// TIA Portal V17 export
// export: Created 2025-05-22T05:59:43.897412Z, ExportSetting WithDefaults, DisplayName Totally Integrated Automation Portal, DisplayVersion V17 Update 8, DisplayName TIA Portal Openness, DisplayVersion V17 Update 8, DisplayName TIA Portal Version Control Interface, DisplayVersion V17, DisplayName SINAMICS Startdrive Advanced, DisplayVersion V17 SP2, DisplayName SINAMICS Startdrive G110M, G120, G120C, G120D, G120P, G115D, DisplayVersion V17 SP2, DisplayName SINAMICS Startdrive G130, G150, S120, S150, SINAMICS MV, S210, DisplayVersion V17 SP2, DisplayName STEP 7 Professional, DisplayVersion V17 Update 8, DisplayName SINUMERIK ONE STEP 7 Toolbox, DisplayVersion V17 Update 12, DisplayName SINUMERIK ONE PLC Basic Program Plus, DisplayVersion V17 Update 12, DisplayName SINUMERIK 840D sl STEP 7 Toolbox, DisplayVersion V17 Update 12, DisplayName STEP 7 Safety, DisplayVersion V17 Update 6, DisplayName WinCC Advanced, DisplayVersion V17 Update 8
FUNCTION "FC7331_MACHINE_TO_ROBOT_CELL_INTERLOCK" : Void   // FC7331, LAD
{ S7_Optimized_Access := 'FALSE' }
AUTHOR : ETXETAR
VERSION : 1.0
// stored: AutoNumber false, IsIECCheckEnabled false, SetENOAutomatically false, UDAEnableTagReadback false
   VAR_TEMP
      OPTION_OFF : Bool;
      OPTION_ON : Bool;
      dry_load_side0 : Bool;
      dry_load_side180 : Bool;
      Status_receive : Int;
      QC_FORECAST : Int;
      QC_EXPIRED : Int;
      QC_COUNTS : Int;
      RETVAL_FILL : Int;
      temp0 : Int;
      status_sfc21 : Int;
      RETVAL_FILL_1 : Int;
      ONE : Byte;
      ZERO : Byte;
      retval_sfc21 : Int;
      Counts_for_error : Int;
      AUX_1_GTRY_SWITCH_OFF : Bool;
      AUX_2_GTRY_SWITCH_OFF : Bool;
      WITH_MANUAL_LOADER : Bool;
      WITH_OUT_MANUAL_LOADER : Bool;
      PART_TYPE_POSSIBLE : Bool;
      SHIFTING_DEVICES_OK : Bool;
      PART_ID_NEXT_FIXT : Bool;
      PART_TYPE_GTY : Bool;
      STATUS : Byte;
      RET : Byte;
   END_VAR
   VAR CONSTANT
      FC_NUMBER : DInt := 7331;   // FC NUMBER
   END_VAR
   VAR_TEMP   // added for the SCL form of the ladder/FBD networks
      _w1 : Bool;
   END_VAR
BEGIN

REGION Network 1: >>>>>>>>>>>>>>>> INTERLOCKS MACHINE TO CELL GENERAL <<<<<<<<<<<<<<<<
END_REGION

REGION Network 2: MACHINE MEASURING STATION CALIBRATION REQUIRED
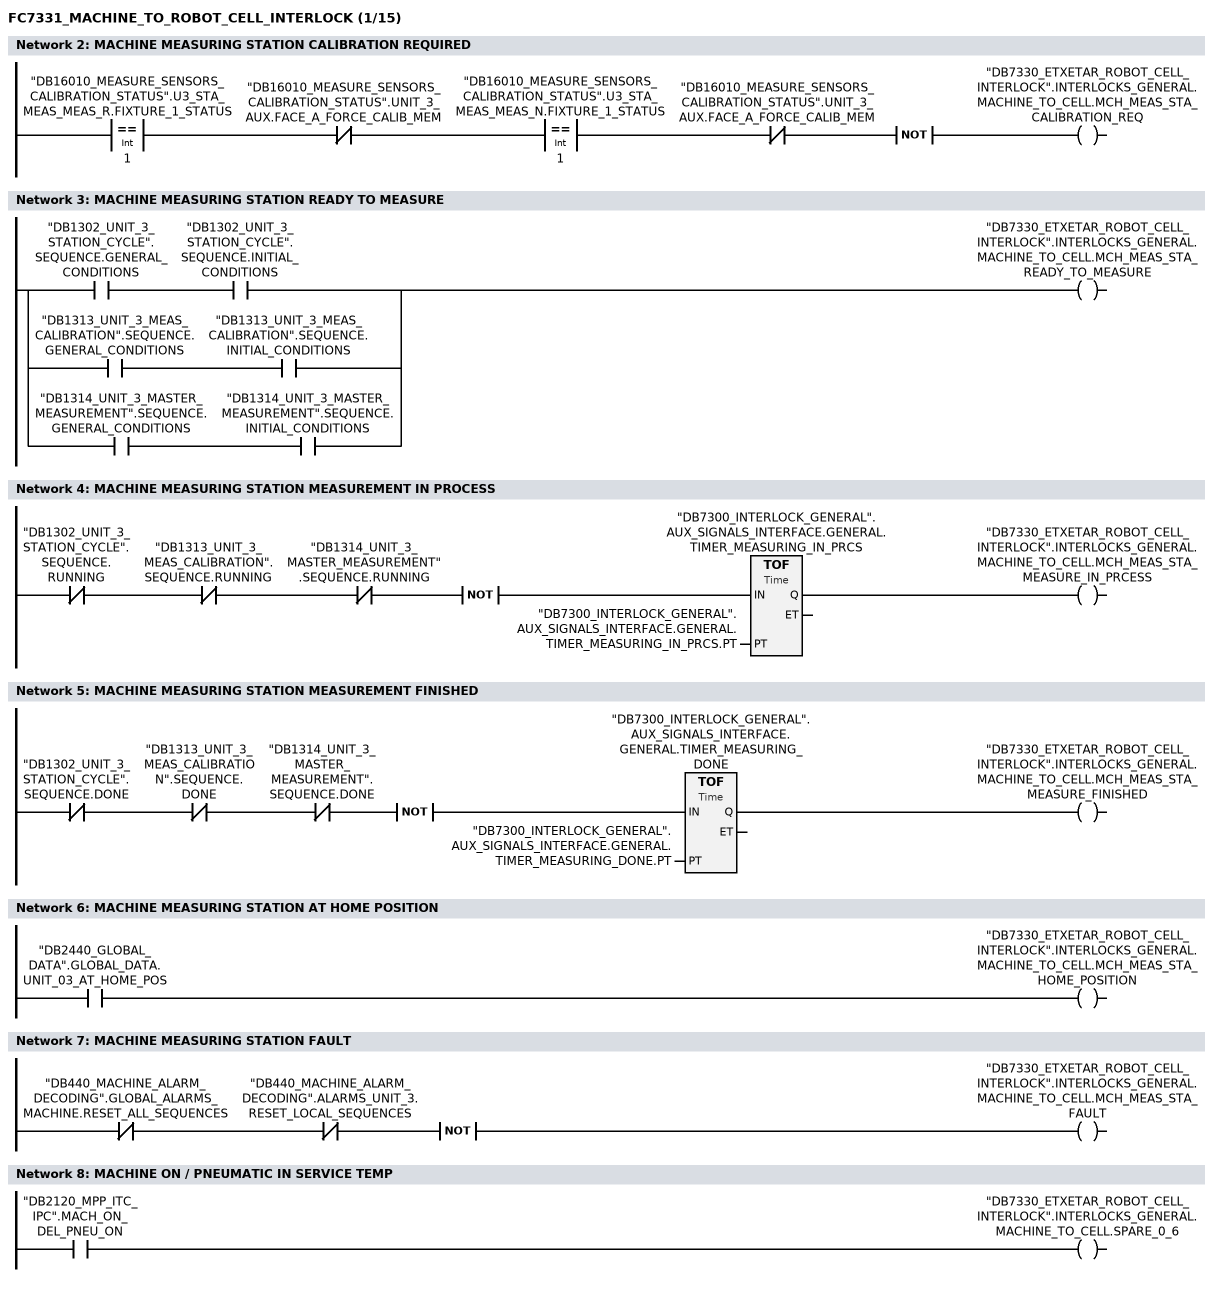
   RUNG wire#powerrail
      { S7_Templates := "SrcType := Int" } EQ_Contact(in1 := "DB16010_MEASURE_SENSORS_CALIBRATION_STATUS".U3_STA_MEAS_MEAS_R.FIXTURE_1_STATUS, in2 := 1)
      I_Contact( "DB16010_MEASURE_SENSORS_CALIBRATION_STATUS".UNIT_3_AUX.FACE_A_FORCE_CALIB_MEM )
      { S7_Templates := "SrcType := Int" } EQ_Contact(in1 := "DB16010_MEASURE_SENSORS_CALIBRATION_STATUS".U3_STA_MEAS_MEAS_N.FIXTURE_1_STATUS, in2 := 1)
      I_Contact( "DB16010_MEASURE_SENSORS_CALIBRATION_STATUS".UNIT_3_AUX.FACE_A_FORCE_CALIB_MEM )
      Not()
      Coil( "DB7330_ETXETAR_ROBOT_CELL_INTERLOCK".INTERLOCKS_GENERAL.MACHINE_TO_CELL.MCH_MEAS_STA_CALIBRATION_REQ )
   END_RUNG
   // the same network as SCL:
   "DB7330_ETXETAR_ROBOT_CELL_INTERLOCK".INTERLOCKS_GENERAL.MACHINE_TO_CELL.MCH_MEAS_STA_CALIBRATION_REQ := NOT (("DB16010_MEASURE_SENSORS_CALIBRATION_STATUS".U3_STA_MEAS_MEAS_R.FIXTURE_1_STATUS = 1) AND NOT "DB16010_MEASURE_SENSORS_CALIBRATION_STATUS".UNIT_3_AUX.FACE_A_FORCE_CALIB_MEM AND ("DB16010_MEASURE_SENSORS_CALIBRATION_STATUS".U3_STA_MEAS_MEAS_N.FIXTURE_1_STATUS = 1) AND NOT "DB16010_MEASURE_SENSORS_CALIBRATION_STATUS".UNIT_3_AUX.FACE_A_FORCE_CALIB_MEM);
END_REGION

REGION Network 3: MACHINE MEASURING STATION READY TO MEASURE
   RUNG wire#powerrail
      Contact( "DB1302_UNIT_3_STATION_CYCLE".SEQUENCE.GENERAL_CONDITIONS )
      Contact( "DB1302_UNIT_3_STATION_CYCLE".SEQUENCE.INITIAL_CONDITIONS )
      wire#w1
      Coil( "DB7330_ETXETAR_ROBOT_CELL_INTERLOCK".INTERLOCKS_GENERAL.MACHINE_TO_CELL.MCH_MEAS_STA_READY_TO_MEASURE )
   END_RUNG
   RUNG wire#powerrail
      Contact( "DB1313_UNIT_3_MEAS_CALIBRATION".SEQUENCE.GENERAL_CONDITIONS )
      Contact( "DB1313_UNIT_3_MEAS_CALIBRATION".SEQUENCE.INITIAL_CONDITIONS )
   END_RUNG wire#w1
   RUNG wire#powerrail
      Contact( "DB1314_UNIT_3_MASTER_MEASUREMENT".SEQUENCE.GENERAL_CONDITIONS )
      Contact( "DB1314_UNIT_3_MASTER_MEASUREMENT".SEQUENCE.INITIAL_CONDITIONS )
   END_RUNG wire#w1
   // the same network as SCL:
   "DB7330_ETXETAR_ROBOT_CELL_INTERLOCK".INTERLOCKS_GENERAL.MACHINE_TO_CELL.MCH_MEAS_STA_READY_TO_MEASURE := ("DB1302_UNIT_3_STATION_CYCLE".SEQUENCE.GENERAL_CONDITIONS AND "DB1302_UNIT_3_STATION_CYCLE".SEQUENCE.INITIAL_CONDITIONS) OR ("DB1313_UNIT_3_MEAS_CALIBRATION".SEQUENCE.GENERAL_CONDITIONS AND "DB1313_UNIT_3_MEAS_CALIBRATION".SEQUENCE.INITIAL_CONDITIONS) OR ("DB1314_UNIT_3_MASTER_MEASUREMENT".SEQUENCE.GENERAL_CONDITIONS AND "DB1314_UNIT_3_MASTER_MEASUREMENT".SEQUENCE.INITIAL_CONDITIONS);
END_REGION

REGION Network 4: MACHINE MEASURING STATION MEASUREMENT IN PROCESS
   RUNG wire#powerrail
      I_Contact( "DB1302_UNIT_3_STATION_CYCLE".SEQUENCE.RUNNING )
      I_Contact( "DB1313_UNIT_3_MEAS_CALIBRATION".SEQUENCE.RUNNING )
      I_Contact( "DB1314_UNIT_3_MASTER_MEASUREMENT".SEQUENCE.RUNNING )
      Not()
      { S7_Templates := "time_type := Time" } "DB7300_INTERLOCK_GENERAL".AUX_SIGNALS_INTERFACE.GENERAL.TIMER_MEASURING_IN_PRCS.TOF(pt := "DB7300_INTERLOCK_GENERAL".AUX_SIGNALS_INTERFACE.GENERAL.TIMER_MEASURING_IN_PRCS.PT, et =>)
      Coil( "DB7330_ETXETAR_ROBOT_CELL_INTERLOCK".INTERLOCKS_GENERAL.MACHINE_TO_CELL.MCH_MEAS_STA_MEASURE_IN_PRCESS )
   END_RUNG
   // the same network as SCL:
   "DB7300_INTERLOCK_GENERAL".AUX_SIGNALS_INTERFACE.GENERAL.TIMER_MEASURING_IN_PRCS.TOF(IN := NOT (NOT "DB1302_UNIT_3_STATION_CYCLE".SEQUENCE.RUNNING AND NOT "DB1313_UNIT_3_MEAS_CALIBRATION".SEQUENCE.RUNNING AND NOT "DB1314_UNIT_3_MASTER_MEASUREMENT".SEQUENCE.RUNNING),
                           PT := "DB7300_INTERLOCK_GENERAL".AUX_SIGNALS_INTERFACE.GENERAL.TIMER_MEASURING_IN_PRCS.PT);
   "DB7330_ETXETAR_ROBOT_CELL_INTERLOCK".INTERLOCKS_GENERAL.MACHINE_TO_CELL.MCH_MEAS_STA_MEASURE_IN_PRCESS := "DB7300_INTERLOCK_GENERAL".AUX_SIGNALS_INTERFACE.GENERAL.TIMER_MEASURING_IN_PRCS.Q;
END_REGION

REGION Network 5: MACHINE MEASURING STATION MEASUREMENT FINISHED
   RUNG wire#powerrail
      I_Contact( "DB1302_UNIT_3_STATION_CYCLE".SEQUENCE.DONE )
      I_Contact( "DB1313_UNIT_3_MEAS_CALIBRATION".SEQUENCE.DONE )
      I_Contact( "DB1314_UNIT_3_MASTER_MEASUREMENT".SEQUENCE.DONE )
      Not()
      { S7_Templates := "time_type := Time" } "DB7300_INTERLOCK_GENERAL".AUX_SIGNALS_INTERFACE.GENERAL.TIMER_MEASURING_DONE.TOF(pt := "DB7300_INTERLOCK_GENERAL".AUX_SIGNALS_INTERFACE.GENERAL.TIMER_MEASURING_DONE.PT, et =>)
      Coil( "DB7330_ETXETAR_ROBOT_CELL_INTERLOCK".INTERLOCKS_GENERAL.MACHINE_TO_CELL.MCH_MEAS_STA_MEASURE_FINISHED )
   END_RUNG
   // the same network as SCL:
   "DB7300_INTERLOCK_GENERAL".AUX_SIGNALS_INTERFACE.GENERAL.TIMER_MEASURING_DONE.TOF(IN := NOT (NOT "DB1302_UNIT_3_STATION_CYCLE".SEQUENCE.DONE AND NOT "DB1313_UNIT_3_MEAS_CALIBRATION".SEQUENCE.DONE AND NOT "DB1314_UNIT_3_MASTER_MEASUREMENT".SEQUENCE.DONE),
                           PT := "DB7300_INTERLOCK_GENERAL".AUX_SIGNALS_INTERFACE.GENERAL.TIMER_MEASURING_DONE.PT);
   "DB7330_ETXETAR_ROBOT_CELL_INTERLOCK".INTERLOCKS_GENERAL.MACHINE_TO_CELL.MCH_MEAS_STA_MEASURE_FINISHED := "DB7300_INTERLOCK_GENERAL".AUX_SIGNALS_INTERFACE.GENERAL.TIMER_MEASURING_DONE.Q;
END_REGION

REGION Network 6: MACHINE MEASURING STATION AT HOME POSITION
   RUNG wire#powerrail
      Contact( "DB2440_GLOBAL_DATA".GLOBAL_DATA.UNIT_03_AT_HOME_POS )
      Coil( "DB7330_ETXETAR_ROBOT_CELL_INTERLOCK".INTERLOCKS_GENERAL.MACHINE_TO_CELL.MCH_MEAS_STA_HOME_POSITION )
   END_RUNG
   // the same network as SCL:
   "DB7330_ETXETAR_ROBOT_CELL_INTERLOCK".INTERLOCKS_GENERAL.MACHINE_TO_CELL.MCH_MEAS_STA_HOME_POSITION := "DB2440_GLOBAL_DATA".GLOBAL_DATA.UNIT_03_AT_HOME_POS;
END_REGION

REGION Network 7: MACHINE MEASURING STATION FAULT
   RUNG wire#powerrail
      I_Contact( "DB440_MACHINE_ALARM_DECODING".GLOBAL_ALARMS_MACHINE.RESET_ALL_SEQUENCES )
      I_Contact( "DB440_MACHINE_ALARM_DECODING".ALARMS_UNIT_3.RESET_LOCAL_SEQUENCES )
      Not()
      Coil( "DB7330_ETXETAR_ROBOT_CELL_INTERLOCK".INTERLOCKS_GENERAL.MACHINE_TO_CELL.MCH_MEAS_STA_FAULT )
   END_RUNG
   // the same network as SCL:
   "DB7330_ETXETAR_ROBOT_CELL_INTERLOCK".INTERLOCKS_GENERAL.MACHINE_TO_CELL.MCH_MEAS_STA_FAULT := NOT (NOT "DB440_MACHINE_ALARM_DECODING".GLOBAL_ALARMS_MACHINE.RESET_ALL_SEQUENCES AND NOT "DB440_MACHINE_ALARM_DECODING".ALARMS_UNIT_3.RESET_LOCAL_SEQUENCES);
END_REGION

REGION Network 8: MACHINE ON / PNEUMATIC IN SERVICE TEMP
   RUNG wire#powerrail
      Contact( "DB2120_MPP_ITC_IPC".MACH_ON_DEL_PNEU_ON )
      Coil( "DB7330_ETXETAR_ROBOT_CELL_INTERLOCK".INTERLOCKS_GENERAL.MACHINE_TO_CELL.SPARE_0_6 )
   END_RUNG
   // the same network as SCL:
   "DB7330_ETXETAR_ROBOT_CELL_INTERLOCK".INTERLOCKS_GENERAL.MACHINE_TO_CELL.SPARE_0_6 := "DB2120_MPP_ITC_IPC".MACH_ON_DEL_PNEU_ON;
END_REGION

REGION Network 9: MACHINE MEASURING STATION MICROEPSILON FACE R ENABLED
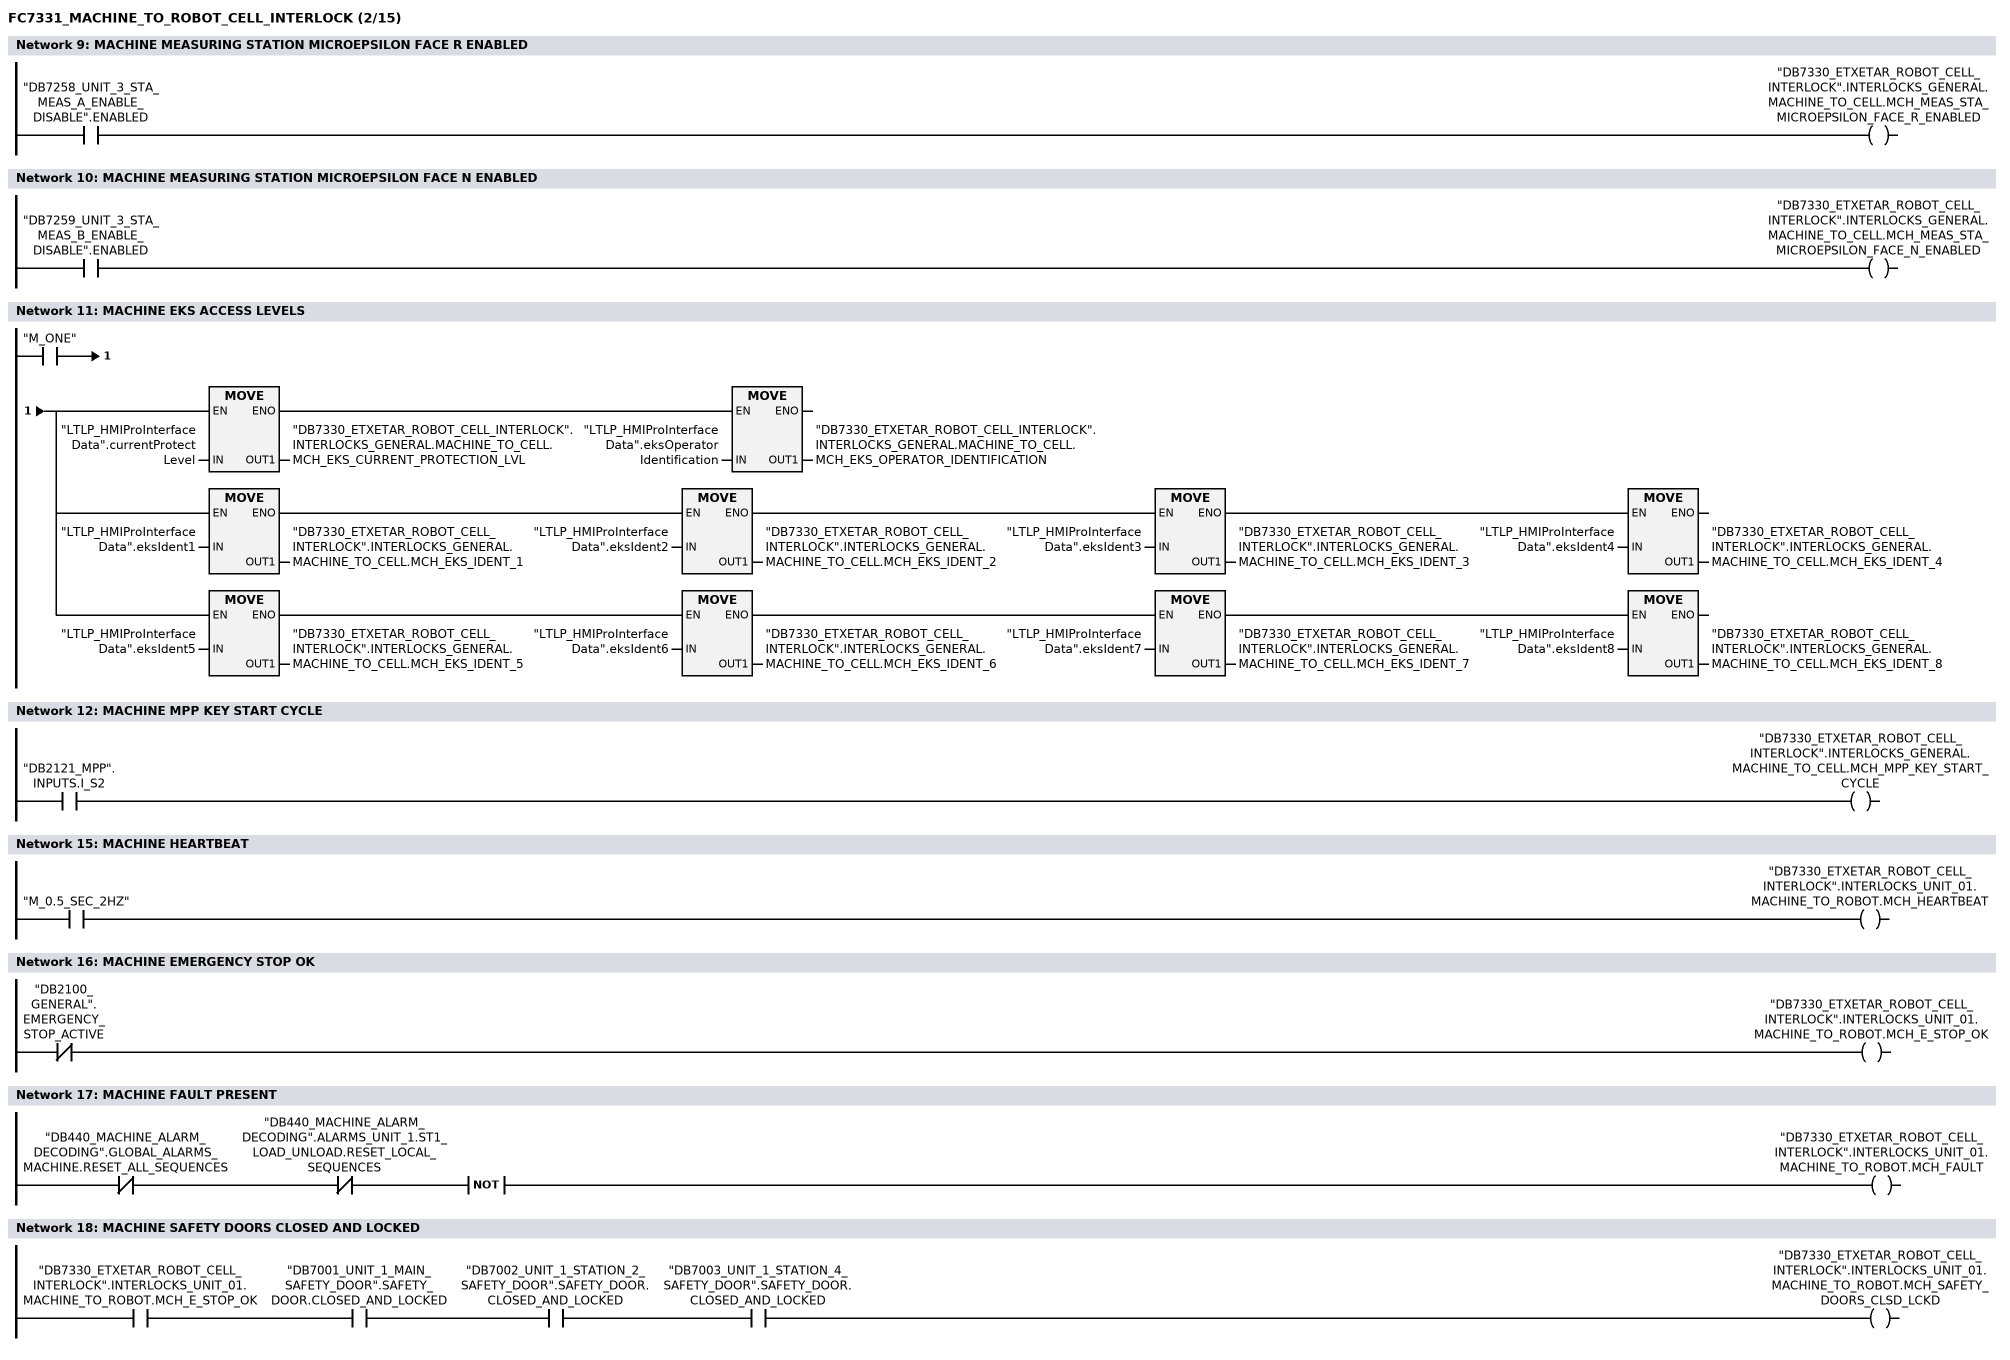
   RUNG wire#powerrail
      Contact( "DB7258_UNIT_3_STA_MEAS_A_ENABLE_DISABLE".ENABLED )
      Coil( "DB7330_ETXETAR_ROBOT_CELL_INTERLOCK".INTERLOCKS_GENERAL.MACHINE_TO_CELL.MCH_MEAS_STA_MICROEPSILON_FACE_R_ENABLED )
   END_RUNG
   // the same network as SCL:
   "DB7330_ETXETAR_ROBOT_CELL_INTERLOCK".INTERLOCKS_GENERAL.MACHINE_TO_CELL.MCH_MEAS_STA_MICROEPSILON_FACE_R_ENABLED := "DB7258_UNIT_3_STA_MEAS_A_ENABLE_DISABLE".ENABLED;
END_REGION

REGION Network 10: MACHINE MEASURING STATION MICROEPSILON FACE N ENABLED
   RUNG wire#powerrail
      Contact( "DB7259_UNIT_3_STA_MEAS_B_ENABLE_DISABLE".ENABLED )
      Coil( "DB7330_ETXETAR_ROBOT_CELL_INTERLOCK".INTERLOCKS_GENERAL.MACHINE_TO_CELL.MCH_MEAS_STA_MICROEPSILON_FACE_N_ENABLED )
   END_RUNG
   // the same network as SCL:
   "DB7330_ETXETAR_ROBOT_CELL_INTERLOCK".INTERLOCKS_GENERAL.MACHINE_TO_CELL.MCH_MEAS_STA_MICROEPSILON_FACE_N_ENABLED := "DB7259_UNIT_3_STA_MEAS_B_ENABLE_DISABLE".ENABLED;
END_REGION

REGION Network 11: MACHINE EKS ACCESS LEVELS
   RUNG wire#powerrail
      Contact( "M_ONE" )
      wire#w1
      Move(in := "LTLP_HMIProInterfaceData".currentProtectLevel, out1 => "DB7330_ETXETAR_ROBOT_CELL_INTERLOCK".INTERLOCKS_GENERAL.MACHINE_TO_CELL.MCH_EKS_CURRENT_PROTECTION_LVL)
      Move(in := "LTLP_HMIProInterfaceData".eksOperatorIdentification, out1 => "DB7330_ETXETAR_ROBOT_CELL_INTERLOCK".INTERLOCKS_GENERAL.MACHINE_TO_CELL.MCH_EKS_OPERATOR_IDENTIFICATION)
   END_RUNG
   RUNG wire#w1
      Move(in := "LTLP_HMIProInterfaceData".eksIdent1, out1 => "DB7330_ETXETAR_ROBOT_CELL_INTERLOCK".INTERLOCKS_GENERAL.MACHINE_TO_CELL.MCH_EKS_IDENT_1)
      Move(in := "LTLP_HMIProInterfaceData".eksIdent2, out1 => "DB7330_ETXETAR_ROBOT_CELL_INTERLOCK".INTERLOCKS_GENERAL.MACHINE_TO_CELL.MCH_EKS_IDENT_2)
      Move(in := "LTLP_HMIProInterfaceData".eksIdent3, out1 => "DB7330_ETXETAR_ROBOT_CELL_INTERLOCK".INTERLOCKS_GENERAL.MACHINE_TO_CELL.MCH_EKS_IDENT_3)
      Move(in := "LTLP_HMIProInterfaceData".eksIdent4, out1 => "DB7330_ETXETAR_ROBOT_CELL_INTERLOCK".INTERLOCKS_GENERAL.MACHINE_TO_CELL.MCH_EKS_IDENT_4)
   END_RUNG
   RUNG wire#w1
      Move(in := "LTLP_HMIProInterfaceData".eksIdent5, out1 => "DB7330_ETXETAR_ROBOT_CELL_INTERLOCK".INTERLOCKS_GENERAL.MACHINE_TO_CELL.MCH_EKS_IDENT_5)
      Move(in := "LTLP_HMIProInterfaceData".eksIdent6, out1 => "DB7330_ETXETAR_ROBOT_CELL_INTERLOCK".INTERLOCKS_GENERAL.MACHINE_TO_CELL.MCH_EKS_IDENT_6)
      Move(in := "LTLP_HMIProInterfaceData".eksIdent7, out1 => "DB7330_ETXETAR_ROBOT_CELL_INTERLOCK".INTERLOCKS_GENERAL.MACHINE_TO_CELL.MCH_EKS_IDENT_7)
      Move(in := "LTLP_HMIProInterfaceData".eksIdent8, out1 => "DB7330_ETXETAR_ROBOT_CELL_INTERLOCK".INTERLOCKS_GENERAL.MACHINE_TO_CELL.MCH_EKS_IDENT_8)
   END_RUNG
   // the same network as SCL:
   IF "M_ONE" THEN
       "DB7330_ETXETAR_ROBOT_CELL_INTERLOCK".INTERLOCKS_GENERAL.MACHINE_TO_CELL.MCH_EKS_CURRENT_PROTECTION_LVL := "LTLP_HMIProInterfaceData".currentProtectLevel;
       "DB7330_ETXETAR_ROBOT_CELL_INTERLOCK".INTERLOCKS_GENERAL.MACHINE_TO_CELL.MCH_EKS_OPERATOR_IDENTIFICATION := "LTLP_HMIProInterfaceData".eksOperatorIdentification;
       "DB7330_ETXETAR_ROBOT_CELL_INTERLOCK".INTERLOCKS_GENERAL.MACHINE_TO_CELL.MCH_EKS_IDENT_1 := "LTLP_HMIProInterfaceData".eksIdent1;
       "DB7330_ETXETAR_ROBOT_CELL_INTERLOCK".INTERLOCKS_GENERAL.MACHINE_TO_CELL.MCH_EKS_IDENT_2 := "LTLP_HMIProInterfaceData".eksIdent2;
       "DB7330_ETXETAR_ROBOT_CELL_INTERLOCK".INTERLOCKS_GENERAL.MACHINE_TO_CELL.MCH_EKS_IDENT_3 := "LTLP_HMIProInterfaceData".eksIdent3;
       "DB7330_ETXETAR_ROBOT_CELL_INTERLOCK".INTERLOCKS_GENERAL.MACHINE_TO_CELL.MCH_EKS_IDENT_4 := "LTLP_HMIProInterfaceData".eksIdent4;
       "DB7330_ETXETAR_ROBOT_CELL_INTERLOCK".INTERLOCKS_GENERAL.MACHINE_TO_CELL.MCH_EKS_IDENT_5 := "LTLP_HMIProInterfaceData".eksIdent5;
       "DB7330_ETXETAR_ROBOT_CELL_INTERLOCK".INTERLOCKS_GENERAL.MACHINE_TO_CELL.MCH_EKS_IDENT_6 := "LTLP_HMIProInterfaceData".eksIdent6;
       "DB7330_ETXETAR_ROBOT_CELL_INTERLOCK".INTERLOCKS_GENERAL.MACHINE_TO_CELL.MCH_EKS_IDENT_7 := "LTLP_HMIProInterfaceData".eksIdent7;
       "DB7330_ETXETAR_ROBOT_CELL_INTERLOCK".INTERLOCKS_GENERAL.MACHINE_TO_CELL.MCH_EKS_IDENT_8 := "LTLP_HMIProInterfaceData".eksIdent8;
   END_IF;
END_REGION

REGION Network 12: MACHINE MPP KEY START CYCLE
   RUNG wire#powerrail
      Contact( "DB2121_MPP".INPUTS.I_S2 )
      Coil( "DB7330_ETXETAR_ROBOT_CELL_INTERLOCK".INTERLOCKS_GENERAL.MACHINE_TO_CELL.MCH_MPP_KEY_START_CYCLE )
   END_RUNG
   // the same network as SCL:
   "DB7330_ETXETAR_ROBOT_CELL_INTERLOCK".INTERLOCKS_GENERAL.MACHINE_TO_CELL.MCH_MPP_KEY_START_CYCLE := "DB2121_MPP".INPUTS.I_S2;
END_REGION

REGION Network 14: >>>>>>>>>>>>>>>> INTERLOCKS MACHINE TO ROBOT UNIT 01 <<<<<<<<<<<<<<<<
END_REGION

REGION Network 15: MACHINE HEARTBEAT
   RUNG wire#powerrail
      Contact( "M_0.5_SEC_2HZ" )
      Coil( "DB7330_ETXETAR_ROBOT_CELL_INTERLOCK".INTERLOCKS_UNIT_01.MACHINE_TO_ROBOT.MCH_HEARTBEAT )
   END_RUNG
   // the same network as SCL:
   "DB7330_ETXETAR_ROBOT_CELL_INTERLOCK".INTERLOCKS_UNIT_01.MACHINE_TO_ROBOT.MCH_HEARTBEAT := "M_0.5_SEC_2HZ";
END_REGION

REGION Network 16: MACHINE EMERGENCY STOP OK
   RUNG wire#powerrail
      I_Contact( "DB2100_GENERAL".EMERGENCY_STOP_ACTIVE )
      Coil( "DB7330_ETXETAR_ROBOT_CELL_INTERLOCK".INTERLOCKS_UNIT_01.MACHINE_TO_ROBOT.MCH_E_STOP_OK )
   END_RUNG
   // the same network as SCL:
   "DB7330_ETXETAR_ROBOT_CELL_INTERLOCK".INTERLOCKS_UNIT_01.MACHINE_TO_ROBOT.MCH_E_STOP_OK := NOT "DB2100_GENERAL".EMERGENCY_STOP_ACTIVE;
END_REGION

REGION Network 17: MACHINE FAULT PRESENT
   RUNG wire#powerrail
      I_Contact( "DB440_MACHINE_ALARM_DECODING".GLOBAL_ALARMS_MACHINE.RESET_ALL_SEQUENCES )
      I_Contact( "DB440_MACHINE_ALARM_DECODING".ALARMS_UNIT_1.ST1_LOAD_UNLOAD.RESET_LOCAL_SEQUENCES )
      Not()
      Coil( "DB7330_ETXETAR_ROBOT_CELL_INTERLOCK".INTERLOCKS_UNIT_01.MACHINE_TO_ROBOT.MCH_FAULT )
   END_RUNG
   // the same network as SCL:
   "DB7330_ETXETAR_ROBOT_CELL_INTERLOCK".INTERLOCKS_UNIT_01.MACHINE_TO_ROBOT.MCH_FAULT := NOT (NOT "DB440_MACHINE_ALARM_DECODING".GLOBAL_ALARMS_MACHINE.RESET_ALL_SEQUENCES AND NOT "DB440_MACHINE_ALARM_DECODING".ALARMS_UNIT_1.ST1_LOAD_UNLOAD.RESET_LOCAL_SEQUENCES);
END_REGION

REGION Network 18: MACHINE SAFETY DOORS CLOSED AND LOCKED
   RUNG wire#powerrail
      Contact( "DB7330_ETXETAR_ROBOT_CELL_INTERLOCK".INTERLOCKS_UNIT_01.MACHINE_TO_ROBOT.MCH_E_STOP_OK )
      Contact( "DB7001_UNIT_1_MAIN_SAFETY_DOOR".SAFETY_DOOR.CLOSED_AND_LOCKED )
      Contact( "DB7002_UNIT_1_STATION_2_SAFETY_DOOR".SAFETY_DOOR.CLOSED_AND_LOCKED )
      Contact( "DB7003_UNIT_1_STATION_4_SAFETY_DOOR".SAFETY_DOOR.CLOSED_AND_LOCKED )
      Coil( "DB7330_ETXETAR_ROBOT_CELL_INTERLOCK".INTERLOCKS_UNIT_01.MACHINE_TO_ROBOT.MCH_SAFETY_DOORS_CLSD_LCKD )
   END_RUNG
   // the same network as SCL:
   "DB7330_ETXETAR_ROBOT_CELL_INTERLOCK".INTERLOCKS_UNIT_01.MACHINE_TO_ROBOT.MCH_SAFETY_DOORS_CLSD_LCKD := "DB7330_ETXETAR_ROBOT_CELL_INTERLOCK".INTERLOCKS_UNIT_01.MACHINE_TO_ROBOT.MCH_E_STOP_OK AND "DB7001_UNIT_1_MAIN_SAFETY_DOOR".SAFETY_DOOR.CLOSED_AND_LOCKED AND "DB7002_UNIT_1_STATION_2_SAFETY_DOOR".SAFETY_DOOR.CLOSED_AND_LOCKED AND "DB7003_UNIT_1_STATION_4_SAFETY_DOOR".SAFETY_DOOR.CLOSED_AND_LOCKED;
END_REGION

REGION Network 19: MACHINE MANUAL MODE SELECTED
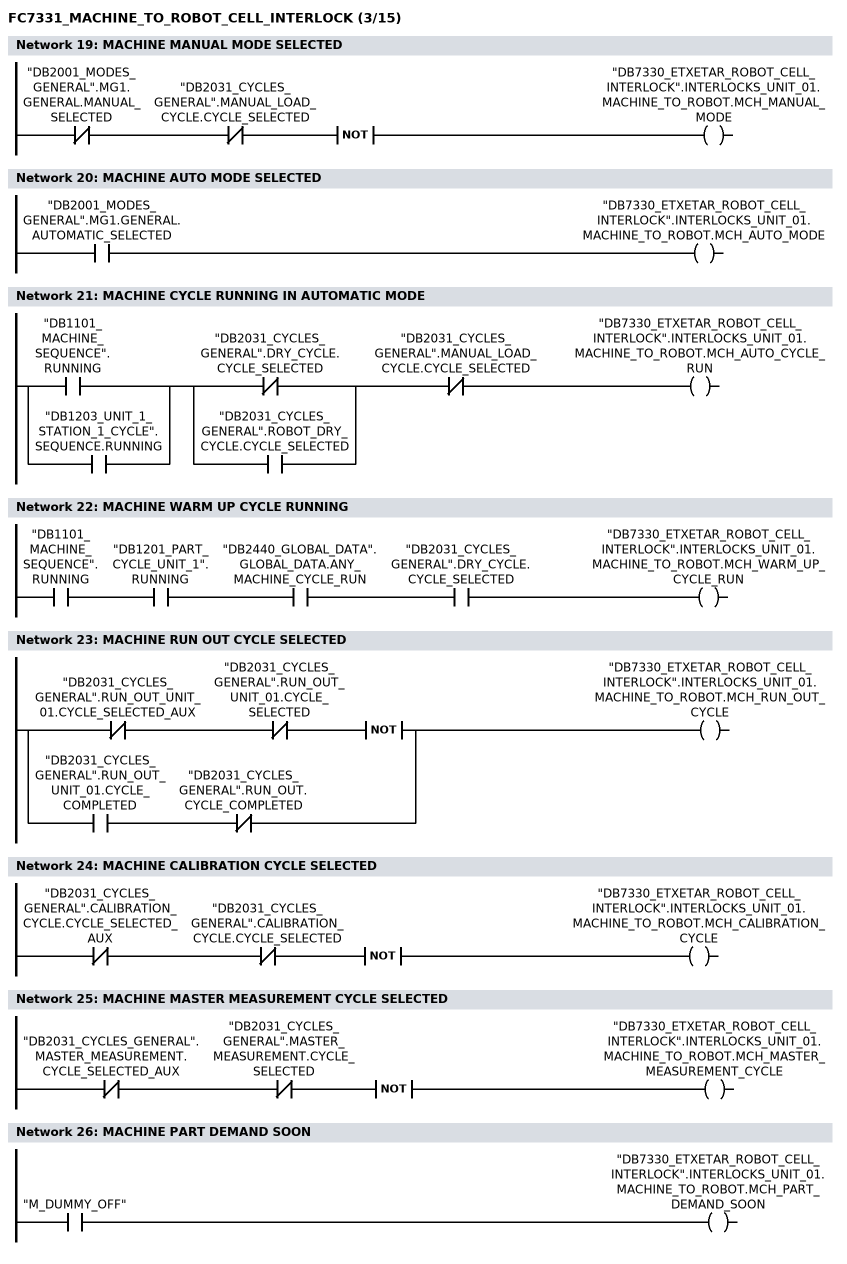
   RUNG wire#powerrail
      I_Contact( "DB2001_MODES_GENERAL".MG1.GENERAL.MANUAL_SELECTED )
      I_Contact( "DB2031_CYCLES_GENERAL".MANUAL_LOAD_CYCLE.CYCLE_SELECTED )
      Not()
      Coil( "DB7330_ETXETAR_ROBOT_CELL_INTERLOCK".INTERLOCKS_UNIT_01.MACHINE_TO_ROBOT.MCH_MANUAL_MODE )
   END_RUNG
   // the same network as SCL:
   "DB7330_ETXETAR_ROBOT_CELL_INTERLOCK".INTERLOCKS_UNIT_01.MACHINE_TO_ROBOT.MCH_MANUAL_MODE := NOT (NOT "DB2001_MODES_GENERAL".MG1.GENERAL.MANUAL_SELECTED AND NOT "DB2031_CYCLES_GENERAL".MANUAL_LOAD_CYCLE.CYCLE_SELECTED);
END_REGION

REGION Network 20: MACHINE AUTO MODE SELECTED
   RUNG wire#powerrail
      Contact( "DB2001_MODES_GENERAL".MG1.GENERAL.AUTOMATIC_SELECTED )
      Coil( "DB7330_ETXETAR_ROBOT_CELL_INTERLOCK".INTERLOCKS_UNIT_01.MACHINE_TO_ROBOT.MCH_AUTO_MODE )
   END_RUNG
   // the same network as SCL:
   "DB7330_ETXETAR_ROBOT_CELL_INTERLOCK".INTERLOCKS_UNIT_01.MACHINE_TO_ROBOT.MCH_AUTO_MODE := "DB2001_MODES_GENERAL".MG1.GENERAL.AUTOMATIC_SELECTED;
END_REGION

REGION Network 21: MACHINE CYCLE RUNNING IN AUTOMATIC MODE
   RUNG wire#powerrail
      Contact( "DB1101_MACHINE_SEQUENCE".RUNNING )
      wire#w1
      I_Contact( "DB2031_CYCLES_GENERAL".DRY_CYCLE.CYCLE_SELECTED )
      wire#w2
      I_Contact( "DB2031_CYCLES_GENERAL".MANUAL_LOAD_CYCLE.CYCLE_SELECTED )
      Coil( "DB7330_ETXETAR_ROBOT_CELL_INTERLOCK".INTERLOCKS_UNIT_01.MACHINE_TO_ROBOT.MCH_AUTO_CYCLE_RUN )
   END_RUNG
   RUNG wire#powerrail
      Contact( "DB1203_UNIT_1_STATION_1_CYCLE".SEQUENCE.RUNNING )
   END_RUNG wire#w1
   RUNG wire#w1
      Contact( "DB2031_CYCLES_GENERAL".ROBOT_DRY_CYCLE.CYCLE_SELECTED )
   END_RUNG wire#w2
   // the same network as SCL:
   "DB7330_ETXETAR_ROBOT_CELL_INTERLOCK".INTERLOCKS_UNIT_01.MACHINE_TO_ROBOT.MCH_AUTO_CYCLE_RUN := ("DB1101_MACHINE_SEQUENCE".RUNNING OR "DB1203_UNIT_1_STATION_1_CYCLE".SEQUENCE.RUNNING) AND (NOT "DB2031_CYCLES_GENERAL".DRY_CYCLE.CYCLE_SELECTED OR "DB2031_CYCLES_GENERAL".ROBOT_DRY_CYCLE.CYCLE_SELECTED) AND NOT "DB2031_CYCLES_GENERAL".MANUAL_LOAD_CYCLE.CYCLE_SELECTED;
END_REGION

REGION Network 22: MACHINE WARM UP CYCLE RUNNING
   RUNG wire#powerrail
      Contact( "DB1101_MACHINE_SEQUENCE".RUNNING )
      Contact( "DB1201_PART_CYCLE_UNIT_1".RUNNING )
      Contact( "DB2440_GLOBAL_DATA".GLOBAL_DATA.ANY_MACHINE_CYCLE_RUN )
      Contact( "DB2031_CYCLES_GENERAL".DRY_CYCLE.CYCLE_SELECTED )
      Coil( "DB7330_ETXETAR_ROBOT_CELL_INTERLOCK".INTERLOCKS_UNIT_01.MACHINE_TO_ROBOT.MCH_WARM_UP_CYCLE_RUN )
   END_RUNG
   // the same network as SCL:
   "DB7330_ETXETAR_ROBOT_CELL_INTERLOCK".INTERLOCKS_UNIT_01.MACHINE_TO_ROBOT.MCH_WARM_UP_CYCLE_RUN := "DB1101_MACHINE_SEQUENCE".RUNNING AND "DB1201_PART_CYCLE_UNIT_1".RUNNING AND "DB2440_GLOBAL_DATA".GLOBAL_DATA.ANY_MACHINE_CYCLE_RUN AND "DB2031_CYCLES_GENERAL".DRY_CYCLE.CYCLE_SELECTED;
END_REGION

REGION Network 23: MACHINE RUN OUT CYCLE SELECTED
   RUNG wire#powerrail
      I_Contact( "DB2031_CYCLES_GENERAL".RUN_OUT_UNIT_01.CYCLE_SELECTED_AUX )
      I_Contact( "DB2031_CYCLES_GENERAL".RUN_OUT_UNIT_01.CYCLE_SELECTED )
      Not()
      wire#w1
      Coil( "DB7330_ETXETAR_ROBOT_CELL_INTERLOCK".INTERLOCKS_UNIT_01.MACHINE_TO_ROBOT.MCH_RUN_OUT_CYCLE )
   END_RUNG
   RUNG wire#powerrail
      Contact( "DB2031_CYCLES_GENERAL".RUN_OUT_UNIT_01.CYCLE_COMPLETED )
      I_Contact( "DB2031_CYCLES_GENERAL".RUN_OUT.CYCLE_COMPLETED )
   END_RUNG wire#w1
   // the same network as SCL:
   "DB7330_ETXETAR_ROBOT_CELL_INTERLOCK".INTERLOCKS_UNIT_01.MACHINE_TO_ROBOT.MCH_RUN_OUT_CYCLE := NOT (NOT "DB2031_CYCLES_GENERAL".RUN_OUT_UNIT_01.CYCLE_SELECTED_AUX AND NOT "DB2031_CYCLES_GENERAL".RUN_OUT_UNIT_01.CYCLE_SELECTED) OR ("DB2031_CYCLES_GENERAL".RUN_OUT_UNIT_01.CYCLE_COMPLETED AND NOT "DB2031_CYCLES_GENERAL".RUN_OUT.CYCLE_COMPLETED);
END_REGION

REGION Network 24: MACHINE CALIBRATION CYCLE SELECTED
   RUNG wire#powerrail
      I_Contact( "DB2031_CYCLES_GENERAL".CALIBRATION_CYCLE.CYCLE_SELECTED_AUX )
      I_Contact( "DB2031_CYCLES_GENERAL".CALIBRATION_CYCLE.CYCLE_SELECTED )
      Not()
      Coil( "DB7330_ETXETAR_ROBOT_CELL_INTERLOCK".INTERLOCKS_UNIT_01.MACHINE_TO_ROBOT.MCH_CALIBRATION_CYCLE )
   END_RUNG
   // the same network as SCL:
   "DB7330_ETXETAR_ROBOT_CELL_INTERLOCK".INTERLOCKS_UNIT_01.MACHINE_TO_ROBOT.MCH_CALIBRATION_CYCLE := NOT (NOT "DB2031_CYCLES_GENERAL".CALIBRATION_CYCLE.CYCLE_SELECTED_AUX AND NOT "DB2031_CYCLES_GENERAL".CALIBRATION_CYCLE.CYCLE_SELECTED);
END_REGION

REGION Network 25: MACHINE MASTER MEASUREMENT CYCLE SELECTED
   RUNG wire#powerrail
      I_Contact( "DB2031_CYCLES_GENERAL".MASTER_MEASUREMENT.CYCLE_SELECTED_AUX )
      I_Contact( "DB2031_CYCLES_GENERAL".MASTER_MEASUREMENT.CYCLE_SELECTED )
      Not()
      Coil( "DB7330_ETXETAR_ROBOT_CELL_INTERLOCK".INTERLOCKS_UNIT_01.MACHINE_TO_ROBOT.MCH_MASTER_MEASUREMENT_CYCLE )
   END_RUNG
   // the same network as SCL:
   "DB7330_ETXETAR_ROBOT_CELL_INTERLOCK".INTERLOCKS_UNIT_01.MACHINE_TO_ROBOT.MCH_MASTER_MEASUREMENT_CYCLE := NOT (NOT "DB2031_CYCLES_GENERAL".MASTER_MEASUREMENT.CYCLE_SELECTED_AUX AND NOT "DB2031_CYCLES_GENERAL".MASTER_MEASUREMENT.CYCLE_SELECTED);
END_REGION

REGION Network 26: MACHINE PART DEMAND SOON
   RUNG wire#powerrail
      Contact( "M_DUMMY_OFF" )
      Coil( "DB7330_ETXETAR_ROBOT_CELL_INTERLOCK".INTERLOCKS_UNIT_01.MACHINE_TO_ROBOT.MCH_PART_DEMAND_SOON )
   END_RUNG
   // the same network as SCL:
   "DB7330_ETXETAR_ROBOT_CELL_INTERLOCK".INTERLOCKS_UNIT_01.MACHINE_TO_ROBOT.MCH_PART_DEMAND_SOON := "M_DUMMY_OFF";
END_REGION

REGION Network 27: MACHINE SAFETY DOOR OPEN REQUEST
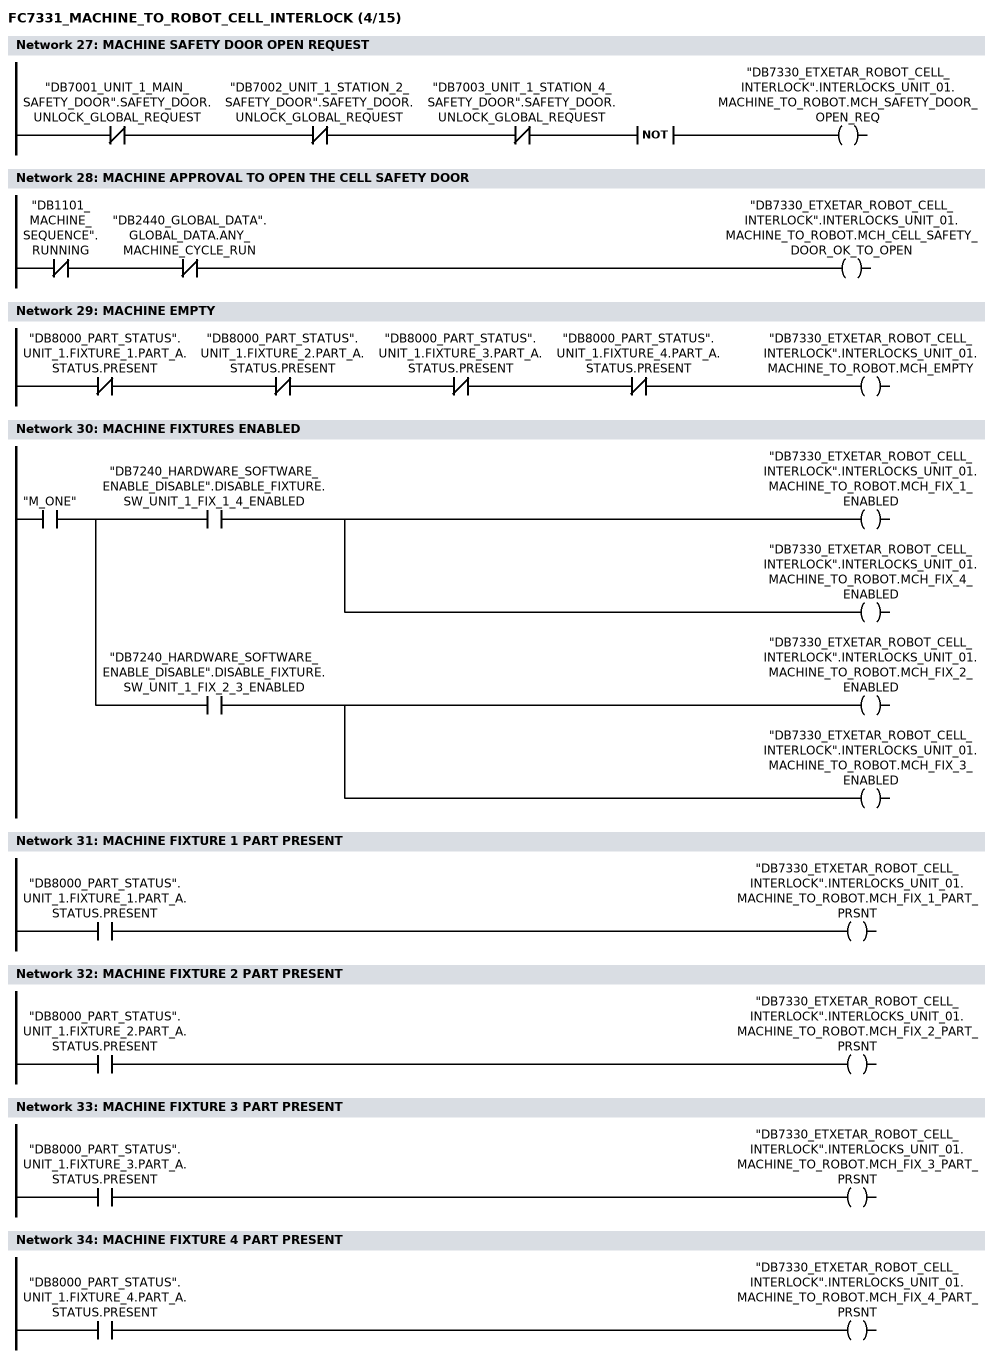
   RUNG wire#powerrail
      I_Contact( "DB7001_UNIT_1_MAIN_SAFETY_DOOR".SAFETY_DOOR.UNLOCK_GLOBAL_REQUEST )
      I_Contact( "DB7002_UNIT_1_STATION_2_SAFETY_DOOR".SAFETY_DOOR.UNLOCK_GLOBAL_REQUEST )
      I_Contact( "DB7003_UNIT_1_STATION_4_SAFETY_DOOR".SAFETY_DOOR.UNLOCK_GLOBAL_REQUEST )
      Not()
      Coil( "DB7330_ETXETAR_ROBOT_CELL_INTERLOCK".INTERLOCKS_UNIT_01.MACHINE_TO_ROBOT.MCH_SAFETY_DOOR_OPEN_REQ )
   END_RUNG
   // the same network as SCL:
   "DB7330_ETXETAR_ROBOT_CELL_INTERLOCK".INTERLOCKS_UNIT_01.MACHINE_TO_ROBOT.MCH_SAFETY_DOOR_OPEN_REQ := NOT (NOT "DB7001_UNIT_1_MAIN_SAFETY_DOOR".SAFETY_DOOR.UNLOCK_GLOBAL_REQUEST AND NOT "DB7002_UNIT_1_STATION_2_SAFETY_DOOR".SAFETY_DOOR.UNLOCK_GLOBAL_REQUEST AND NOT "DB7003_UNIT_1_STATION_4_SAFETY_DOOR".SAFETY_DOOR.UNLOCK_GLOBAL_REQUEST);
END_REGION

REGION Network 28: MACHINE APPROVAL TO OPEN THE CELL SAFETY DOOR
   RUNG wire#powerrail
      I_Contact( "DB1101_MACHINE_SEQUENCE".RUNNING )
      I_Contact( "DB2440_GLOBAL_DATA".GLOBAL_DATA.ANY_MACHINE_CYCLE_RUN )
      Coil( "DB7330_ETXETAR_ROBOT_CELL_INTERLOCK".INTERLOCKS_UNIT_01.MACHINE_TO_ROBOT.MCH_CELL_SAFETY_DOOR_OK_TO_OPEN )
   END_RUNG
   // the same network as SCL:
   "DB7330_ETXETAR_ROBOT_CELL_INTERLOCK".INTERLOCKS_UNIT_01.MACHINE_TO_ROBOT.MCH_CELL_SAFETY_DOOR_OK_TO_OPEN := NOT "DB1101_MACHINE_SEQUENCE".RUNNING AND NOT "DB2440_GLOBAL_DATA".GLOBAL_DATA.ANY_MACHINE_CYCLE_RUN;
END_REGION

REGION Network 29: MACHINE EMPTY
   RUNG wire#powerrail
      I_Contact( "DB8000_PART_STATUS".UNIT_1.FIXTURE_1.PART_A.STATUS.PRESENT )
      I_Contact( "DB8000_PART_STATUS".UNIT_1.FIXTURE_2.PART_A.STATUS.PRESENT )
      I_Contact( "DB8000_PART_STATUS".UNIT_1.FIXTURE_3.PART_A.STATUS.PRESENT )
      I_Contact( "DB8000_PART_STATUS".UNIT_1.FIXTURE_4.PART_A.STATUS.PRESENT )
      Coil( "DB7330_ETXETAR_ROBOT_CELL_INTERLOCK".INTERLOCKS_UNIT_01.MACHINE_TO_ROBOT.MCH_EMPTY )
   END_RUNG
   // the same network as SCL:
   "DB7330_ETXETAR_ROBOT_CELL_INTERLOCK".INTERLOCKS_UNIT_01.MACHINE_TO_ROBOT.MCH_EMPTY := NOT "DB8000_PART_STATUS".UNIT_1.FIXTURE_1.PART_A.STATUS.PRESENT AND NOT "DB8000_PART_STATUS".UNIT_1.FIXTURE_2.PART_A.STATUS.PRESENT AND NOT "DB8000_PART_STATUS".UNIT_1.FIXTURE_3.PART_A.STATUS.PRESENT AND NOT "DB8000_PART_STATUS".UNIT_1.FIXTURE_4.PART_A.STATUS.PRESENT;
END_REGION

REGION Network 30: MACHINE FIXTURES ENABLED
   RUNG wire#powerrail
      Contact( "M_ONE" )
      wire#w1
      Contact( "DB7240_HARDWARE_SOFTWARE_ENABLE_DISABLE".DISABLE_FIXTURE.SW_UNIT_1_FIX_1_4_ENABLED )
      wire#w2
      Coil( "DB7330_ETXETAR_ROBOT_CELL_INTERLOCK".INTERLOCKS_UNIT_01.MACHINE_TO_ROBOT.MCH_FIX_1_ENABLED )
   END_RUNG
   RUNG wire#w2
      Coil( "DB7330_ETXETAR_ROBOT_CELL_INTERLOCK".INTERLOCKS_UNIT_01.MACHINE_TO_ROBOT.MCH_FIX_4_ENABLED )
   END_RUNG
   RUNG wire#w1
      Contact( "DB7240_HARDWARE_SOFTWARE_ENABLE_DISABLE".DISABLE_FIXTURE.SW_UNIT_1_FIX_2_3_ENABLED )
      wire#w3
      Coil( "DB7330_ETXETAR_ROBOT_CELL_INTERLOCK".INTERLOCKS_UNIT_01.MACHINE_TO_ROBOT.MCH_FIX_2_ENABLED )
   END_RUNG
   RUNG wire#w3
      Coil( "DB7330_ETXETAR_ROBOT_CELL_INTERLOCK".INTERLOCKS_UNIT_01.MACHINE_TO_ROBOT.MCH_FIX_3_ENABLED )
   END_RUNG
   // the same network as SCL:
   "DB7330_ETXETAR_ROBOT_CELL_INTERLOCK".INTERLOCKS_UNIT_01.MACHINE_TO_ROBOT.MCH_FIX_1_ENABLED := "M_ONE" AND "DB7240_HARDWARE_SOFTWARE_ENABLE_DISABLE".DISABLE_FIXTURE.SW_UNIT_1_FIX_1_4_ENABLED;
   "DB7330_ETXETAR_ROBOT_CELL_INTERLOCK".INTERLOCKS_UNIT_01.MACHINE_TO_ROBOT.MCH_FIX_4_ENABLED := "DB7330_ETXETAR_ROBOT_CELL_INTERLOCK".INTERLOCKS_UNIT_01.MACHINE_TO_ROBOT.MCH_FIX_1_ENABLED;
   "DB7330_ETXETAR_ROBOT_CELL_INTERLOCK".INTERLOCKS_UNIT_01.MACHINE_TO_ROBOT.MCH_FIX_2_ENABLED := "M_ONE" AND "DB7240_HARDWARE_SOFTWARE_ENABLE_DISABLE".DISABLE_FIXTURE.SW_UNIT_1_FIX_2_3_ENABLED;
   "DB7330_ETXETAR_ROBOT_CELL_INTERLOCK".INTERLOCKS_UNIT_01.MACHINE_TO_ROBOT.MCH_FIX_3_ENABLED := "DB7330_ETXETAR_ROBOT_CELL_INTERLOCK".INTERLOCKS_UNIT_01.MACHINE_TO_ROBOT.MCH_FIX_2_ENABLED;
END_REGION

REGION Network 31: MACHINE FIXTURE 1 PART PRESENT
   RUNG wire#powerrail
      Contact( "DB8000_PART_STATUS".UNIT_1.FIXTURE_1.PART_A.STATUS.PRESENT )
      Coil( "DB7330_ETXETAR_ROBOT_CELL_INTERLOCK".INTERLOCKS_UNIT_01.MACHINE_TO_ROBOT.MCH_FIX_1_PART_PRSNT )
   END_RUNG
   // the same network as SCL:
   "DB7330_ETXETAR_ROBOT_CELL_INTERLOCK".INTERLOCKS_UNIT_01.MACHINE_TO_ROBOT.MCH_FIX_1_PART_PRSNT := "DB8000_PART_STATUS".UNIT_1.FIXTURE_1.PART_A.STATUS.PRESENT;
END_REGION

REGION Network 32: MACHINE FIXTURE 2 PART PRESENT
   RUNG wire#powerrail
      Contact( "DB8000_PART_STATUS".UNIT_1.FIXTURE_2.PART_A.STATUS.PRESENT )
      Coil( "DB7330_ETXETAR_ROBOT_CELL_INTERLOCK".INTERLOCKS_UNIT_01.MACHINE_TO_ROBOT.MCH_FIX_2_PART_PRSNT )
   END_RUNG
   // the same network as SCL:
   "DB7330_ETXETAR_ROBOT_CELL_INTERLOCK".INTERLOCKS_UNIT_01.MACHINE_TO_ROBOT.MCH_FIX_2_PART_PRSNT := "DB8000_PART_STATUS".UNIT_1.FIXTURE_2.PART_A.STATUS.PRESENT;
END_REGION

REGION Network 33: MACHINE FIXTURE 3 PART PRESENT
   RUNG wire#powerrail
      Contact( "DB8000_PART_STATUS".UNIT_1.FIXTURE_3.PART_A.STATUS.PRESENT )
      Coil( "DB7330_ETXETAR_ROBOT_CELL_INTERLOCK".INTERLOCKS_UNIT_01.MACHINE_TO_ROBOT.MCH_FIX_3_PART_PRSNT )
   END_RUNG
   // the same network as SCL:
   "DB7330_ETXETAR_ROBOT_CELL_INTERLOCK".INTERLOCKS_UNIT_01.MACHINE_TO_ROBOT.MCH_FIX_3_PART_PRSNT := "DB8000_PART_STATUS".UNIT_1.FIXTURE_3.PART_A.STATUS.PRESENT;
END_REGION

REGION Network 34: MACHINE FIXTURE 4 PART PRESENT
   RUNG wire#powerrail
      Contact( "DB8000_PART_STATUS".UNIT_1.FIXTURE_4.PART_A.STATUS.PRESENT )
      Coil( "DB7330_ETXETAR_ROBOT_CELL_INTERLOCK".INTERLOCKS_UNIT_01.MACHINE_TO_ROBOT.MCH_FIX_4_PART_PRSNT )
   END_RUNG
   // the same network as SCL:
   "DB7330_ETXETAR_ROBOT_CELL_INTERLOCK".INTERLOCKS_UNIT_01.MACHINE_TO_ROBOT.MCH_FIX_4_PART_PRSNT := "DB8000_PART_STATUS".UNIT_1.FIXTURE_4.PART_A.STATUS.PRESENT;
END_REGION

REGION Network 35: MACHINE FIXTURE 1 CALIBRATION REQUIRED
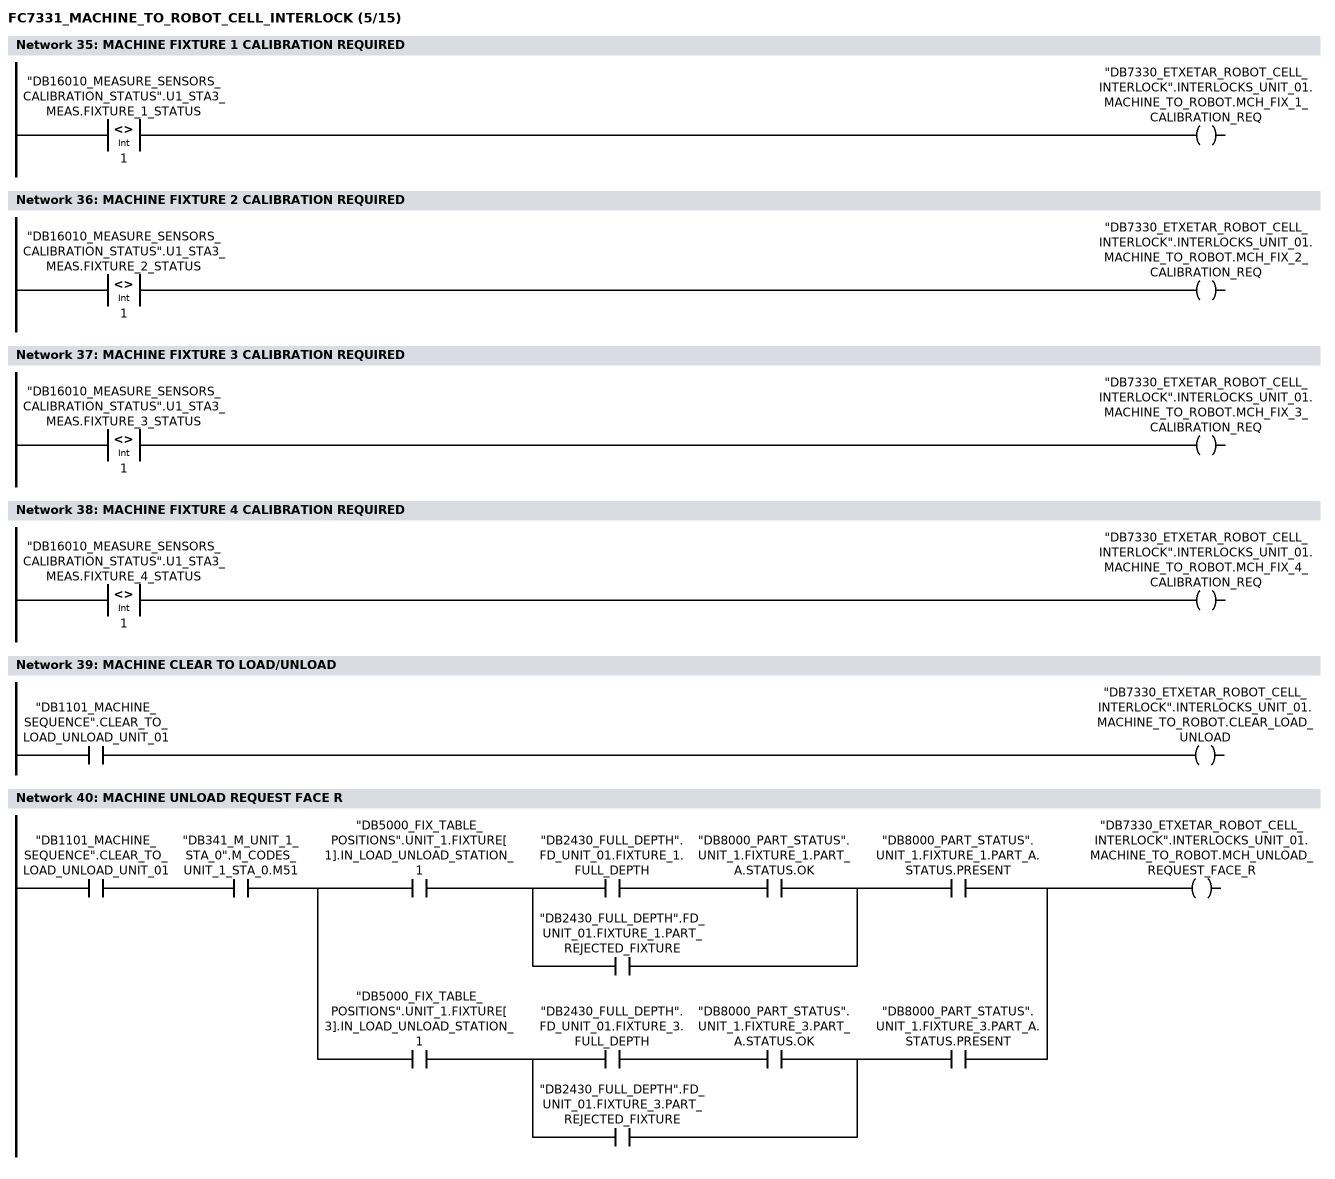
   RUNG wire#powerrail
      { S7_Templates := "SrcType := Int" } NE_Contact(in1 := "DB16010_MEASURE_SENSORS_CALIBRATION_STATUS".U1_STA3_MEAS.FIXTURE_1_STATUS, in2 := 1)
      Coil( "DB7330_ETXETAR_ROBOT_CELL_INTERLOCK".INTERLOCKS_UNIT_01.MACHINE_TO_ROBOT.MCH_FIX_1_CALIBRATION_REQ )
   END_RUNG
   // the same network as SCL:
   "DB7330_ETXETAR_ROBOT_CELL_INTERLOCK".INTERLOCKS_UNIT_01.MACHINE_TO_ROBOT.MCH_FIX_1_CALIBRATION_REQ := "DB16010_MEASURE_SENSORS_CALIBRATION_STATUS".U1_STA3_MEAS.FIXTURE_1_STATUS <> 1;
END_REGION

REGION Network 36: MACHINE FIXTURE 2 CALIBRATION REQUIRED
   RUNG wire#powerrail
      { S7_Templates := "SrcType := Int" } NE_Contact(in1 := "DB16010_MEASURE_SENSORS_CALIBRATION_STATUS".U1_STA3_MEAS.FIXTURE_2_STATUS, in2 := 1)
      Coil( "DB7330_ETXETAR_ROBOT_CELL_INTERLOCK".INTERLOCKS_UNIT_01.MACHINE_TO_ROBOT.MCH_FIX_2_CALIBRATION_REQ )
   END_RUNG
   // the same network as SCL:
   "DB7330_ETXETAR_ROBOT_CELL_INTERLOCK".INTERLOCKS_UNIT_01.MACHINE_TO_ROBOT.MCH_FIX_2_CALIBRATION_REQ := "DB16010_MEASURE_SENSORS_CALIBRATION_STATUS".U1_STA3_MEAS.FIXTURE_2_STATUS <> 1;
END_REGION

REGION Network 37: MACHINE FIXTURE 3 CALIBRATION REQUIRED
   RUNG wire#powerrail
      { S7_Templates := "SrcType := Int" } NE_Contact(in1 := "DB16010_MEASURE_SENSORS_CALIBRATION_STATUS".U1_STA3_MEAS.FIXTURE_3_STATUS, in2 := 1)
      Coil( "DB7330_ETXETAR_ROBOT_CELL_INTERLOCK".INTERLOCKS_UNIT_01.MACHINE_TO_ROBOT.MCH_FIX_3_CALIBRATION_REQ )
   END_RUNG
   // the same network as SCL:
   "DB7330_ETXETAR_ROBOT_CELL_INTERLOCK".INTERLOCKS_UNIT_01.MACHINE_TO_ROBOT.MCH_FIX_3_CALIBRATION_REQ := "DB16010_MEASURE_SENSORS_CALIBRATION_STATUS".U1_STA3_MEAS.FIXTURE_3_STATUS <> 1;
END_REGION

REGION Network 38: MACHINE FIXTURE 4 CALIBRATION REQUIRED
   RUNG wire#powerrail
      { S7_Templates := "SrcType := Int" } NE_Contact(in1 := "DB16010_MEASURE_SENSORS_CALIBRATION_STATUS".U1_STA3_MEAS.FIXTURE_4_STATUS, in2 := 1)
      Coil( "DB7330_ETXETAR_ROBOT_CELL_INTERLOCK".INTERLOCKS_UNIT_01.MACHINE_TO_ROBOT.MCH_FIX_4_CALIBRATION_REQ )
   END_RUNG
   // the same network as SCL:
   "DB7330_ETXETAR_ROBOT_CELL_INTERLOCK".INTERLOCKS_UNIT_01.MACHINE_TO_ROBOT.MCH_FIX_4_CALIBRATION_REQ := "DB16010_MEASURE_SENSORS_CALIBRATION_STATUS".U1_STA3_MEAS.FIXTURE_4_STATUS <> 1;
END_REGION

REGION Network 39: MACHINE CLEAR TO LOAD/UNLOAD
   RUNG wire#powerrail
      Contact( "DB1101_MACHINE_SEQUENCE".CLEAR_TO_LOAD_UNLOAD_UNIT_01 )
      Coil( "DB7330_ETXETAR_ROBOT_CELL_INTERLOCK".INTERLOCKS_UNIT_01.MACHINE_TO_ROBOT.CLEAR_LOAD_UNLOAD )
   END_RUNG
   // the same network as SCL:
   "DB7330_ETXETAR_ROBOT_CELL_INTERLOCK".INTERLOCKS_UNIT_01.MACHINE_TO_ROBOT.CLEAR_LOAD_UNLOAD := "DB1101_MACHINE_SEQUENCE".CLEAR_TO_LOAD_UNLOAD_UNIT_01;
END_REGION

REGION Network 40: MACHINE UNLOAD REQUEST FACE R
   RUNG wire#powerrail
      Contact( "DB1101_MACHINE_SEQUENCE".CLEAR_TO_LOAD_UNLOAD_UNIT_01 )
      Contact( "DB341_M_UNIT_1_STA_0".M_CODES_UNIT_1_STA_0.M51 )
      wire#w1
      Contact( "DB5000_FIX_TABLE_POSITIONS".UNIT_1.FIXTURE[1].IN_LOAD_UNLOAD_STATION_1 )
      wire#w2
      Contact( "DB2430_FULL_DEPTH".FD_UNIT_01.FIXTURE_1.FULL_DEPTH )
      Contact( "DB8000_PART_STATUS".UNIT_1.FIXTURE_1.PART_A.STATUS.OK )
      wire#w3
      Contact( "DB8000_PART_STATUS".UNIT_1.FIXTURE_1.PART_A.STATUS.PRESENT )
      wire#w4
      Coil( "DB7330_ETXETAR_ROBOT_CELL_INTERLOCK".INTERLOCKS_UNIT_01.MACHINE_TO_ROBOT.MCH_UNLOAD_REQUEST_FACE_R )
   END_RUNG
   RUNG wire#w2
      Contact( "DB2430_FULL_DEPTH".FD_UNIT_01.FIXTURE_1.PART_REJECTED_FIXTURE )
   END_RUNG wire#w3
   RUNG wire#w1
      Contact( "DB5000_FIX_TABLE_POSITIONS".UNIT_1.FIXTURE[3].IN_LOAD_UNLOAD_STATION_1 )
      wire#w5
      Contact( "DB2430_FULL_DEPTH".FD_UNIT_01.FIXTURE_3.FULL_DEPTH )
      Contact( "DB8000_PART_STATUS".UNIT_1.FIXTURE_3.PART_A.STATUS.OK )
      wire#w6
      Contact( "DB8000_PART_STATUS".UNIT_1.FIXTURE_3.PART_A.STATUS.PRESENT )
   END_RUNG wire#w4
   RUNG wire#w5
      Contact( "DB2430_FULL_DEPTH".FD_UNIT_01.FIXTURE_3.PART_REJECTED_FIXTURE )
   END_RUNG wire#w6
   // the same network as SCL:
   "DB7330_ETXETAR_ROBOT_CELL_INTERLOCK".INTERLOCKS_UNIT_01.MACHINE_TO_ROBOT.MCH_UNLOAD_REQUEST_FACE_R := "DB1101_MACHINE_SEQUENCE".CLEAR_TO_LOAD_UNLOAD_UNIT_01 AND "DB341_M_UNIT_1_STA_0".M_CODES_UNIT_1_STA_0.M51 AND (("DB5000_FIX_TABLE_POSITIONS".UNIT_1.FIXTURE[1].IN_LOAD_UNLOAD_STATION_1 AND (("DB2430_FULL_DEPTH".FD_UNIT_01.FIXTURE_1.FULL_DEPTH AND "DB8000_PART_STATUS".UNIT_1.FIXTURE_1.PART_A.STATUS.OK) OR "DB2430_FULL_DEPTH".FD_UNIT_01.FIXTURE_1.PART_REJECTED_FIXTURE) AND "DB8000_PART_STATUS".UNIT_1.FIXTURE_1.PART_A.STATUS.PRESENT) OR ("DB5000_FIX_TABLE_POSITIONS".UNIT_1.FIXTURE[3].IN_LOAD_UNLOAD_STATION_1 AND (("DB2430_FULL_DEPTH".FD_UNIT_01.FIXTURE_3.FULL_DEPTH AND "DB8000_PART_STATUS".UNIT_1.FIXTURE_3.PART_A.STATUS.OK) OR "DB2430_FULL_DEPTH".FD_UNIT_01.FIXTURE_3.PART_REJECTED_FIXTURE) AND "DB8000_PART_STATUS".UNIT_1.FIXTURE_3.PART_A.STATUS.PRESENT));
END_REGION

REGION Network 41: MACHINE UNLOAD REQUEST FACE N
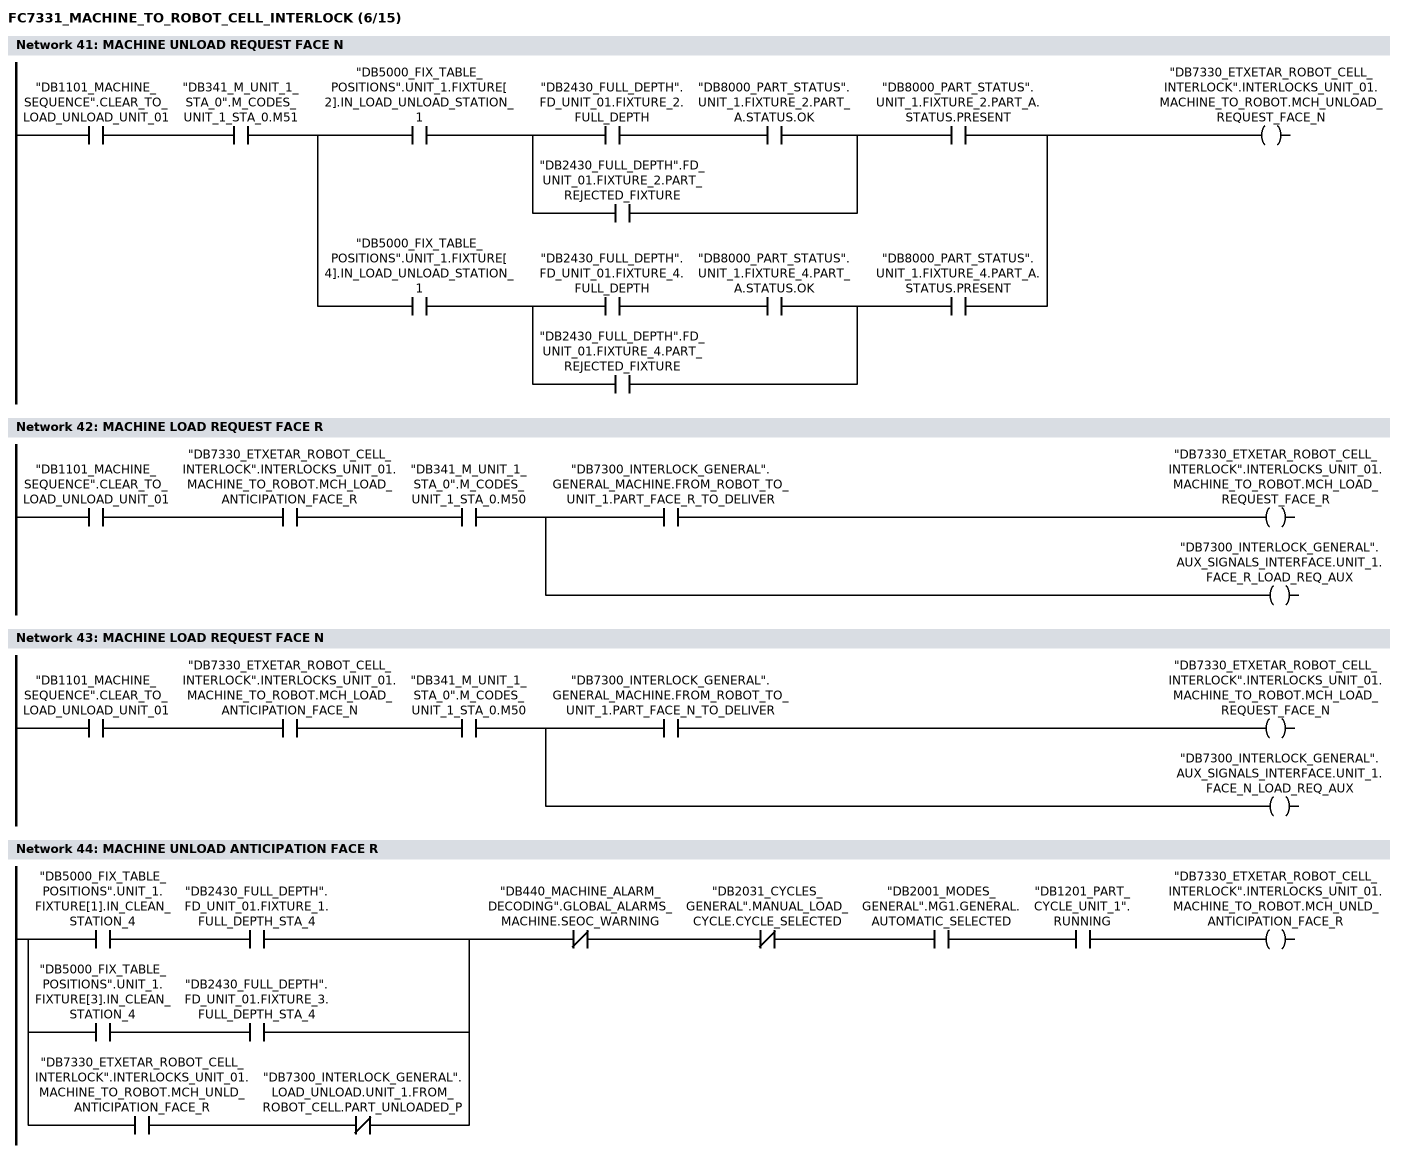
   RUNG wire#powerrail
      Contact( "DB1101_MACHINE_SEQUENCE".CLEAR_TO_LOAD_UNLOAD_UNIT_01 )
      Contact( "DB341_M_UNIT_1_STA_0".M_CODES_UNIT_1_STA_0.M51 )
      wire#w1
      Contact( "DB5000_FIX_TABLE_POSITIONS".UNIT_1.FIXTURE[2].IN_LOAD_UNLOAD_STATION_1 )
      wire#w2
      Contact( "DB2430_FULL_DEPTH".FD_UNIT_01.FIXTURE_2.FULL_DEPTH )
      Contact( "DB8000_PART_STATUS".UNIT_1.FIXTURE_2.PART_A.STATUS.OK )
      wire#w3
      Contact( "DB8000_PART_STATUS".UNIT_1.FIXTURE_2.PART_A.STATUS.PRESENT )
      wire#w4
      Coil( "DB7330_ETXETAR_ROBOT_CELL_INTERLOCK".INTERLOCKS_UNIT_01.MACHINE_TO_ROBOT.MCH_UNLOAD_REQUEST_FACE_N )
   END_RUNG
   RUNG wire#w2
      Contact( "DB2430_FULL_DEPTH".FD_UNIT_01.FIXTURE_2.PART_REJECTED_FIXTURE )
   END_RUNG wire#w3
   RUNG wire#w1
      Contact( "DB5000_FIX_TABLE_POSITIONS".UNIT_1.FIXTURE[4].IN_LOAD_UNLOAD_STATION_1 )
      wire#w5
      Contact( "DB2430_FULL_DEPTH".FD_UNIT_01.FIXTURE_4.FULL_DEPTH )
      Contact( "DB8000_PART_STATUS".UNIT_1.FIXTURE_4.PART_A.STATUS.OK )
      wire#w6
      Contact( "DB8000_PART_STATUS".UNIT_1.FIXTURE_4.PART_A.STATUS.PRESENT )
   END_RUNG wire#w4
   RUNG wire#w5
      Contact( "DB2430_FULL_DEPTH".FD_UNIT_01.FIXTURE_4.PART_REJECTED_FIXTURE )
   END_RUNG wire#w6
   // the same network as SCL:
   "DB7330_ETXETAR_ROBOT_CELL_INTERLOCK".INTERLOCKS_UNIT_01.MACHINE_TO_ROBOT.MCH_UNLOAD_REQUEST_FACE_N := "DB1101_MACHINE_SEQUENCE".CLEAR_TO_LOAD_UNLOAD_UNIT_01 AND "DB341_M_UNIT_1_STA_0".M_CODES_UNIT_1_STA_0.M51 AND (("DB5000_FIX_TABLE_POSITIONS".UNIT_1.FIXTURE[2].IN_LOAD_UNLOAD_STATION_1 AND (("DB2430_FULL_DEPTH".FD_UNIT_01.FIXTURE_2.FULL_DEPTH AND "DB8000_PART_STATUS".UNIT_1.FIXTURE_2.PART_A.STATUS.OK) OR "DB2430_FULL_DEPTH".FD_UNIT_01.FIXTURE_2.PART_REJECTED_FIXTURE) AND "DB8000_PART_STATUS".UNIT_1.FIXTURE_2.PART_A.STATUS.PRESENT) OR ("DB5000_FIX_TABLE_POSITIONS".UNIT_1.FIXTURE[4].IN_LOAD_UNLOAD_STATION_1 AND (("DB2430_FULL_DEPTH".FD_UNIT_01.FIXTURE_4.FULL_DEPTH AND "DB8000_PART_STATUS".UNIT_1.FIXTURE_4.PART_A.STATUS.OK) OR "DB2430_FULL_DEPTH".FD_UNIT_01.FIXTURE_4.PART_REJECTED_FIXTURE) AND "DB8000_PART_STATUS".UNIT_1.FIXTURE_4.PART_A.STATUS.PRESENT));
END_REGION

REGION Network 42: MACHINE LOAD REQUEST FACE R
   RUNG wire#powerrail
      Contact( "DB1101_MACHINE_SEQUENCE".CLEAR_TO_LOAD_UNLOAD_UNIT_01 )
      Contact( "DB7330_ETXETAR_ROBOT_CELL_INTERLOCK".INTERLOCKS_UNIT_01.MACHINE_TO_ROBOT.MCH_LOAD_ANTICIPATION_FACE_R )
      Contact( "DB341_M_UNIT_1_STA_0".M_CODES_UNIT_1_STA_0.M50 )
      wire#w1
      Contact( "DB7300_INTERLOCK_GENERAL".GENERAL_MACHINE.FROM_ROBOT_TO_UNIT_1.PART_FACE_R_TO_DELIVER )
      Coil( "DB7330_ETXETAR_ROBOT_CELL_INTERLOCK".INTERLOCKS_UNIT_01.MACHINE_TO_ROBOT.MCH_LOAD_REQUEST_FACE_R )
   END_RUNG
   RUNG wire#w1
      Coil( "DB7300_INTERLOCK_GENERAL".AUX_SIGNALS_INTERFACE.UNIT_1.FACE_R_LOAD_REQ_AUX )
   END_RUNG
   // the same network as SCL:
   #_w1 := "DB1101_MACHINE_SEQUENCE".CLEAR_TO_LOAD_UNLOAD_UNIT_01 AND "DB7330_ETXETAR_ROBOT_CELL_INTERLOCK".INTERLOCKS_UNIT_01.MACHINE_TO_ROBOT.MCH_LOAD_ANTICIPATION_FACE_R AND "DB341_M_UNIT_1_STA_0".M_CODES_UNIT_1_STA_0.M50;
   "DB7330_ETXETAR_ROBOT_CELL_INTERLOCK".INTERLOCKS_UNIT_01.MACHINE_TO_ROBOT.MCH_LOAD_REQUEST_FACE_R := #_w1 AND "DB7300_INTERLOCK_GENERAL".GENERAL_MACHINE.FROM_ROBOT_TO_UNIT_1.PART_FACE_R_TO_DELIVER;
   "DB7300_INTERLOCK_GENERAL".AUX_SIGNALS_INTERFACE.UNIT_1.FACE_R_LOAD_REQ_AUX := #_w1;
END_REGION

REGION Network 43: MACHINE LOAD REQUEST FACE N
   RUNG wire#powerrail
      Contact( "DB1101_MACHINE_SEQUENCE".CLEAR_TO_LOAD_UNLOAD_UNIT_01 )
      Contact( "DB7330_ETXETAR_ROBOT_CELL_INTERLOCK".INTERLOCKS_UNIT_01.MACHINE_TO_ROBOT.MCH_LOAD_ANTICIPATION_FACE_N )
      Contact( "DB341_M_UNIT_1_STA_0".M_CODES_UNIT_1_STA_0.M50 )
      wire#w1
      Contact( "DB7300_INTERLOCK_GENERAL".GENERAL_MACHINE.FROM_ROBOT_TO_UNIT_1.PART_FACE_N_TO_DELIVER )
      Coil( "DB7330_ETXETAR_ROBOT_CELL_INTERLOCK".INTERLOCKS_UNIT_01.MACHINE_TO_ROBOT.MCH_LOAD_REQUEST_FACE_N )
   END_RUNG
   RUNG wire#w1
      Coil( "DB7300_INTERLOCK_GENERAL".AUX_SIGNALS_INTERFACE.UNIT_1.FACE_N_LOAD_REQ_AUX )
   END_RUNG
   // the same network as SCL:
   #_w1 := "DB1101_MACHINE_SEQUENCE".CLEAR_TO_LOAD_UNLOAD_UNIT_01 AND "DB7330_ETXETAR_ROBOT_CELL_INTERLOCK".INTERLOCKS_UNIT_01.MACHINE_TO_ROBOT.MCH_LOAD_ANTICIPATION_FACE_N AND "DB341_M_UNIT_1_STA_0".M_CODES_UNIT_1_STA_0.M50;
   "DB7330_ETXETAR_ROBOT_CELL_INTERLOCK".INTERLOCKS_UNIT_01.MACHINE_TO_ROBOT.MCH_LOAD_REQUEST_FACE_N := #_w1 AND "DB7300_INTERLOCK_GENERAL".GENERAL_MACHINE.FROM_ROBOT_TO_UNIT_1.PART_FACE_N_TO_DELIVER;
   "DB7300_INTERLOCK_GENERAL".AUX_SIGNALS_INTERFACE.UNIT_1.FACE_N_LOAD_REQ_AUX := #_w1;
END_REGION

REGION Network 44: MACHINE UNLOAD ANTICIPATION FACE R
   RUNG wire#powerrail
      Contact( "DB5000_FIX_TABLE_POSITIONS".UNIT_1.FIXTURE[1].IN_CLEAN_STATION_4 )
      Contact( "DB2430_FULL_DEPTH".FD_UNIT_01.FIXTURE_1.FULL_DEPTH_STA_4 )
      wire#w1
      I_Contact( "DB440_MACHINE_ALARM_DECODING".GLOBAL_ALARMS_MACHINE.SEOC_WARNING )
      I_Contact( "DB2031_CYCLES_GENERAL".MANUAL_LOAD_CYCLE.CYCLE_SELECTED )
      Contact( "DB2001_MODES_GENERAL".MG1.GENERAL.AUTOMATIC_SELECTED )
      Contact( "DB1201_PART_CYCLE_UNIT_1".RUNNING )
      Coil( "DB7330_ETXETAR_ROBOT_CELL_INTERLOCK".INTERLOCKS_UNIT_01.MACHINE_TO_ROBOT.MCH_UNLD_ANTICIPATION_FACE_R )
   END_RUNG
   RUNG wire#powerrail
      Contact( "DB5000_FIX_TABLE_POSITIONS".UNIT_1.FIXTURE[3].IN_CLEAN_STATION_4 )
      Contact( "DB2430_FULL_DEPTH".FD_UNIT_01.FIXTURE_3.FULL_DEPTH_STA_4 )
   END_RUNG wire#w1
   RUNG wire#powerrail
      Contact( "DB7330_ETXETAR_ROBOT_CELL_INTERLOCK".INTERLOCKS_UNIT_01.MACHINE_TO_ROBOT.MCH_UNLD_ANTICIPATION_FACE_R )
      I_Contact( "DB7300_INTERLOCK_GENERAL".LOAD_UNLOAD.UNIT_1.FROM_ROBOT_CELL.PART_UNLOADED_P )
   END_RUNG wire#w1
   // the same network as SCL:
   "DB7330_ETXETAR_ROBOT_CELL_INTERLOCK".INTERLOCKS_UNIT_01.MACHINE_TO_ROBOT.MCH_UNLD_ANTICIPATION_FACE_R := (("DB5000_FIX_TABLE_POSITIONS".UNIT_1.FIXTURE[1].IN_CLEAN_STATION_4 AND "DB2430_FULL_DEPTH".FD_UNIT_01.FIXTURE_1.FULL_DEPTH_STA_4) OR ("DB5000_FIX_TABLE_POSITIONS".UNIT_1.FIXTURE[3].IN_CLEAN_STATION_4 AND "DB2430_FULL_DEPTH".FD_UNIT_01.FIXTURE_3.FULL_DEPTH_STA_4) OR ("DB7330_ETXETAR_ROBOT_CELL_INTERLOCK".INTERLOCKS_UNIT_01.MACHINE_TO_ROBOT.MCH_UNLD_ANTICIPATION_FACE_R AND NOT "DB7300_INTERLOCK_GENERAL".LOAD_UNLOAD.UNIT_1.FROM_ROBOT_CELL.PART_UNLOADED_P)) AND NOT "DB440_MACHINE_ALARM_DECODING".GLOBAL_ALARMS_MACHINE.SEOC_WARNING AND NOT "DB2031_CYCLES_GENERAL".MANUAL_LOAD_CYCLE.CYCLE_SELECTED AND "DB2001_MODES_GENERAL".MG1.GENERAL.AUTOMATIC_SELECTED AND "DB1201_PART_CYCLE_UNIT_1".RUNNING;
END_REGION

REGION Network 45: MACHINE UNLOAD ANTICIPATION FACE N
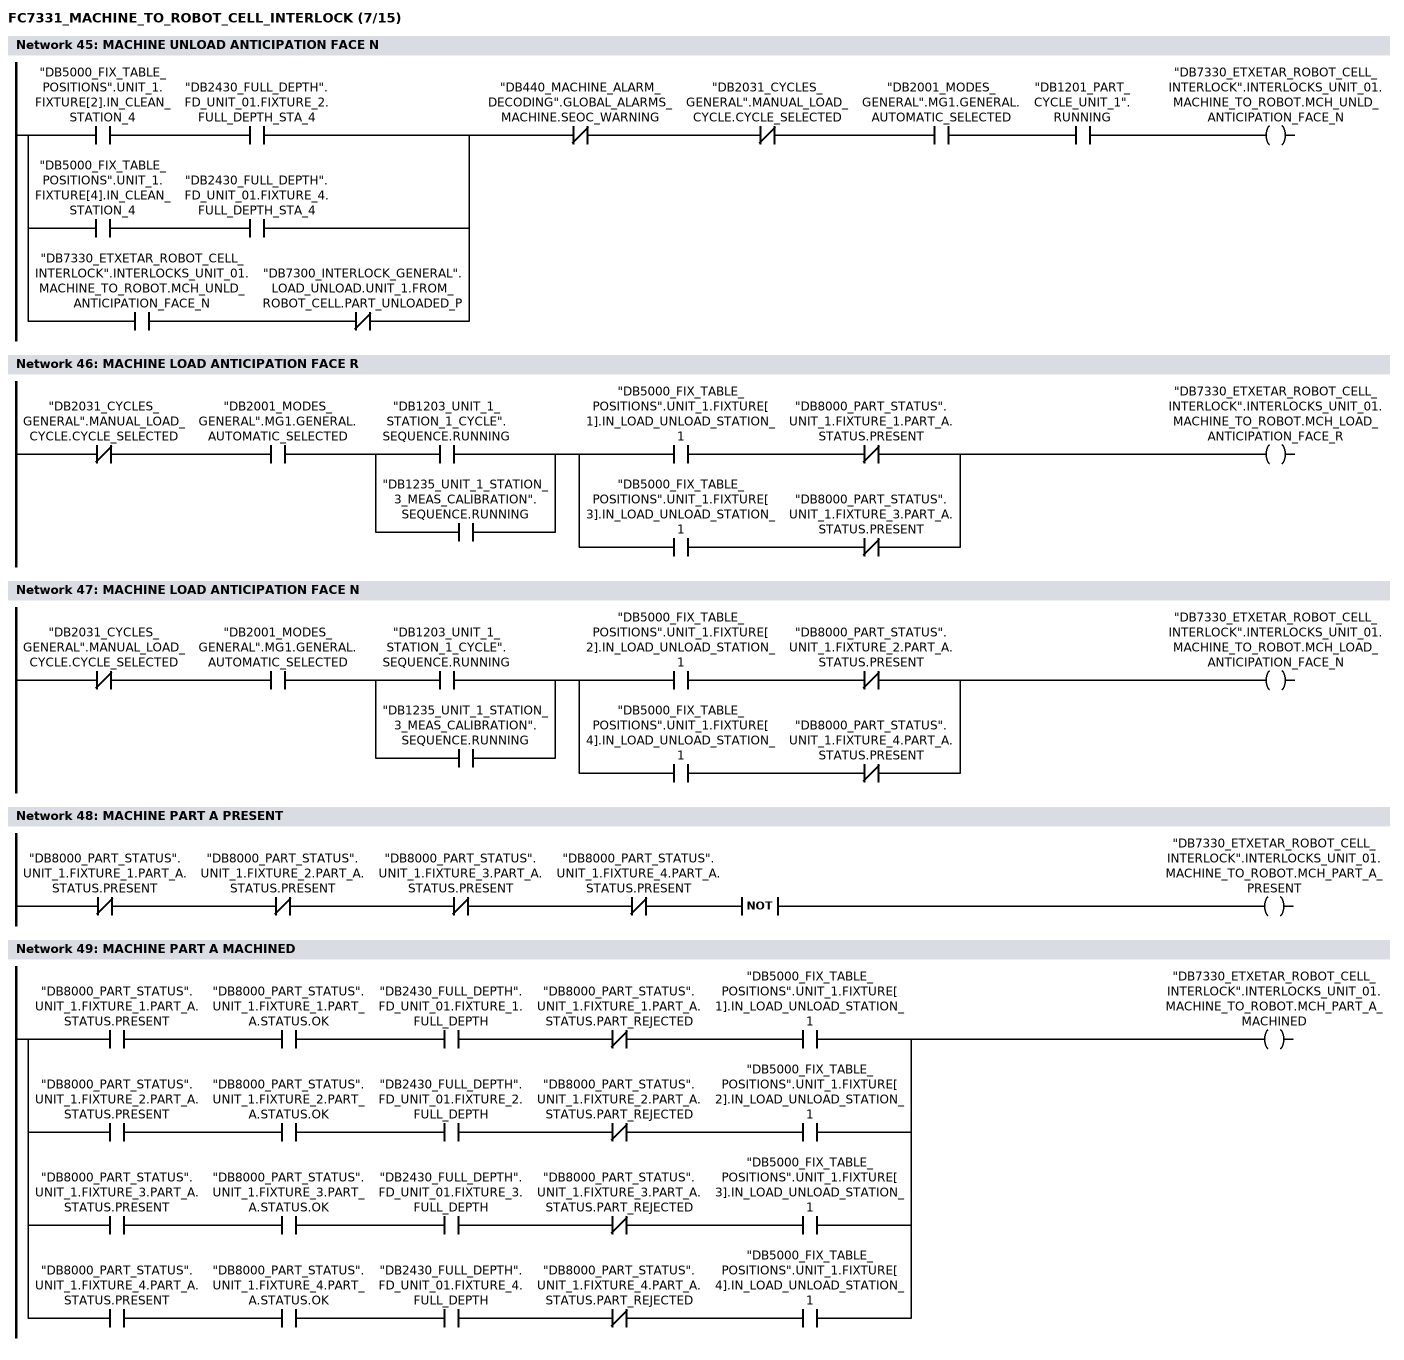
   RUNG wire#powerrail
      Contact( "DB5000_FIX_TABLE_POSITIONS".UNIT_1.FIXTURE[2].IN_CLEAN_STATION_4 )
      Contact( "DB2430_FULL_DEPTH".FD_UNIT_01.FIXTURE_2.FULL_DEPTH_STA_4 )
      wire#w1
      I_Contact( "DB440_MACHINE_ALARM_DECODING".GLOBAL_ALARMS_MACHINE.SEOC_WARNING )
      I_Contact( "DB2031_CYCLES_GENERAL".MANUAL_LOAD_CYCLE.CYCLE_SELECTED )
      Contact( "DB2001_MODES_GENERAL".MG1.GENERAL.AUTOMATIC_SELECTED )
      Contact( "DB1201_PART_CYCLE_UNIT_1".RUNNING )
      Coil( "DB7330_ETXETAR_ROBOT_CELL_INTERLOCK".INTERLOCKS_UNIT_01.MACHINE_TO_ROBOT.MCH_UNLD_ANTICIPATION_FACE_N )
   END_RUNG
   RUNG wire#powerrail
      Contact( "DB5000_FIX_TABLE_POSITIONS".UNIT_1.FIXTURE[4].IN_CLEAN_STATION_4 )
      Contact( "DB2430_FULL_DEPTH".FD_UNIT_01.FIXTURE_4.FULL_DEPTH_STA_4 )
   END_RUNG wire#w1
   RUNG wire#powerrail
      Contact( "DB7330_ETXETAR_ROBOT_CELL_INTERLOCK".INTERLOCKS_UNIT_01.MACHINE_TO_ROBOT.MCH_UNLD_ANTICIPATION_FACE_N )
      I_Contact( "DB7300_INTERLOCK_GENERAL".LOAD_UNLOAD.UNIT_1.FROM_ROBOT_CELL.PART_UNLOADED_P )
   END_RUNG wire#w1
   // the same network as SCL:
   "DB7330_ETXETAR_ROBOT_CELL_INTERLOCK".INTERLOCKS_UNIT_01.MACHINE_TO_ROBOT.MCH_UNLD_ANTICIPATION_FACE_N := (("DB5000_FIX_TABLE_POSITIONS".UNIT_1.FIXTURE[2].IN_CLEAN_STATION_4 AND "DB2430_FULL_DEPTH".FD_UNIT_01.FIXTURE_2.FULL_DEPTH_STA_4) OR ("DB5000_FIX_TABLE_POSITIONS".UNIT_1.FIXTURE[4].IN_CLEAN_STATION_4 AND "DB2430_FULL_DEPTH".FD_UNIT_01.FIXTURE_4.FULL_DEPTH_STA_4) OR ("DB7330_ETXETAR_ROBOT_CELL_INTERLOCK".INTERLOCKS_UNIT_01.MACHINE_TO_ROBOT.MCH_UNLD_ANTICIPATION_FACE_N AND NOT "DB7300_INTERLOCK_GENERAL".LOAD_UNLOAD.UNIT_1.FROM_ROBOT_CELL.PART_UNLOADED_P)) AND NOT "DB440_MACHINE_ALARM_DECODING".GLOBAL_ALARMS_MACHINE.SEOC_WARNING AND NOT "DB2031_CYCLES_GENERAL".MANUAL_LOAD_CYCLE.CYCLE_SELECTED AND "DB2001_MODES_GENERAL".MG1.GENERAL.AUTOMATIC_SELECTED AND "DB1201_PART_CYCLE_UNIT_1".RUNNING;
END_REGION

REGION Network 46: MACHINE LOAD ANTICIPATION FACE R
   RUNG wire#powerrail
      I_Contact( "DB2031_CYCLES_GENERAL".MANUAL_LOAD_CYCLE.CYCLE_SELECTED )
      Contact( "DB2001_MODES_GENERAL".MG1.GENERAL.AUTOMATIC_SELECTED )
      wire#w1
      Contact( "DB1203_UNIT_1_STATION_1_CYCLE".SEQUENCE.RUNNING )
      wire#w2
      Contact( "DB5000_FIX_TABLE_POSITIONS".UNIT_1.FIXTURE[1].IN_LOAD_UNLOAD_STATION_1 )
      I_Contact( "DB8000_PART_STATUS".UNIT_1.FIXTURE_1.PART_A.STATUS.PRESENT )
      wire#w3
      Coil( "DB7330_ETXETAR_ROBOT_CELL_INTERLOCK".INTERLOCKS_UNIT_01.MACHINE_TO_ROBOT.MCH_LOAD_ANTICIPATION_FACE_R )
   END_RUNG
   RUNG wire#w1
      Contact( "DB1235_UNIT_1_STATION_3_MEAS_CALIBRATION".SEQUENCE.RUNNING )
   END_RUNG wire#w2
   RUNG wire#w2
      Contact( "DB5000_FIX_TABLE_POSITIONS".UNIT_1.FIXTURE[3].IN_LOAD_UNLOAD_STATION_1 )
      I_Contact( "DB8000_PART_STATUS".UNIT_1.FIXTURE_3.PART_A.STATUS.PRESENT )
   END_RUNG wire#w3
   // the same network as SCL:
   "DB7330_ETXETAR_ROBOT_CELL_INTERLOCK".INTERLOCKS_UNIT_01.MACHINE_TO_ROBOT.MCH_LOAD_ANTICIPATION_FACE_R := NOT "DB2031_CYCLES_GENERAL".MANUAL_LOAD_CYCLE.CYCLE_SELECTED AND "DB2001_MODES_GENERAL".MG1.GENERAL.AUTOMATIC_SELECTED AND ("DB1203_UNIT_1_STATION_1_CYCLE".SEQUENCE.RUNNING OR "DB1235_UNIT_1_STATION_3_MEAS_CALIBRATION".SEQUENCE.RUNNING) AND (("DB5000_FIX_TABLE_POSITIONS".UNIT_1.FIXTURE[1].IN_LOAD_UNLOAD_STATION_1 AND NOT "DB8000_PART_STATUS".UNIT_1.FIXTURE_1.PART_A.STATUS.PRESENT) OR ("DB5000_FIX_TABLE_POSITIONS".UNIT_1.FIXTURE[3].IN_LOAD_UNLOAD_STATION_1 AND NOT "DB8000_PART_STATUS".UNIT_1.FIXTURE_3.PART_A.STATUS.PRESENT));
END_REGION

REGION Network 47: MACHINE LOAD ANTICIPATION FACE N
   RUNG wire#powerrail
      I_Contact( "DB2031_CYCLES_GENERAL".MANUAL_LOAD_CYCLE.CYCLE_SELECTED )
      Contact( "DB2001_MODES_GENERAL".MG1.GENERAL.AUTOMATIC_SELECTED )
      wire#w1
      Contact( "DB1203_UNIT_1_STATION_1_CYCLE".SEQUENCE.RUNNING )
      wire#w2
      Contact( "DB5000_FIX_TABLE_POSITIONS".UNIT_1.FIXTURE[2].IN_LOAD_UNLOAD_STATION_1 )
      I_Contact( "DB8000_PART_STATUS".UNIT_1.FIXTURE_2.PART_A.STATUS.PRESENT )
      wire#w3
      Coil( "DB7330_ETXETAR_ROBOT_CELL_INTERLOCK".INTERLOCKS_UNIT_01.MACHINE_TO_ROBOT.MCH_LOAD_ANTICIPATION_FACE_N )
   END_RUNG
   RUNG wire#w1
      Contact( "DB1235_UNIT_1_STATION_3_MEAS_CALIBRATION".SEQUENCE.RUNNING )
   END_RUNG wire#w2
   RUNG wire#w2
      Contact( "DB5000_FIX_TABLE_POSITIONS".UNIT_1.FIXTURE[4].IN_LOAD_UNLOAD_STATION_1 )
      I_Contact( "DB8000_PART_STATUS".UNIT_1.FIXTURE_4.PART_A.STATUS.PRESENT )
   END_RUNG wire#w3
   // the same network as SCL:
   "DB7330_ETXETAR_ROBOT_CELL_INTERLOCK".INTERLOCKS_UNIT_01.MACHINE_TO_ROBOT.MCH_LOAD_ANTICIPATION_FACE_N := NOT "DB2031_CYCLES_GENERAL".MANUAL_LOAD_CYCLE.CYCLE_SELECTED AND "DB2001_MODES_GENERAL".MG1.GENERAL.AUTOMATIC_SELECTED AND ("DB1203_UNIT_1_STATION_1_CYCLE".SEQUENCE.RUNNING OR "DB1235_UNIT_1_STATION_3_MEAS_CALIBRATION".SEQUENCE.RUNNING) AND (("DB5000_FIX_TABLE_POSITIONS".UNIT_1.FIXTURE[2].IN_LOAD_UNLOAD_STATION_1 AND NOT "DB8000_PART_STATUS".UNIT_1.FIXTURE_2.PART_A.STATUS.PRESENT) OR ("DB5000_FIX_TABLE_POSITIONS".UNIT_1.FIXTURE[4].IN_LOAD_UNLOAD_STATION_1 AND NOT "DB8000_PART_STATUS".UNIT_1.FIXTURE_4.PART_A.STATUS.PRESENT));
END_REGION

REGION Network 48: MACHINE PART A PRESENT
   RUNG wire#powerrail
      I_Contact( "DB8000_PART_STATUS".UNIT_1.FIXTURE_1.PART_A.STATUS.PRESENT )
      I_Contact( "DB8000_PART_STATUS".UNIT_1.FIXTURE_2.PART_A.STATUS.PRESENT )
      I_Contact( "DB8000_PART_STATUS".UNIT_1.FIXTURE_3.PART_A.STATUS.PRESENT )
      I_Contact( "DB8000_PART_STATUS".UNIT_1.FIXTURE_4.PART_A.STATUS.PRESENT )
      Not()
      Coil( "DB7330_ETXETAR_ROBOT_CELL_INTERLOCK".INTERLOCKS_UNIT_01.MACHINE_TO_ROBOT.MCH_PART_A_PRESENT )
   END_RUNG
   // the same network as SCL:
   "DB7330_ETXETAR_ROBOT_CELL_INTERLOCK".INTERLOCKS_UNIT_01.MACHINE_TO_ROBOT.MCH_PART_A_PRESENT := NOT (NOT "DB8000_PART_STATUS".UNIT_1.FIXTURE_1.PART_A.STATUS.PRESENT AND NOT "DB8000_PART_STATUS".UNIT_1.FIXTURE_2.PART_A.STATUS.PRESENT AND NOT "DB8000_PART_STATUS".UNIT_1.FIXTURE_3.PART_A.STATUS.PRESENT AND NOT "DB8000_PART_STATUS".UNIT_1.FIXTURE_4.PART_A.STATUS.PRESENT);
END_REGION

REGION Network 49: MACHINE PART A MACHINED
   RUNG wire#powerrail
      Contact( "DB8000_PART_STATUS".UNIT_1.FIXTURE_1.PART_A.STATUS.PRESENT )
      Contact( "DB8000_PART_STATUS".UNIT_1.FIXTURE_1.PART_A.STATUS.OK )
      Contact( "DB2430_FULL_DEPTH".FD_UNIT_01.FIXTURE_1.FULL_DEPTH )
      I_Contact( "DB8000_PART_STATUS".UNIT_1.FIXTURE_1.PART_A.STATUS.PART_REJECTED )
      Contact( "DB5000_FIX_TABLE_POSITIONS".UNIT_1.FIXTURE[1].IN_LOAD_UNLOAD_STATION_1 )
      wire#w1
      Coil( "DB7330_ETXETAR_ROBOT_CELL_INTERLOCK".INTERLOCKS_UNIT_01.MACHINE_TO_ROBOT.MCH_PART_A_MACHINED )
   END_RUNG
   RUNG wire#powerrail
      Contact( "DB8000_PART_STATUS".UNIT_1.FIXTURE_2.PART_A.STATUS.PRESENT )
      Contact( "DB8000_PART_STATUS".UNIT_1.FIXTURE_2.PART_A.STATUS.OK )
      Contact( "DB2430_FULL_DEPTH".FD_UNIT_01.FIXTURE_2.FULL_DEPTH )
      I_Contact( "DB8000_PART_STATUS".UNIT_1.FIXTURE_2.PART_A.STATUS.PART_REJECTED )
      Contact( "DB5000_FIX_TABLE_POSITIONS".UNIT_1.FIXTURE[2].IN_LOAD_UNLOAD_STATION_1 )
   END_RUNG wire#w1
   RUNG wire#powerrail
      Contact( "DB8000_PART_STATUS".UNIT_1.FIXTURE_3.PART_A.STATUS.PRESENT )
      Contact( "DB8000_PART_STATUS".UNIT_1.FIXTURE_3.PART_A.STATUS.OK )
      Contact( "DB2430_FULL_DEPTH".FD_UNIT_01.FIXTURE_3.FULL_DEPTH )
      I_Contact( "DB8000_PART_STATUS".UNIT_1.FIXTURE_3.PART_A.STATUS.PART_REJECTED )
      Contact( "DB5000_FIX_TABLE_POSITIONS".UNIT_1.FIXTURE[3].IN_LOAD_UNLOAD_STATION_1 )
   END_RUNG wire#w1
   RUNG wire#powerrail
      Contact( "DB8000_PART_STATUS".UNIT_1.FIXTURE_4.PART_A.STATUS.PRESENT )
      Contact( "DB8000_PART_STATUS".UNIT_1.FIXTURE_4.PART_A.STATUS.OK )
      Contact( "DB2430_FULL_DEPTH".FD_UNIT_01.FIXTURE_4.FULL_DEPTH )
      I_Contact( "DB8000_PART_STATUS".UNIT_1.FIXTURE_4.PART_A.STATUS.PART_REJECTED )
      Contact( "DB5000_FIX_TABLE_POSITIONS".UNIT_1.FIXTURE[4].IN_LOAD_UNLOAD_STATION_1 )
   END_RUNG wire#w1
   // the same network as SCL:
   "DB7330_ETXETAR_ROBOT_CELL_INTERLOCK".INTERLOCKS_UNIT_01.MACHINE_TO_ROBOT.MCH_PART_A_MACHINED := ("DB8000_PART_STATUS".UNIT_1.FIXTURE_1.PART_A.STATUS.PRESENT AND "DB8000_PART_STATUS".UNIT_1.FIXTURE_1.PART_A.STATUS.OK AND "DB2430_FULL_DEPTH".FD_UNIT_01.FIXTURE_1.FULL_DEPTH AND NOT "DB8000_PART_STATUS".UNIT_1.FIXTURE_1.PART_A.STATUS.PART_REJECTED AND "DB5000_FIX_TABLE_POSITIONS".UNIT_1.FIXTURE[1].IN_LOAD_UNLOAD_STATION_1) OR ("DB8000_PART_STATUS".UNIT_1.FIXTURE_2.PART_A.STATUS.PRESENT AND "DB8000_PART_STATUS".UNIT_1.FIXTURE_2.PART_A.STATUS.OK AND "DB2430_FULL_DEPTH".FD_UNIT_01.FIXTURE_2.FULL_DEPTH AND NOT "DB8000_PART_STATUS".UNIT_1.FIXTURE_2.PART_A.STATUS.PART_REJECTED AND "DB5000_FIX_TABLE_POSITIONS".UNIT_1.FIXTURE[2].IN_LOAD_UNLOAD_STATION_1) OR ("DB8000_PART_STATUS".UNIT_1.FIXTURE_3.PART_A.STATUS.PRESENT AND "DB8000_PART_STATUS".UNIT_1.FIXTURE_3.PART_A.STATUS.OK AND "DB2430_FULL_DEPTH".FD_UNIT_01.FIXTURE_3.FULL_DEPTH AND NOT "DB8000_PART_STATUS".UNIT_1.FIXTURE_3.PART_A.STATUS.PART_REJECTED AND "DB5000_FIX_TABLE_POSITIONS".UNIT_1.FIXTURE[3].IN_LOAD_UNLOAD_STATION_1) OR ("DB8000_PART_STATUS".UNIT_1.FIXTURE_4.PART_A.STATUS.PRESENT AND "DB8000_PART_STATUS".UNIT_1.FIXTURE_4.PART_A.STATUS.OK AND "DB2430_FULL_DEPTH".FD_UNIT_01.FIXTURE_4.FULL_DEPTH AND NOT "DB8000_PART_STATUS".UNIT_1.FIXTURE_4.PART_A.STATUS.PART_REJECTED AND "DB5000_FIX_TABLE_POSITIONS".UNIT_1.FIXTURE[4].IN_LOAD_UNLOAD_STATION_1);
END_REGION

REGION Network 50: MACHINE PART A REJECTED
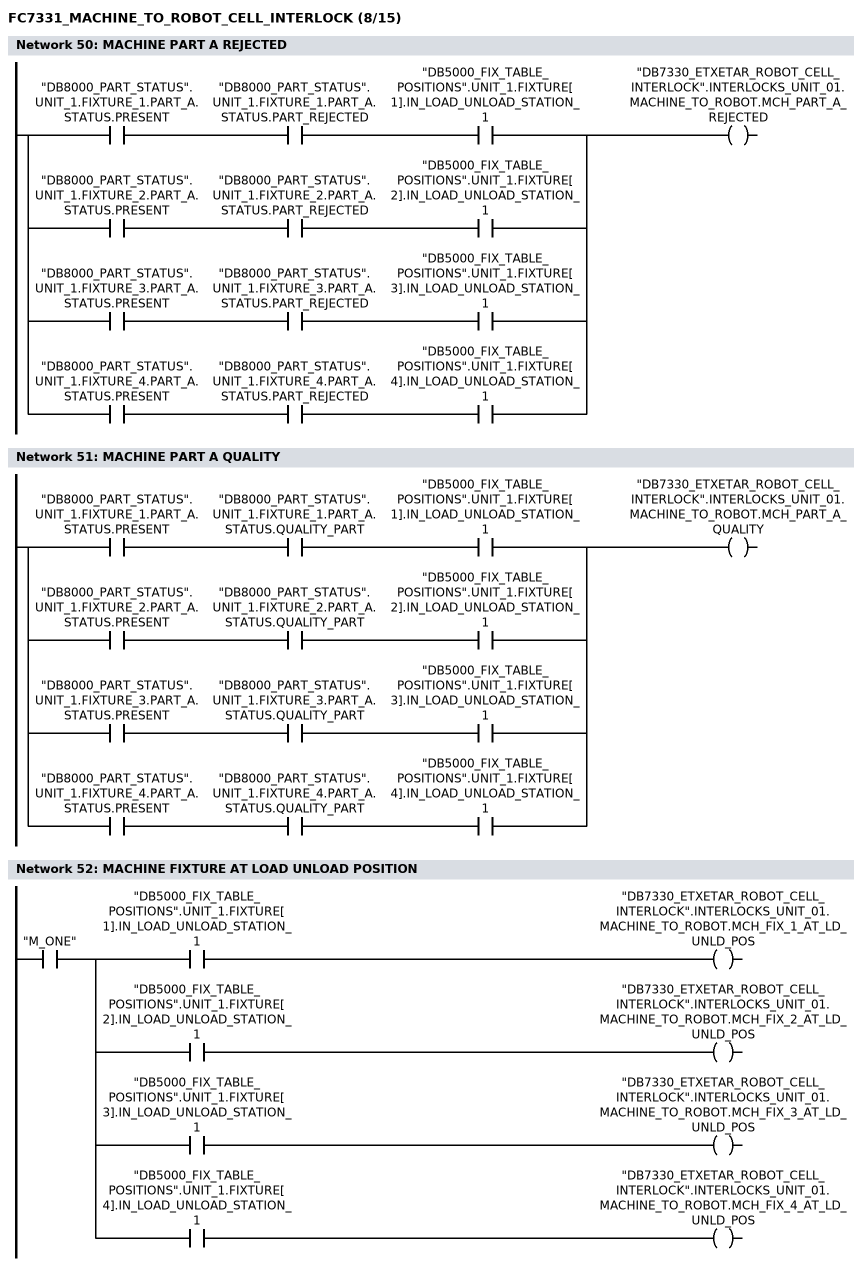
   RUNG wire#powerrail
      Contact( "DB8000_PART_STATUS".UNIT_1.FIXTURE_1.PART_A.STATUS.PRESENT )
      Contact( "DB8000_PART_STATUS".UNIT_1.FIXTURE_1.PART_A.STATUS.PART_REJECTED )
      Contact( "DB5000_FIX_TABLE_POSITIONS".UNIT_1.FIXTURE[1].IN_LOAD_UNLOAD_STATION_1 )
      wire#w1
      Coil( "DB7330_ETXETAR_ROBOT_CELL_INTERLOCK".INTERLOCKS_UNIT_01.MACHINE_TO_ROBOT.MCH_PART_A_REJECTED )
   END_RUNG
   RUNG wire#powerrail
      Contact( "DB8000_PART_STATUS".UNIT_1.FIXTURE_2.PART_A.STATUS.PRESENT )
      Contact( "DB8000_PART_STATUS".UNIT_1.FIXTURE_2.PART_A.STATUS.PART_REJECTED )
      Contact( "DB5000_FIX_TABLE_POSITIONS".UNIT_1.FIXTURE[2].IN_LOAD_UNLOAD_STATION_1 )
   END_RUNG wire#w1
   RUNG wire#powerrail
      Contact( "DB8000_PART_STATUS".UNIT_1.FIXTURE_3.PART_A.STATUS.PRESENT )
      Contact( "DB8000_PART_STATUS".UNIT_1.FIXTURE_3.PART_A.STATUS.PART_REJECTED )
      Contact( "DB5000_FIX_TABLE_POSITIONS".UNIT_1.FIXTURE[3].IN_LOAD_UNLOAD_STATION_1 )
   END_RUNG wire#w1
   RUNG wire#powerrail
      Contact( "DB8000_PART_STATUS".UNIT_1.FIXTURE_4.PART_A.STATUS.PRESENT )
      Contact( "DB8000_PART_STATUS".UNIT_1.FIXTURE_4.PART_A.STATUS.PART_REJECTED )
      Contact( "DB5000_FIX_TABLE_POSITIONS".UNIT_1.FIXTURE[4].IN_LOAD_UNLOAD_STATION_1 )
   END_RUNG wire#w1
   // the same network as SCL:
   "DB7330_ETXETAR_ROBOT_CELL_INTERLOCK".INTERLOCKS_UNIT_01.MACHINE_TO_ROBOT.MCH_PART_A_REJECTED := ("DB8000_PART_STATUS".UNIT_1.FIXTURE_1.PART_A.STATUS.PRESENT AND "DB8000_PART_STATUS".UNIT_1.FIXTURE_1.PART_A.STATUS.PART_REJECTED AND "DB5000_FIX_TABLE_POSITIONS".UNIT_1.FIXTURE[1].IN_LOAD_UNLOAD_STATION_1) OR ("DB8000_PART_STATUS".UNIT_1.FIXTURE_2.PART_A.STATUS.PRESENT AND "DB8000_PART_STATUS".UNIT_1.FIXTURE_2.PART_A.STATUS.PART_REJECTED AND "DB5000_FIX_TABLE_POSITIONS".UNIT_1.FIXTURE[2].IN_LOAD_UNLOAD_STATION_1) OR ("DB8000_PART_STATUS".UNIT_1.FIXTURE_3.PART_A.STATUS.PRESENT AND "DB8000_PART_STATUS".UNIT_1.FIXTURE_3.PART_A.STATUS.PART_REJECTED AND "DB5000_FIX_TABLE_POSITIONS".UNIT_1.FIXTURE[3].IN_LOAD_UNLOAD_STATION_1) OR ("DB8000_PART_STATUS".UNIT_1.FIXTURE_4.PART_A.STATUS.PRESENT AND "DB8000_PART_STATUS".UNIT_1.FIXTURE_4.PART_A.STATUS.PART_REJECTED AND "DB5000_FIX_TABLE_POSITIONS".UNIT_1.FIXTURE[4].IN_LOAD_UNLOAD_STATION_1);
END_REGION

REGION Network 51: MACHINE PART A QUALITY
   RUNG wire#powerrail
      Contact( "DB8000_PART_STATUS".UNIT_1.FIXTURE_1.PART_A.STATUS.PRESENT )
      Contact( "DB8000_PART_STATUS".UNIT_1.FIXTURE_1.PART_A.STATUS.QUALITY_PART )
      Contact( "DB5000_FIX_TABLE_POSITIONS".UNIT_1.FIXTURE[1].IN_LOAD_UNLOAD_STATION_1 )
      wire#w1
      Coil( "DB7330_ETXETAR_ROBOT_CELL_INTERLOCK".INTERLOCKS_UNIT_01.MACHINE_TO_ROBOT.MCH_PART_A_QUALITY )
   END_RUNG
   RUNG wire#powerrail
      Contact( "DB8000_PART_STATUS".UNIT_1.FIXTURE_2.PART_A.STATUS.PRESENT )
      Contact( "DB8000_PART_STATUS".UNIT_1.FIXTURE_2.PART_A.STATUS.QUALITY_PART )
      Contact( "DB5000_FIX_TABLE_POSITIONS".UNIT_1.FIXTURE[2].IN_LOAD_UNLOAD_STATION_1 )
   END_RUNG wire#w1
   RUNG wire#powerrail
      Contact( "DB8000_PART_STATUS".UNIT_1.FIXTURE_3.PART_A.STATUS.PRESENT )
      Contact( "DB8000_PART_STATUS".UNIT_1.FIXTURE_3.PART_A.STATUS.QUALITY_PART )
      Contact( "DB5000_FIX_TABLE_POSITIONS".UNIT_1.FIXTURE[3].IN_LOAD_UNLOAD_STATION_1 )
   END_RUNG wire#w1
   RUNG wire#powerrail
      Contact( "DB8000_PART_STATUS".UNIT_1.FIXTURE_4.PART_A.STATUS.PRESENT )
      Contact( "DB8000_PART_STATUS".UNIT_1.FIXTURE_4.PART_A.STATUS.QUALITY_PART )
      Contact( "DB5000_FIX_TABLE_POSITIONS".UNIT_1.FIXTURE[4].IN_LOAD_UNLOAD_STATION_1 )
   END_RUNG wire#w1
   // the same network as SCL:
   "DB7330_ETXETAR_ROBOT_CELL_INTERLOCK".INTERLOCKS_UNIT_01.MACHINE_TO_ROBOT.MCH_PART_A_QUALITY := ("DB8000_PART_STATUS".UNIT_1.FIXTURE_1.PART_A.STATUS.PRESENT AND "DB8000_PART_STATUS".UNIT_1.FIXTURE_1.PART_A.STATUS.QUALITY_PART AND "DB5000_FIX_TABLE_POSITIONS".UNIT_1.FIXTURE[1].IN_LOAD_UNLOAD_STATION_1) OR ("DB8000_PART_STATUS".UNIT_1.FIXTURE_2.PART_A.STATUS.PRESENT AND "DB8000_PART_STATUS".UNIT_1.FIXTURE_2.PART_A.STATUS.QUALITY_PART AND "DB5000_FIX_TABLE_POSITIONS".UNIT_1.FIXTURE[2].IN_LOAD_UNLOAD_STATION_1) OR ("DB8000_PART_STATUS".UNIT_1.FIXTURE_3.PART_A.STATUS.PRESENT AND "DB8000_PART_STATUS".UNIT_1.FIXTURE_3.PART_A.STATUS.QUALITY_PART AND "DB5000_FIX_TABLE_POSITIONS".UNIT_1.FIXTURE[3].IN_LOAD_UNLOAD_STATION_1) OR ("DB8000_PART_STATUS".UNIT_1.FIXTURE_4.PART_A.STATUS.PRESENT AND "DB8000_PART_STATUS".UNIT_1.FIXTURE_4.PART_A.STATUS.QUALITY_PART AND "DB5000_FIX_TABLE_POSITIONS".UNIT_1.FIXTURE[4].IN_LOAD_UNLOAD_STATION_1);
END_REGION

REGION Network 52: MACHINE FIXTURE AT LOAD UNLOAD POSITION
   RUNG wire#powerrail
      Contact( "M_ONE" )
      wire#w1
      Contact( "DB5000_FIX_TABLE_POSITIONS".UNIT_1.FIXTURE[1].IN_LOAD_UNLOAD_STATION_1 )
      Coil( "DB7330_ETXETAR_ROBOT_CELL_INTERLOCK".INTERLOCKS_UNIT_01.MACHINE_TO_ROBOT.MCH_FIX_1_AT_LD_UNLD_POS )
   END_RUNG
   RUNG wire#w1
      Contact( "DB5000_FIX_TABLE_POSITIONS".UNIT_1.FIXTURE[2].IN_LOAD_UNLOAD_STATION_1 )
      Coil( "DB7330_ETXETAR_ROBOT_CELL_INTERLOCK".INTERLOCKS_UNIT_01.MACHINE_TO_ROBOT.MCH_FIX_2_AT_LD_UNLD_POS )
   END_RUNG
   RUNG wire#w1
      Contact( "DB5000_FIX_TABLE_POSITIONS".UNIT_1.FIXTURE[3].IN_LOAD_UNLOAD_STATION_1 )
      Coil( "DB7330_ETXETAR_ROBOT_CELL_INTERLOCK".INTERLOCKS_UNIT_01.MACHINE_TO_ROBOT.MCH_FIX_3_AT_LD_UNLD_POS )
   END_RUNG
   RUNG wire#w1
      Contact( "DB5000_FIX_TABLE_POSITIONS".UNIT_1.FIXTURE[4].IN_LOAD_UNLOAD_STATION_1 )
      Coil( "DB7330_ETXETAR_ROBOT_CELL_INTERLOCK".INTERLOCKS_UNIT_01.MACHINE_TO_ROBOT.MCH_FIX_4_AT_LD_UNLD_POS )
   END_RUNG
   // the same network as SCL:
   "DB7330_ETXETAR_ROBOT_CELL_INTERLOCK".INTERLOCKS_UNIT_01.MACHINE_TO_ROBOT.MCH_FIX_1_AT_LD_UNLD_POS := "M_ONE" AND "DB5000_FIX_TABLE_POSITIONS".UNIT_1.FIXTURE[1].IN_LOAD_UNLOAD_STATION_1;
   "DB7330_ETXETAR_ROBOT_CELL_INTERLOCK".INTERLOCKS_UNIT_01.MACHINE_TO_ROBOT.MCH_FIX_2_AT_LD_UNLD_POS := "M_ONE" AND "DB5000_FIX_TABLE_POSITIONS".UNIT_1.FIXTURE[2].IN_LOAD_UNLOAD_STATION_1;
   "DB7330_ETXETAR_ROBOT_CELL_INTERLOCK".INTERLOCKS_UNIT_01.MACHINE_TO_ROBOT.MCH_FIX_3_AT_LD_UNLD_POS := "M_ONE" AND "DB5000_FIX_TABLE_POSITIONS".UNIT_1.FIXTURE[3].IN_LOAD_UNLOAD_STATION_1;
   "DB7330_ETXETAR_ROBOT_CELL_INTERLOCK".INTERLOCKS_UNIT_01.MACHINE_TO_ROBOT.MCH_FIX_4_AT_LD_UNLD_POS := "M_ONE" AND "DB5000_FIX_TABLE_POSITIONS".UNIT_1.FIXTURE[4].IN_LOAD_UNLOAD_STATION_1;
END_REGION

REGION Network 53: MACHINE PART TYPE
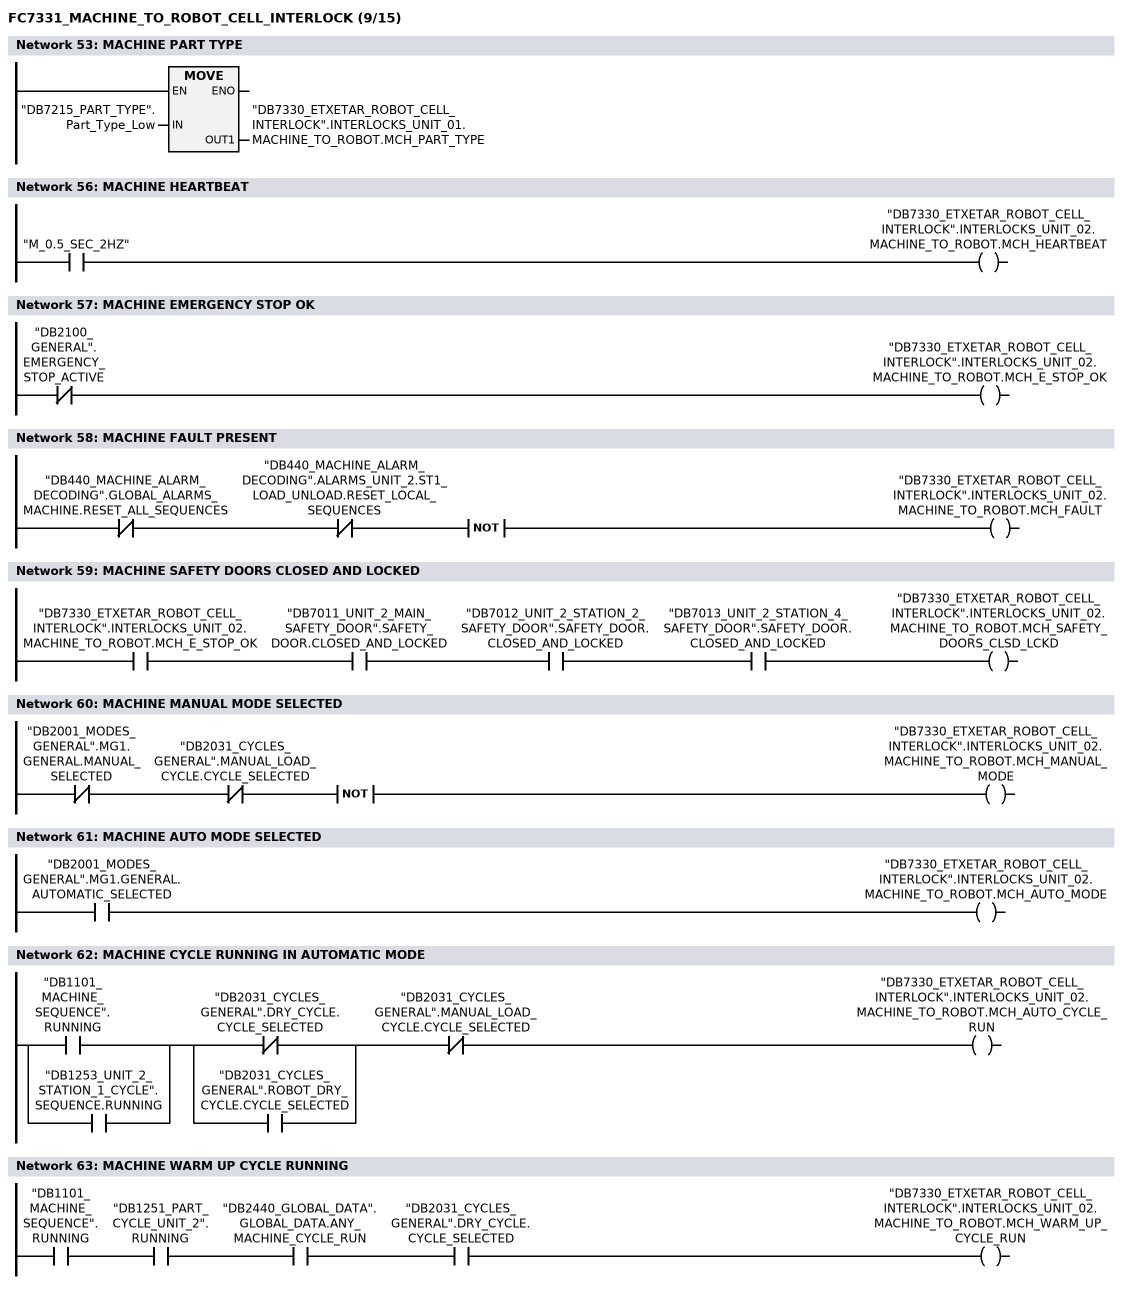
   RUNG wire#powerrail
      { S7_GenerateENO := "TRUE" } Move(in := "DB7215_PART_TYPE".Part_Type_Low, out1 => "DB7330_ETXETAR_ROBOT_CELL_INTERLOCK".INTERLOCKS_UNIT_01.MACHINE_TO_ROBOT.MCH_PART_TYPE)
   END_RUNG
   // the same network as SCL:
   "DB7330_ETXETAR_ROBOT_CELL_INTERLOCK".INTERLOCKS_UNIT_01.MACHINE_TO_ROBOT.MCH_PART_TYPE := "DB7215_PART_TYPE".Part_Type_Low;
END_REGION

REGION Network 55: >>>>>>>>>>>>>>>> INTERLOCKS MACHINE TO ROBOT UNIT 02 <<<<<<<<<<<<<<<<
END_REGION

REGION Network 56: MACHINE HEARTBEAT
   RUNG wire#powerrail
      Contact( "M_0.5_SEC_2HZ" )
      Coil( "DB7330_ETXETAR_ROBOT_CELL_INTERLOCK".INTERLOCKS_UNIT_02.MACHINE_TO_ROBOT.MCH_HEARTBEAT )
   END_RUNG
   // the same network as SCL:
   "DB7330_ETXETAR_ROBOT_CELL_INTERLOCK".INTERLOCKS_UNIT_02.MACHINE_TO_ROBOT.MCH_HEARTBEAT := "M_0.5_SEC_2HZ";
END_REGION

REGION Network 57: MACHINE EMERGENCY STOP OK
   RUNG wire#powerrail
      I_Contact( "DB2100_GENERAL".EMERGENCY_STOP_ACTIVE )
      Coil( "DB7330_ETXETAR_ROBOT_CELL_INTERLOCK".INTERLOCKS_UNIT_02.MACHINE_TO_ROBOT.MCH_E_STOP_OK )
   END_RUNG
   // the same network as SCL:
   "DB7330_ETXETAR_ROBOT_CELL_INTERLOCK".INTERLOCKS_UNIT_02.MACHINE_TO_ROBOT.MCH_E_STOP_OK := NOT "DB2100_GENERAL".EMERGENCY_STOP_ACTIVE;
END_REGION

REGION Network 58: MACHINE FAULT PRESENT
   RUNG wire#powerrail
      I_Contact( "DB440_MACHINE_ALARM_DECODING".GLOBAL_ALARMS_MACHINE.RESET_ALL_SEQUENCES )
      I_Contact( "DB440_MACHINE_ALARM_DECODING".ALARMS_UNIT_2.ST1_LOAD_UNLOAD.RESET_LOCAL_SEQUENCES )
      Not()
      Coil( "DB7330_ETXETAR_ROBOT_CELL_INTERLOCK".INTERLOCKS_UNIT_02.MACHINE_TO_ROBOT.MCH_FAULT )
   END_RUNG
   // the same network as SCL:
   "DB7330_ETXETAR_ROBOT_CELL_INTERLOCK".INTERLOCKS_UNIT_02.MACHINE_TO_ROBOT.MCH_FAULT := NOT (NOT "DB440_MACHINE_ALARM_DECODING".GLOBAL_ALARMS_MACHINE.RESET_ALL_SEQUENCES AND NOT "DB440_MACHINE_ALARM_DECODING".ALARMS_UNIT_2.ST1_LOAD_UNLOAD.RESET_LOCAL_SEQUENCES);
END_REGION

REGION Network 59: MACHINE SAFETY DOORS CLOSED AND LOCKED
   RUNG wire#powerrail
      Contact( "DB7330_ETXETAR_ROBOT_CELL_INTERLOCK".INTERLOCKS_UNIT_02.MACHINE_TO_ROBOT.MCH_E_STOP_OK )
      Contact( "DB7011_UNIT_2_MAIN_SAFETY_DOOR".SAFETY_DOOR.CLOSED_AND_LOCKED )
      Contact( "DB7012_UNIT_2_STATION_2_SAFETY_DOOR".SAFETY_DOOR.CLOSED_AND_LOCKED )
      Contact( "DB7013_UNIT_2_STATION_4_SAFETY_DOOR".SAFETY_DOOR.CLOSED_AND_LOCKED )
      Coil( "DB7330_ETXETAR_ROBOT_CELL_INTERLOCK".INTERLOCKS_UNIT_02.MACHINE_TO_ROBOT.MCH_SAFETY_DOORS_CLSD_LCKD )
   END_RUNG
   // the same network as SCL:
   "DB7330_ETXETAR_ROBOT_CELL_INTERLOCK".INTERLOCKS_UNIT_02.MACHINE_TO_ROBOT.MCH_SAFETY_DOORS_CLSD_LCKD := "DB7330_ETXETAR_ROBOT_CELL_INTERLOCK".INTERLOCKS_UNIT_02.MACHINE_TO_ROBOT.MCH_E_STOP_OK AND "DB7011_UNIT_2_MAIN_SAFETY_DOOR".SAFETY_DOOR.CLOSED_AND_LOCKED AND "DB7012_UNIT_2_STATION_2_SAFETY_DOOR".SAFETY_DOOR.CLOSED_AND_LOCKED AND "DB7013_UNIT_2_STATION_4_SAFETY_DOOR".SAFETY_DOOR.CLOSED_AND_LOCKED;
END_REGION

REGION Network 60: MACHINE MANUAL MODE SELECTED
   RUNG wire#powerrail
      I_Contact( "DB2001_MODES_GENERAL".MG1.GENERAL.MANUAL_SELECTED )
      I_Contact( "DB2031_CYCLES_GENERAL".MANUAL_LOAD_CYCLE.CYCLE_SELECTED )
      Not()
      Coil( "DB7330_ETXETAR_ROBOT_CELL_INTERLOCK".INTERLOCKS_UNIT_02.MACHINE_TO_ROBOT.MCH_MANUAL_MODE )
   END_RUNG
   // the same network as SCL:
   "DB7330_ETXETAR_ROBOT_CELL_INTERLOCK".INTERLOCKS_UNIT_02.MACHINE_TO_ROBOT.MCH_MANUAL_MODE := NOT (NOT "DB2001_MODES_GENERAL".MG1.GENERAL.MANUAL_SELECTED AND NOT "DB2031_CYCLES_GENERAL".MANUAL_LOAD_CYCLE.CYCLE_SELECTED);
END_REGION

REGION Network 61: MACHINE AUTO MODE SELECTED
   RUNG wire#powerrail
      Contact( "DB2001_MODES_GENERAL".MG1.GENERAL.AUTOMATIC_SELECTED )
      Coil( "DB7330_ETXETAR_ROBOT_CELL_INTERLOCK".INTERLOCKS_UNIT_02.MACHINE_TO_ROBOT.MCH_AUTO_MODE )
   END_RUNG
   // the same network as SCL:
   "DB7330_ETXETAR_ROBOT_CELL_INTERLOCK".INTERLOCKS_UNIT_02.MACHINE_TO_ROBOT.MCH_AUTO_MODE := "DB2001_MODES_GENERAL".MG1.GENERAL.AUTOMATIC_SELECTED;
END_REGION

REGION Network 62: MACHINE CYCLE RUNNING IN AUTOMATIC MODE
   RUNG wire#powerrail
      Contact( "DB1101_MACHINE_SEQUENCE".RUNNING )
      wire#w1
      I_Contact( "DB2031_CYCLES_GENERAL".DRY_CYCLE.CYCLE_SELECTED )
      wire#w2
      I_Contact( "DB2031_CYCLES_GENERAL".MANUAL_LOAD_CYCLE.CYCLE_SELECTED )
      Coil( "DB7330_ETXETAR_ROBOT_CELL_INTERLOCK".INTERLOCKS_UNIT_02.MACHINE_TO_ROBOT.MCH_AUTO_CYCLE_RUN )
   END_RUNG
   RUNG wire#powerrail
      Contact( "DB1253_UNIT_2_STATION_1_CYCLE".SEQUENCE.RUNNING )
   END_RUNG wire#w1
   RUNG wire#w1
      Contact( "DB2031_CYCLES_GENERAL".ROBOT_DRY_CYCLE.CYCLE_SELECTED )
   END_RUNG wire#w2
   // the same network as SCL:
   "DB7330_ETXETAR_ROBOT_CELL_INTERLOCK".INTERLOCKS_UNIT_02.MACHINE_TO_ROBOT.MCH_AUTO_CYCLE_RUN := ("DB1101_MACHINE_SEQUENCE".RUNNING OR "DB1253_UNIT_2_STATION_1_CYCLE".SEQUENCE.RUNNING) AND (NOT "DB2031_CYCLES_GENERAL".DRY_CYCLE.CYCLE_SELECTED OR "DB2031_CYCLES_GENERAL".ROBOT_DRY_CYCLE.CYCLE_SELECTED) AND NOT "DB2031_CYCLES_GENERAL".MANUAL_LOAD_CYCLE.CYCLE_SELECTED;
END_REGION

REGION Network 63: MACHINE WARM UP CYCLE RUNNING
   RUNG wire#powerrail
      Contact( "DB1101_MACHINE_SEQUENCE".RUNNING )
      Contact( "DB1251_PART_CYCLE_UNIT_2".RUNNING )
      Contact( "DB2440_GLOBAL_DATA".GLOBAL_DATA.ANY_MACHINE_CYCLE_RUN )
      Contact( "DB2031_CYCLES_GENERAL".DRY_CYCLE.CYCLE_SELECTED )
      Coil( "DB7330_ETXETAR_ROBOT_CELL_INTERLOCK".INTERLOCKS_UNIT_02.MACHINE_TO_ROBOT.MCH_WARM_UP_CYCLE_RUN )
   END_RUNG
   // the same network as SCL:
   "DB7330_ETXETAR_ROBOT_CELL_INTERLOCK".INTERLOCKS_UNIT_02.MACHINE_TO_ROBOT.MCH_WARM_UP_CYCLE_RUN := "DB1101_MACHINE_SEQUENCE".RUNNING AND "DB1251_PART_CYCLE_UNIT_2".RUNNING AND "DB2440_GLOBAL_DATA".GLOBAL_DATA.ANY_MACHINE_CYCLE_RUN AND "DB2031_CYCLES_GENERAL".DRY_CYCLE.CYCLE_SELECTED;
END_REGION

REGION Network 64: MACHINE RUN OUT CYCLE SELECTED
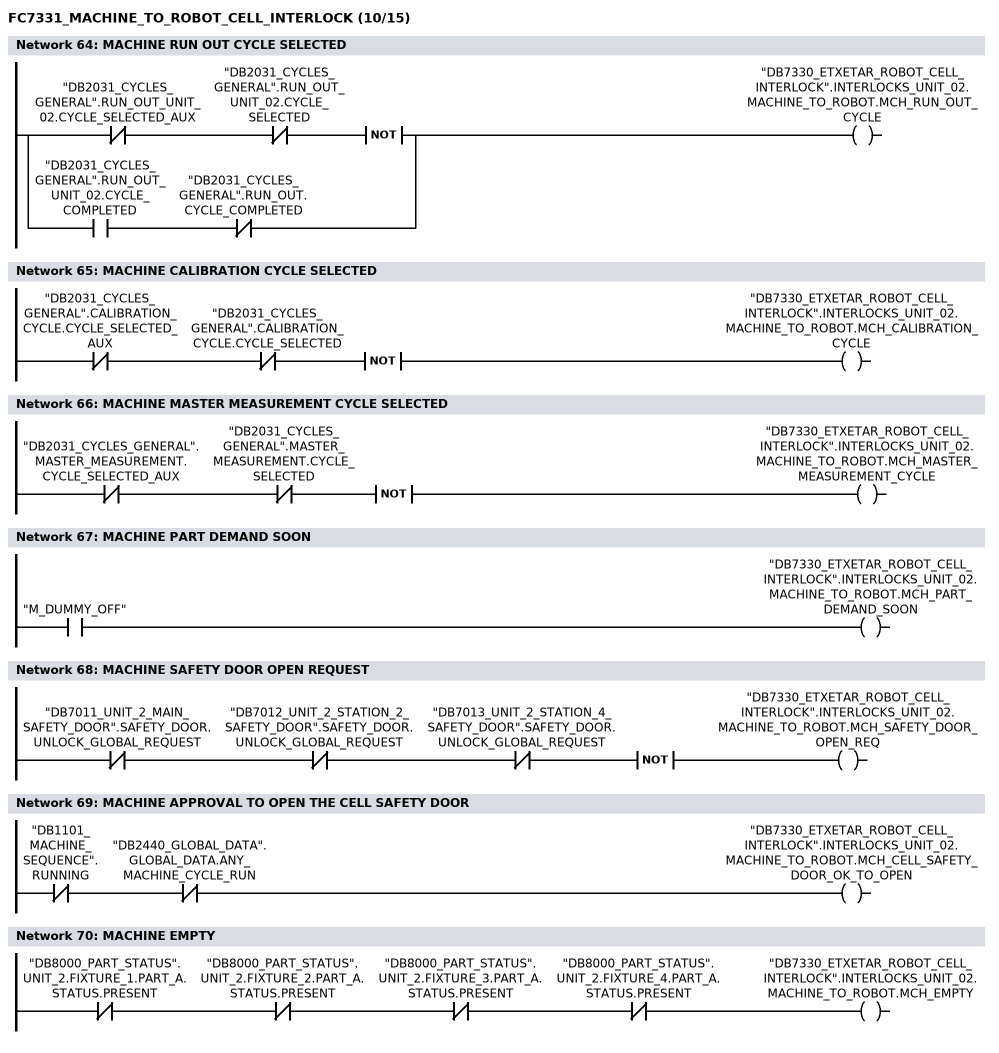
   RUNG wire#powerrail
      I_Contact( "DB2031_CYCLES_GENERAL".RUN_OUT_UNIT_02.CYCLE_SELECTED_AUX )
      I_Contact( "DB2031_CYCLES_GENERAL".RUN_OUT_UNIT_02.CYCLE_SELECTED )
      Not()
      wire#w1
      Coil( "DB7330_ETXETAR_ROBOT_CELL_INTERLOCK".INTERLOCKS_UNIT_02.MACHINE_TO_ROBOT.MCH_RUN_OUT_CYCLE )
   END_RUNG
   RUNG wire#powerrail
      Contact( "DB2031_CYCLES_GENERAL".RUN_OUT_UNIT_02.CYCLE_COMPLETED )
      I_Contact( "DB2031_CYCLES_GENERAL".RUN_OUT.CYCLE_COMPLETED )
   END_RUNG wire#w1
   // the same network as SCL:
   "DB7330_ETXETAR_ROBOT_CELL_INTERLOCK".INTERLOCKS_UNIT_02.MACHINE_TO_ROBOT.MCH_RUN_OUT_CYCLE := NOT (NOT "DB2031_CYCLES_GENERAL".RUN_OUT_UNIT_02.CYCLE_SELECTED_AUX AND NOT "DB2031_CYCLES_GENERAL".RUN_OUT_UNIT_02.CYCLE_SELECTED) OR ("DB2031_CYCLES_GENERAL".RUN_OUT_UNIT_02.CYCLE_COMPLETED AND NOT "DB2031_CYCLES_GENERAL".RUN_OUT.CYCLE_COMPLETED);
END_REGION

REGION Network 65: MACHINE CALIBRATION CYCLE SELECTED
   RUNG wire#powerrail
      I_Contact( "DB2031_CYCLES_GENERAL".CALIBRATION_CYCLE.CYCLE_SELECTED_AUX )
      I_Contact( "DB2031_CYCLES_GENERAL".CALIBRATION_CYCLE.CYCLE_SELECTED )
      Not()
      Coil( "DB7330_ETXETAR_ROBOT_CELL_INTERLOCK".INTERLOCKS_UNIT_02.MACHINE_TO_ROBOT.MCH_CALIBRATION_CYCLE )
   END_RUNG
   // the same network as SCL:
   "DB7330_ETXETAR_ROBOT_CELL_INTERLOCK".INTERLOCKS_UNIT_02.MACHINE_TO_ROBOT.MCH_CALIBRATION_CYCLE := NOT (NOT "DB2031_CYCLES_GENERAL".CALIBRATION_CYCLE.CYCLE_SELECTED_AUX AND NOT "DB2031_CYCLES_GENERAL".CALIBRATION_CYCLE.CYCLE_SELECTED);
END_REGION

REGION Network 66: MACHINE MASTER MEASUREMENT CYCLE SELECTED
   RUNG wire#powerrail
      I_Contact( "DB2031_CYCLES_GENERAL".MASTER_MEASUREMENT.CYCLE_SELECTED_AUX )
      I_Contact( "DB2031_CYCLES_GENERAL".MASTER_MEASUREMENT.CYCLE_SELECTED )
      Not()
      Coil( "DB7330_ETXETAR_ROBOT_CELL_INTERLOCK".INTERLOCKS_UNIT_02.MACHINE_TO_ROBOT.MCH_MASTER_MEASUREMENT_CYCLE )
   END_RUNG
   // the same network as SCL:
   "DB7330_ETXETAR_ROBOT_CELL_INTERLOCK".INTERLOCKS_UNIT_02.MACHINE_TO_ROBOT.MCH_MASTER_MEASUREMENT_CYCLE := NOT (NOT "DB2031_CYCLES_GENERAL".MASTER_MEASUREMENT.CYCLE_SELECTED_AUX AND NOT "DB2031_CYCLES_GENERAL".MASTER_MEASUREMENT.CYCLE_SELECTED);
END_REGION

REGION Network 67: MACHINE PART DEMAND SOON
   RUNG wire#powerrail
      Contact( "M_DUMMY_OFF" )
      Coil( "DB7330_ETXETAR_ROBOT_CELL_INTERLOCK".INTERLOCKS_UNIT_02.MACHINE_TO_ROBOT.MCH_PART_DEMAND_SOON )
   END_RUNG
   // the same network as SCL:
   "DB7330_ETXETAR_ROBOT_CELL_INTERLOCK".INTERLOCKS_UNIT_02.MACHINE_TO_ROBOT.MCH_PART_DEMAND_SOON := "M_DUMMY_OFF";
END_REGION

REGION Network 68: MACHINE SAFETY DOOR OPEN REQUEST
   RUNG wire#powerrail
      I_Contact( "DB7011_UNIT_2_MAIN_SAFETY_DOOR".SAFETY_DOOR.UNLOCK_GLOBAL_REQUEST )
      I_Contact( "DB7012_UNIT_2_STATION_2_SAFETY_DOOR".SAFETY_DOOR.UNLOCK_GLOBAL_REQUEST )
      I_Contact( "DB7013_UNIT_2_STATION_4_SAFETY_DOOR".SAFETY_DOOR.UNLOCK_GLOBAL_REQUEST )
      Not()
      Coil( "DB7330_ETXETAR_ROBOT_CELL_INTERLOCK".INTERLOCKS_UNIT_02.MACHINE_TO_ROBOT.MCH_SAFETY_DOOR_OPEN_REQ )
   END_RUNG
   // the same network as SCL:
   "DB7330_ETXETAR_ROBOT_CELL_INTERLOCK".INTERLOCKS_UNIT_02.MACHINE_TO_ROBOT.MCH_SAFETY_DOOR_OPEN_REQ := NOT (NOT "DB7011_UNIT_2_MAIN_SAFETY_DOOR".SAFETY_DOOR.UNLOCK_GLOBAL_REQUEST AND NOT "DB7012_UNIT_2_STATION_2_SAFETY_DOOR".SAFETY_DOOR.UNLOCK_GLOBAL_REQUEST AND NOT "DB7013_UNIT_2_STATION_4_SAFETY_DOOR".SAFETY_DOOR.UNLOCK_GLOBAL_REQUEST);
END_REGION

REGION Network 69: MACHINE APPROVAL TO OPEN THE CELL SAFETY DOOR
   RUNG wire#powerrail
      I_Contact( "DB1101_MACHINE_SEQUENCE".RUNNING )
      I_Contact( "DB2440_GLOBAL_DATA".GLOBAL_DATA.ANY_MACHINE_CYCLE_RUN )
      Coil( "DB7330_ETXETAR_ROBOT_CELL_INTERLOCK".INTERLOCKS_UNIT_02.MACHINE_TO_ROBOT.MCH_CELL_SAFETY_DOOR_OK_TO_OPEN )
   END_RUNG
   // the same network as SCL:
   "DB7330_ETXETAR_ROBOT_CELL_INTERLOCK".INTERLOCKS_UNIT_02.MACHINE_TO_ROBOT.MCH_CELL_SAFETY_DOOR_OK_TO_OPEN := NOT "DB1101_MACHINE_SEQUENCE".RUNNING AND NOT "DB2440_GLOBAL_DATA".GLOBAL_DATA.ANY_MACHINE_CYCLE_RUN;
END_REGION

REGION Network 70: MACHINE EMPTY
   RUNG wire#powerrail
      I_Contact( "DB8000_PART_STATUS".UNIT_2.FIXTURE_1.PART_A.STATUS.PRESENT )
      I_Contact( "DB8000_PART_STATUS".UNIT_2.FIXTURE_2.PART_A.STATUS.PRESENT )
      I_Contact( "DB8000_PART_STATUS".UNIT_2.FIXTURE_3.PART_A.STATUS.PRESENT )
      I_Contact( "DB8000_PART_STATUS".UNIT_2.FIXTURE_4.PART_A.STATUS.PRESENT )
      Coil( "DB7330_ETXETAR_ROBOT_CELL_INTERLOCK".INTERLOCKS_UNIT_02.MACHINE_TO_ROBOT.MCH_EMPTY )
   END_RUNG
   // the same network as SCL:
   "DB7330_ETXETAR_ROBOT_CELL_INTERLOCK".INTERLOCKS_UNIT_02.MACHINE_TO_ROBOT.MCH_EMPTY := NOT "DB8000_PART_STATUS".UNIT_2.FIXTURE_1.PART_A.STATUS.PRESENT AND NOT "DB8000_PART_STATUS".UNIT_2.FIXTURE_2.PART_A.STATUS.PRESENT AND NOT "DB8000_PART_STATUS".UNIT_2.FIXTURE_3.PART_A.STATUS.PRESENT AND NOT "DB8000_PART_STATUS".UNIT_2.FIXTURE_4.PART_A.STATUS.PRESENT;
END_REGION

REGION Network 71: MACHINE FIXTURES ENABLED
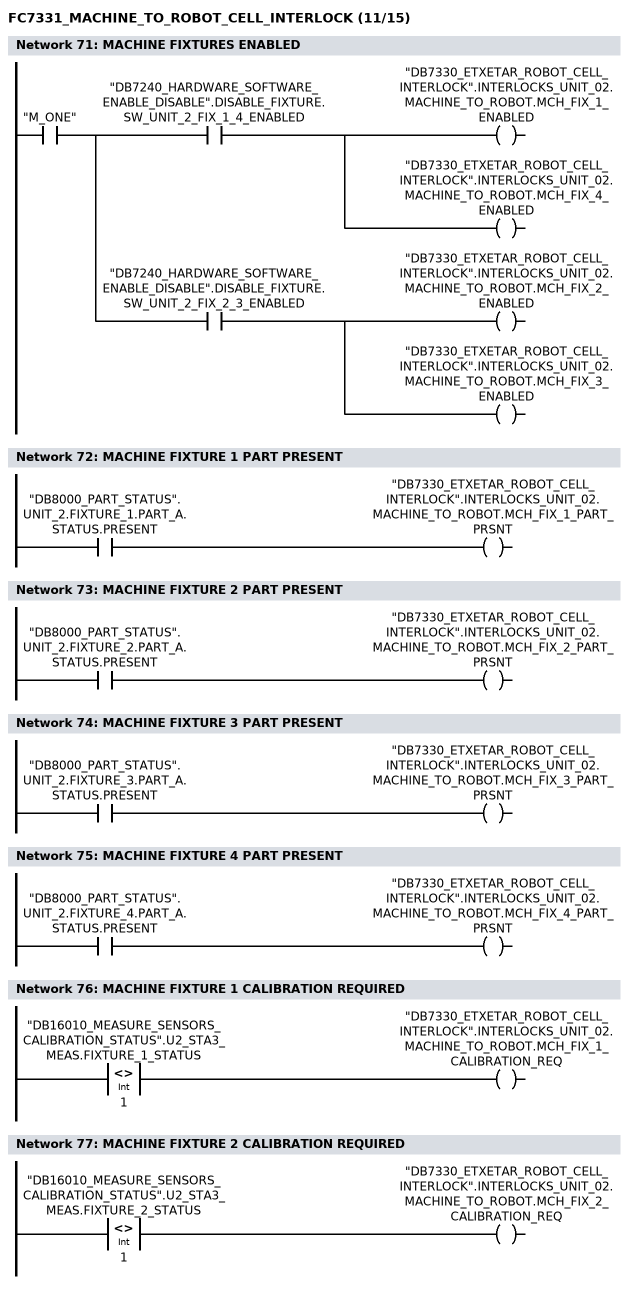
   RUNG wire#powerrail
      Contact( "M_ONE" )
      wire#w1
      Contact( "DB7240_HARDWARE_SOFTWARE_ENABLE_DISABLE".DISABLE_FIXTURE.SW_UNIT_2_FIX_1_4_ENABLED )
      wire#w2
      Coil( "DB7330_ETXETAR_ROBOT_CELL_INTERLOCK".INTERLOCKS_UNIT_02.MACHINE_TO_ROBOT.MCH_FIX_1_ENABLED )
   END_RUNG
   RUNG wire#w2
      Coil( "DB7330_ETXETAR_ROBOT_CELL_INTERLOCK".INTERLOCKS_UNIT_02.MACHINE_TO_ROBOT.MCH_FIX_4_ENABLED )
   END_RUNG
   RUNG wire#w1
      Contact( "DB7240_HARDWARE_SOFTWARE_ENABLE_DISABLE".DISABLE_FIXTURE.SW_UNIT_2_FIX_2_3_ENABLED )
      wire#w3
      Coil( "DB7330_ETXETAR_ROBOT_CELL_INTERLOCK".INTERLOCKS_UNIT_02.MACHINE_TO_ROBOT.MCH_FIX_2_ENABLED )
   END_RUNG
   RUNG wire#w3
      Coil( "DB7330_ETXETAR_ROBOT_CELL_INTERLOCK".INTERLOCKS_UNIT_02.MACHINE_TO_ROBOT.MCH_FIX_3_ENABLED )
   END_RUNG
   // the same network as SCL:
   "DB7330_ETXETAR_ROBOT_CELL_INTERLOCK".INTERLOCKS_UNIT_02.MACHINE_TO_ROBOT.MCH_FIX_1_ENABLED := "M_ONE" AND "DB7240_HARDWARE_SOFTWARE_ENABLE_DISABLE".DISABLE_FIXTURE.SW_UNIT_2_FIX_1_4_ENABLED;
   "DB7330_ETXETAR_ROBOT_CELL_INTERLOCK".INTERLOCKS_UNIT_02.MACHINE_TO_ROBOT.MCH_FIX_4_ENABLED := "DB7330_ETXETAR_ROBOT_CELL_INTERLOCK".INTERLOCKS_UNIT_02.MACHINE_TO_ROBOT.MCH_FIX_1_ENABLED;
   "DB7330_ETXETAR_ROBOT_CELL_INTERLOCK".INTERLOCKS_UNIT_02.MACHINE_TO_ROBOT.MCH_FIX_2_ENABLED := "M_ONE" AND "DB7240_HARDWARE_SOFTWARE_ENABLE_DISABLE".DISABLE_FIXTURE.SW_UNIT_2_FIX_2_3_ENABLED;
   "DB7330_ETXETAR_ROBOT_CELL_INTERLOCK".INTERLOCKS_UNIT_02.MACHINE_TO_ROBOT.MCH_FIX_3_ENABLED := "DB7330_ETXETAR_ROBOT_CELL_INTERLOCK".INTERLOCKS_UNIT_02.MACHINE_TO_ROBOT.MCH_FIX_2_ENABLED;
END_REGION

REGION Network 72: MACHINE FIXTURE 1 PART PRESENT
   RUNG wire#powerrail
      Contact( "DB8000_PART_STATUS".UNIT_2.FIXTURE_1.PART_A.STATUS.PRESENT )
      Coil( "DB7330_ETXETAR_ROBOT_CELL_INTERLOCK".INTERLOCKS_UNIT_02.MACHINE_TO_ROBOT.MCH_FIX_1_PART_PRSNT )
   END_RUNG
   // the same network as SCL:
   "DB7330_ETXETAR_ROBOT_CELL_INTERLOCK".INTERLOCKS_UNIT_02.MACHINE_TO_ROBOT.MCH_FIX_1_PART_PRSNT := "DB8000_PART_STATUS".UNIT_2.FIXTURE_1.PART_A.STATUS.PRESENT;
END_REGION

REGION Network 73: MACHINE FIXTURE 2 PART PRESENT
   RUNG wire#powerrail
      Contact( "DB8000_PART_STATUS".UNIT_2.FIXTURE_2.PART_A.STATUS.PRESENT )
      Coil( "DB7330_ETXETAR_ROBOT_CELL_INTERLOCK".INTERLOCKS_UNIT_02.MACHINE_TO_ROBOT.MCH_FIX_2_PART_PRSNT )
   END_RUNG
   // the same network as SCL:
   "DB7330_ETXETAR_ROBOT_CELL_INTERLOCK".INTERLOCKS_UNIT_02.MACHINE_TO_ROBOT.MCH_FIX_2_PART_PRSNT := "DB8000_PART_STATUS".UNIT_2.FIXTURE_2.PART_A.STATUS.PRESENT;
END_REGION

REGION Network 74: MACHINE FIXTURE 3 PART PRESENT
   RUNG wire#powerrail
      Contact( "DB8000_PART_STATUS".UNIT_2.FIXTURE_3.PART_A.STATUS.PRESENT )
      Coil( "DB7330_ETXETAR_ROBOT_CELL_INTERLOCK".INTERLOCKS_UNIT_02.MACHINE_TO_ROBOT.MCH_FIX_3_PART_PRSNT )
   END_RUNG
   // the same network as SCL:
   "DB7330_ETXETAR_ROBOT_CELL_INTERLOCK".INTERLOCKS_UNIT_02.MACHINE_TO_ROBOT.MCH_FIX_3_PART_PRSNT := "DB8000_PART_STATUS".UNIT_2.FIXTURE_3.PART_A.STATUS.PRESENT;
END_REGION

REGION Network 75: MACHINE FIXTURE 4 PART PRESENT
   RUNG wire#powerrail
      Contact( "DB8000_PART_STATUS".UNIT_2.FIXTURE_4.PART_A.STATUS.PRESENT )
      Coil( "DB7330_ETXETAR_ROBOT_CELL_INTERLOCK".INTERLOCKS_UNIT_02.MACHINE_TO_ROBOT.MCH_FIX_4_PART_PRSNT )
   END_RUNG
   // the same network as SCL:
   "DB7330_ETXETAR_ROBOT_CELL_INTERLOCK".INTERLOCKS_UNIT_02.MACHINE_TO_ROBOT.MCH_FIX_4_PART_PRSNT := "DB8000_PART_STATUS".UNIT_2.FIXTURE_4.PART_A.STATUS.PRESENT;
END_REGION

REGION Network 76: MACHINE FIXTURE 1 CALIBRATION REQUIRED
   RUNG wire#powerrail
      { S7_Templates := "SrcType := Int" } NE_Contact(in1 := "DB16010_MEASURE_SENSORS_CALIBRATION_STATUS".U2_STA3_MEAS.FIXTURE_1_STATUS, in2 := 1)
      Coil( "DB7330_ETXETAR_ROBOT_CELL_INTERLOCK".INTERLOCKS_UNIT_02.MACHINE_TO_ROBOT.MCH_FIX_1_CALIBRATION_REQ )
   END_RUNG
   // the same network as SCL:
   "DB7330_ETXETAR_ROBOT_CELL_INTERLOCK".INTERLOCKS_UNIT_02.MACHINE_TO_ROBOT.MCH_FIX_1_CALIBRATION_REQ := "DB16010_MEASURE_SENSORS_CALIBRATION_STATUS".U2_STA3_MEAS.FIXTURE_1_STATUS <> 1;
END_REGION

REGION Network 77: MACHINE FIXTURE 2 CALIBRATION REQUIRED
   RUNG wire#powerrail
      { S7_Templates := "SrcType := Int" } NE_Contact(in1 := "DB16010_MEASURE_SENSORS_CALIBRATION_STATUS".U2_STA3_MEAS.FIXTURE_2_STATUS, in2 := 1)
      Coil( "DB7330_ETXETAR_ROBOT_CELL_INTERLOCK".INTERLOCKS_UNIT_02.MACHINE_TO_ROBOT.MCH_FIX_2_CALIBRATION_REQ )
   END_RUNG
   // the same network as SCL:
   "DB7330_ETXETAR_ROBOT_CELL_INTERLOCK".INTERLOCKS_UNIT_02.MACHINE_TO_ROBOT.MCH_FIX_2_CALIBRATION_REQ := "DB16010_MEASURE_SENSORS_CALIBRATION_STATUS".U2_STA3_MEAS.FIXTURE_2_STATUS <> 1;
END_REGION

REGION Network 78: MACHINE FIXTURE 3 CALIBRATION REQUIRED
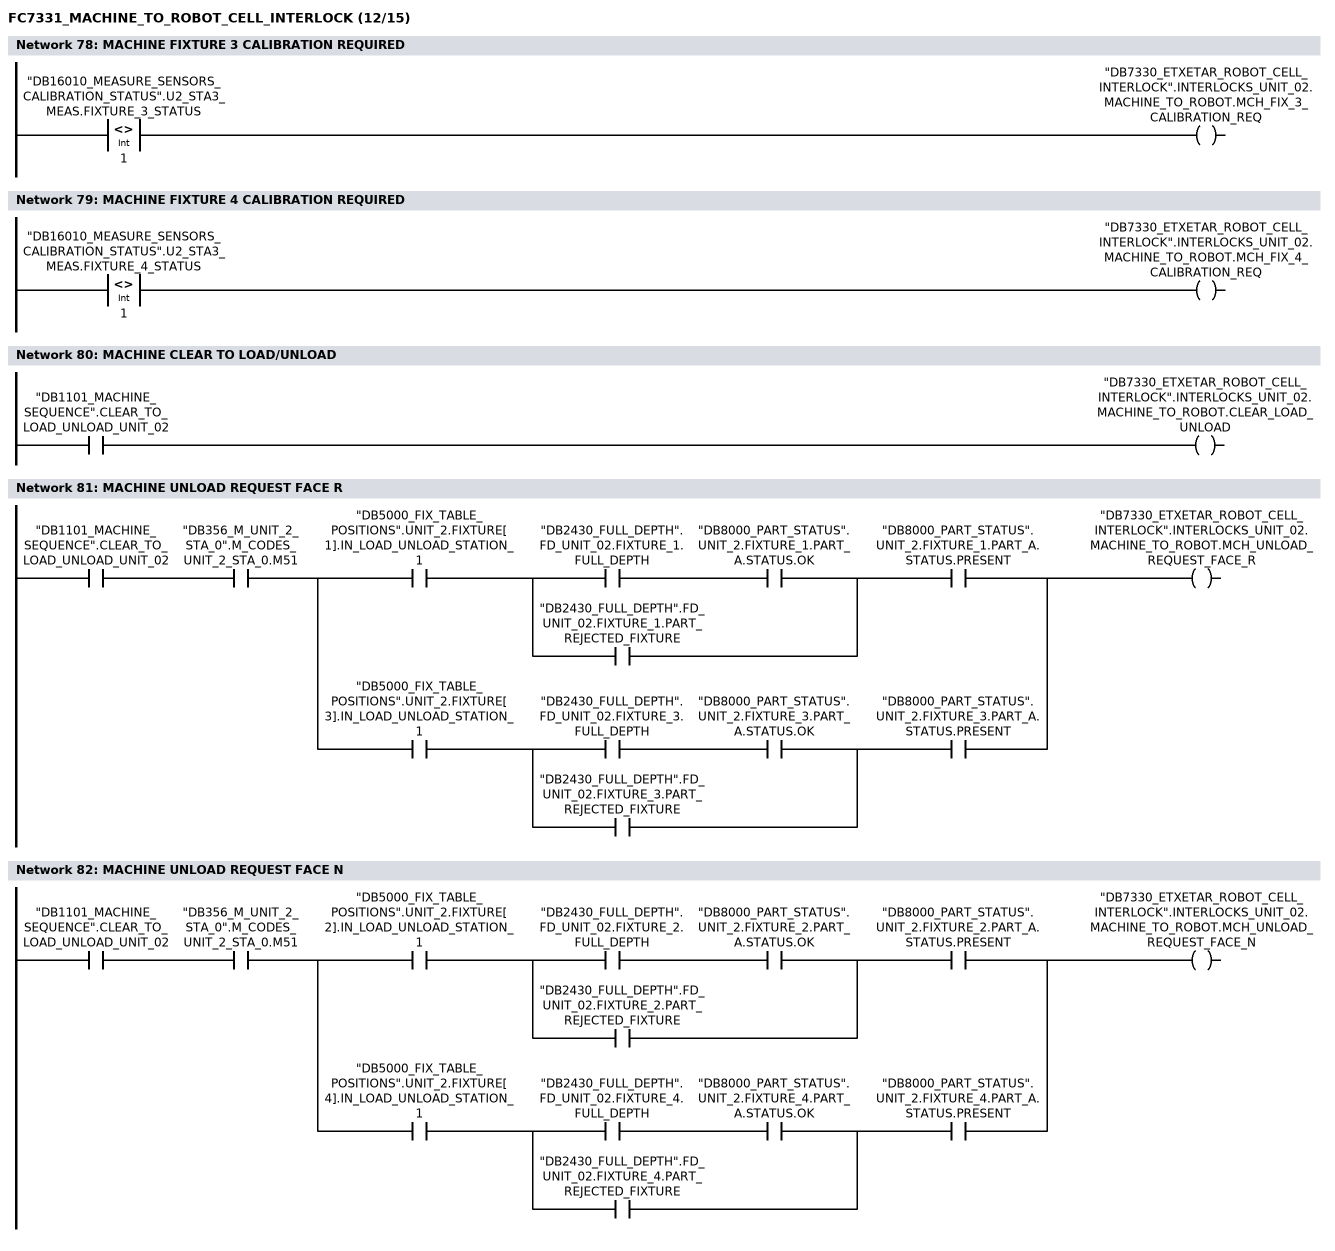
   RUNG wire#powerrail
      { S7_Templates := "SrcType := Int" } NE_Contact(in1 := "DB16010_MEASURE_SENSORS_CALIBRATION_STATUS".U2_STA3_MEAS.FIXTURE_3_STATUS, in2 := 1)
      Coil( "DB7330_ETXETAR_ROBOT_CELL_INTERLOCK".INTERLOCKS_UNIT_02.MACHINE_TO_ROBOT.MCH_FIX_3_CALIBRATION_REQ )
   END_RUNG
   // the same network as SCL:
   "DB7330_ETXETAR_ROBOT_CELL_INTERLOCK".INTERLOCKS_UNIT_02.MACHINE_TO_ROBOT.MCH_FIX_3_CALIBRATION_REQ := "DB16010_MEASURE_SENSORS_CALIBRATION_STATUS".U2_STA3_MEAS.FIXTURE_3_STATUS <> 1;
END_REGION

REGION Network 79: MACHINE FIXTURE 4 CALIBRATION REQUIRED
   RUNG wire#powerrail
      { S7_Templates := "SrcType := Int" } NE_Contact(in1 := "DB16010_MEASURE_SENSORS_CALIBRATION_STATUS".U2_STA3_MEAS.FIXTURE_4_STATUS, in2 := 1)
      Coil( "DB7330_ETXETAR_ROBOT_CELL_INTERLOCK".INTERLOCKS_UNIT_02.MACHINE_TO_ROBOT.MCH_FIX_4_CALIBRATION_REQ )
   END_RUNG
   // the same network as SCL:
   "DB7330_ETXETAR_ROBOT_CELL_INTERLOCK".INTERLOCKS_UNIT_02.MACHINE_TO_ROBOT.MCH_FIX_4_CALIBRATION_REQ := "DB16010_MEASURE_SENSORS_CALIBRATION_STATUS".U2_STA3_MEAS.FIXTURE_4_STATUS <> 1;
END_REGION

REGION Network 80: MACHINE CLEAR TO LOAD/UNLOAD
   RUNG wire#powerrail
      Contact( "DB1101_MACHINE_SEQUENCE".CLEAR_TO_LOAD_UNLOAD_UNIT_02 )
      Coil( "DB7330_ETXETAR_ROBOT_CELL_INTERLOCK".INTERLOCKS_UNIT_02.MACHINE_TO_ROBOT.CLEAR_LOAD_UNLOAD )
   END_RUNG
   // the same network as SCL:
   "DB7330_ETXETAR_ROBOT_CELL_INTERLOCK".INTERLOCKS_UNIT_02.MACHINE_TO_ROBOT.CLEAR_LOAD_UNLOAD := "DB1101_MACHINE_SEQUENCE".CLEAR_TO_LOAD_UNLOAD_UNIT_02;
END_REGION

REGION Network 81: MACHINE UNLOAD REQUEST FACE R
   RUNG wire#powerrail
      Contact( "DB1101_MACHINE_SEQUENCE".CLEAR_TO_LOAD_UNLOAD_UNIT_02 )
      Contact( "DB356_M_UNIT_2_STA_0".M_CODES_UNIT_2_STA_0.M51 )
      wire#w1
      Contact( "DB5000_FIX_TABLE_POSITIONS".UNIT_2.FIXTURE[1].IN_LOAD_UNLOAD_STATION_1 )
      wire#w2
      Contact( "DB2430_FULL_DEPTH".FD_UNIT_02.FIXTURE_1.FULL_DEPTH )
      Contact( "DB8000_PART_STATUS".UNIT_2.FIXTURE_1.PART_A.STATUS.OK )
      wire#w3
      Contact( "DB8000_PART_STATUS".UNIT_2.FIXTURE_1.PART_A.STATUS.PRESENT )
      wire#w4
      Coil( "DB7330_ETXETAR_ROBOT_CELL_INTERLOCK".INTERLOCKS_UNIT_02.MACHINE_TO_ROBOT.MCH_UNLOAD_REQUEST_FACE_R )
   END_RUNG
   RUNG wire#w2
      Contact( "DB2430_FULL_DEPTH".FD_UNIT_02.FIXTURE_1.PART_REJECTED_FIXTURE )
   END_RUNG wire#w3
   RUNG wire#w1
      Contact( "DB5000_FIX_TABLE_POSITIONS".UNIT_2.FIXTURE[3].IN_LOAD_UNLOAD_STATION_1 )
      wire#w5
      Contact( "DB2430_FULL_DEPTH".FD_UNIT_02.FIXTURE_3.FULL_DEPTH )
      Contact( "DB8000_PART_STATUS".UNIT_2.FIXTURE_3.PART_A.STATUS.OK )
      wire#w6
      Contact( "DB8000_PART_STATUS".UNIT_2.FIXTURE_3.PART_A.STATUS.PRESENT )
   END_RUNG wire#w4
   RUNG wire#w5
      Contact( "DB2430_FULL_DEPTH".FD_UNIT_02.FIXTURE_3.PART_REJECTED_FIXTURE )
   END_RUNG wire#w6
   // the same network as SCL:
   "DB7330_ETXETAR_ROBOT_CELL_INTERLOCK".INTERLOCKS_UNIT_02.MACHINE_TO_ROBOT.MCH_UNLOAD_REQUEST_FACE_R := "DB1101_MACHINE_SEQUENCE".CLEAR_TO_LOAD_UNLOAD_UNIT_02 AND "DB356_M_UNIT_2_STA_0".M_CODES_UNIT_2_STA_0.M51 AND (("DB5000_FIX_TABLE_POSITIONS".UNIT_2.FIXTURE[1].IN_LOAD_UNLOAD_STATION_1 AND (("DB2430_FULL_DEPTH".FD_UNIT_02.FIXTURE_1.FULL_DEPTH AND "DB8000_PART_STATUS".UNIT_2.FIXTURE_1.PART_A.STATUS.OK) OR "DB2430_FULL_DEPTH".FD_UNIT_02.FIXTURE_1.PART_REJECTED_FIXTURE) AND "DB8000_PART_STATUS".UNIT_2.FIXTURE_1.PART_A.STATUS.PRESENT) OR ("DB5000_FIX_TABLE_POSITIONS".UNIT_2.FIXTURE[3].IN_LOAD_UNLOAD_STATION_1 AND (("DB2430_FULL_DEPTH".FD_UNIT_02.FIXTURE_3.FULL_DEPTH AND "DB8000_PART_STATUS".UNIT_2.FIXTURE_3.PART_A.STATUS.OK) OR "DB2430_FULL_DEPTH".FD_UNIT_02.FIXTURE_3.PART_REJECTED_FIXTURE) AND "DB8000_PART_STATUS".UNIT_2.FIXTURE_3.PART_A.STATUS.PRESENT));
END_REGION

REGION Network 82: MACHINE UNLOAD REQUEST FACE N
   RUNG wire#powerrail
      Contact( "DB1101_MACHINE_SEQUENCE".CLEAR_TO_LOAD_UNLOAD_UNIT_02 )
      Contact( "DB356_M_UNIT_2_STA_0".M_CODES_UNIT_2_STA_0.M51 )
      wire#w1
      Contact( "DB5000_FIX_TABLE_POSITIONS".UNIT_2.FIXTURE[2].IN_LOAD_UNLOAD_STATION_1 )
      wire#w2
      Contact( "DB2430_FULL_DEPTH".FD_UNIT_02.FIXTURE_2.FULL_DEPTH )
      Contact( "DB8000_PART_STATUS".UNIT_2.FIXTURE_2.PART_A.STATUS.OK )
      wire#w3
      Contact( "DB8000_PART_STATUS".UNIT_2.FIXTURE_2.PART_A.STATUS.PRESENT )
      wire#w4
      Coil( "DB7330_ETXETAR_ROBOT_CELL_INTERLOCK".INTERLOCKS_UNIT_02.MACHINE_TO_ROBOT.MCH_UNLOAD_REQUEST_FACE_N )
   END_RUNG
   RUNG wire#w2
      Contact( "DB2430_FULL_DEPTH".FD_UNIT_02.FIXTURE_2.PART_REJECTED_FIXTURE )
   END_RUNG wire#w3
   RUNG wire#w1
      Contact( "DB5000_FIX_TABLE_POSITIONS".UNIT_2.FIXTURE[4].IN_LOAD_UNLOAD_STATION_1 )
      wire#w5
      Contact( "DB2430_FULL_DEPTH".FD_UNIT_02.FIXTURE_4.FULL_DEPTH )
      Contact( "DB8000_PART_STATUS".UNIT_2.FIXTURE_4.PART_A.STATUS.OK )
      wire#w6
      Contact( "DB8000_PART_STATUS".UNIT_2.FIXTURE_4.PART_A.STATUS.PRESENT )
   END_RUNG wire#w4
   RUNG wire#w5
      Contact( "DB2430_FULL_DEPTH".FD_UNIT_02.FIXTURE_4.PART_REJECTED_FIXTURE )
   END_RUNG wire#w6
   // the same network as SCL:
   "DB7330_ETXETAR_ROBOT_CELL_INTERLOCK".INTERLOCKS_UNIT_02.MACHINE_TO_ROBOT.MCH_UNLOAD_REQUEST_FACE_N := "DB1101_MACHINE_SEQUENCE".CLEAR_TO_LOAD_UNLOAD_UNIT_02 AND "DB356_M_UNIT_2_STA_0".M_CODES_UNIT_2_STA_0.M51 AND (("DB5000_FIX_TABLE_POSITIONS".UNIT_2.FIXTURE[2].IN_LOAD_UNLOAD_STATION_1 AND (("DB2430_FULL_DEPTH".FD_UNIT_02.FIXTURE_2.FULL_DEPTH AND "DB8000_PART_STATUS".UNIT_2.FIXTURE_2.PART_A.STATUS.OK) OR "DB2430_FULL_DEPTH".FD_UNIT_02.FIXTURE_2.PART_REJECTED_FIXTURE) AND "DB8000_PART_STATUS".UNIT_2.FIXTURE_2.PART_A.STATUS.PRESENT) OR ("DB5000_FIX_TABLE_POSITIONS".UNIT_2.FIXTURE[4].IN_LOAD_UNLOAD_STATION_1 AND (("DB2430_FULL_DEPTH".FD_UNIT_02.FIXTURE_4.FULL_DEPTH AND "DB8000_PART_STATUS".UNIT_2.FIXTURE_4.PART_A.STATUS.OK) OR "DB2430_FULL_DEPTH".FD_UNIT_02.FIXTURE_4.PART_REJECTED_FIXTURE) AND "DB8000_PART_STATUS".UNIT_2.FIXTURE_4.PART_A.STATUS.PRESENT));
END_REGION

REGION Network 83: MACHINE LOAD REQUEST FACE R
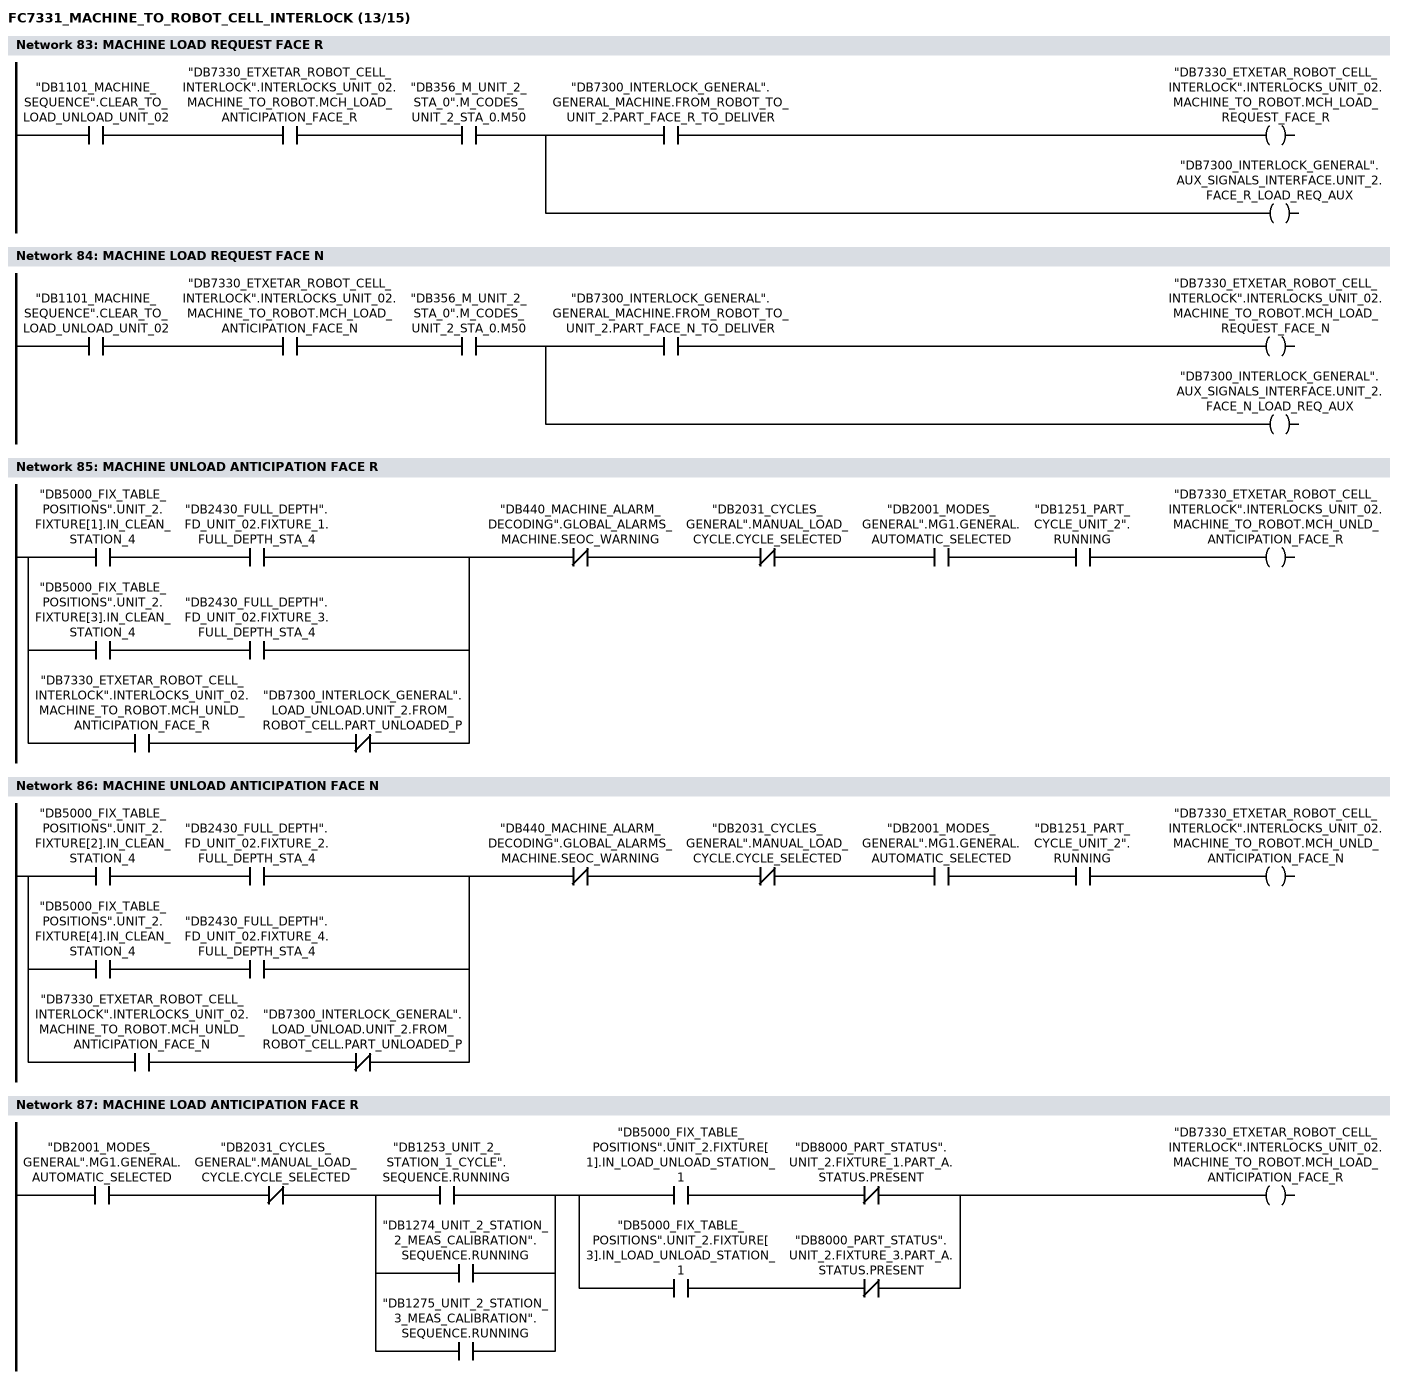
   RUNG wire#powerrail
      Contact( "DB1101_MACHINE_SEQUENCE".CLEAR_TO_LOAD_UNLOAD_UNIT_02 )
      Contact( "DB7330_ETXETAR_ROBOT_CELL_INTERLOCK".INTERLOCKS_UNIT_02.MACHINE_TO_ROBOT.MCH_LOAD_ANTICIPATION_FACE_R )
      Contact( "DB356_M_UNIT_2_STA_0".M_CODES_UNIT_2_STA_0.M50 )
      wire#w1
      Contact( "DB7300_INTERLOCK_GENERAL".GENERAL_MACHINE.FROM_ROBOT_TO_UNIT_2.PART_FACE_R_TO_DELIVER )
      Coil( "DB7330_ETXETAR_ROBOT_CELL_INTERLOCK".INTERLOCKS_UNIT_02.MACHINE_TO_ROBOT.MCH_LOAD_REQUEST_FACE_R )
   END_RUNG
   RUNG wire#w1
      Coil( "DB7300_INTERLOCK_GENERAL".AUX_SIGNALS_INTERFACE.UNIT_2.FACE_R_LOAD_REQ_AUX )
   END_RUNG
   // the same network as SCL:
   #_w1 := "DB1101_MACHINE_SEQUENCE".CLEAR_TO_LOAD_UNLOAD_UNIT_02 AND "DB7330_ETXETAR_ROBOT_CELL_INTERLOCK".INTERLOCKS_UNIT_02.MACHINE_TO_ROBOT.MCH_LOAD_ANTICIPATION_FACE_R AND "DB356_M_UNIT_2_STA_0".M_CODES_UNIT_2_STA_0.M50;
   "DB7330_ETXETAR_ROBOT_CELL_INTERLOCK".INTERLOCKS_UNIT_02.MACHINE_TO_ROBOT.MCH_LOAD_REQUEST_FACE_R := #_w1 AND "DB7300_INTERLOCK_GENERAL".GENERAL_MACHINE.FROM_ROBOT_TO_UNIT_2.PART_FACE_R_TO_DELIVER;
   "DB7300_INTERLOCK_GENERAL".AUX_SIGNALS_INTERFACE.UNIT_2.FACE_R_LOAD_REQ_AUX := #_w1;
END_REGION

REGION Network 84: MACHINE LOAD REQUEST FACE N
   RUNG wire#powerrail
      Contact( "DB1101_MACHINE_SEQUENCE".CLEAR_TO_LOAD_UNLOAD_UNIT_02 )
      Contact( "DB7330_ETXETAR_ROBOT_CELL_INTERLOCK".INTERLOCKS_UNIT_02.MACHINE_TO_ROBOT.MCH_LOAD_ANTICIPATION_FACE_N )
      Contact( "DB356_M_UNIT_2_STA_0".M_CODES_UNIT_2_STA_0.M50 )
      wire#w1
      Contact( "DB7300_INTERLOCK_GENERAL".GENERAL_MACHINE.FROM_ROBOT_TO_UNIT_2.PART_FACE_N_TO_DELIVER )
      Coil( "DB7330_ETXETAR_ROBOT_CELL_INTERLOCK".INTERLOCKS_UNIT_02.MACHINE_TO_ROBOT.MCH_LOAD_REQUEST_FACE_N )
   END_RUNG
   RUNG wire#w1
      Coil( "DB7300_INTERLOCK_GENERAL".AUX_SIGNALS_INTERFACE.UNIT_2.FACE_N_LOAD_REQ_AUX )
   END_RUNG
   // the same network as SCL:
   #_w1 := "DB1101_MACHINE_SEQUENCE".CLEAR_TO_LOAD_UNLOAD_UNIT_02 AND "DB7330_ETXETAR_ROBOT_CELL_INTERLOCK".INTERLOCKS_UNIT_02.MACHINE_TO_ROBOT.MCH_LOAD_ANTICIPATION_FACE_N AND "DB356_M_UNIT_2_STA_0".M_CODES_UNIT_2_STA_0.M50;
   "DB7330_ETXETAR_ROBOT_CELL_INTERLOCK".INTERLOCKS_UNIT_02.MACHINE_TO_ROBOT.MCH_LOAD_REQUEST_FACE_N := #_w1 AND "DB7300_INTERLOCK_GENERAL".GENERAL_MACHINE.FROM_ROBOT_TO_UNIT_2.PART_FACE_N_TO_DELIVER;
   "DB7300_INTERLOCK_GENERAL".AUX_SIGNALS_INTERFACE.UNIT_2.FACE_N_LOAD_REQ_AUX := #_w1;
END_REGION

REGION Network 85: MACHINE UNLOAD ANTICIPATION FACE R
   RUNG wire#powerrail
      Contact( "DB5000_FIX_TABLE_POSITIONS".UNIT_2.FIXTURE[1].IN_CLEAN_STATION_4 )
      Contact( "DB2430_FULL_DEPTH".FD_UNIT_02.FIXTURE_1.FULL_DEPTH_STA_4 )
      wire#w1
      I_Contact( "DB440_MACHINE_ALARM_DECODING".GLOBAL_ALARMS_MACHINE.SEOC_WARNING )
      I_Contact( "DB2031_CYCLES_GENERAL".MANUAL_LOAD_CYCLE.CYCLE_SELECTED )
      Contact( "DB2001_MODES_GENERAL".MG1.GENERAL.AUTOMATIC_SELECTED )
      Contact( "DB1251_PART_CYCLE_UNIT_2".RUNNING )
      Coil( "DB7330_ETXETAR_ROBOT_CELL_INTERLOCK".INTERLOCKS_UNIT_02.MACHINE_TO_ROBOT.MCH_UNLD_ANTICIPATION_FACE_R )
   END_RUNG
   RUNG wire#powerrail
      Contact( "DB5000_FIX_TABLE_POSITIONS".UNIT_2.FIXTURE[3].IN_CLEAN_STATION_4 )
      Contact( "DB2430_FULL_DEPTH".FD_UNIT_02.FIXTURE_3.FULL_DEPTH_STA_4 )
   END_RUNG wire#w1
   RUNG wire#powerrail
      Contact( "DB7330_ETXETAR_ROBOT_CELL_INTERLOCK".INTERLOCKS_UNIT_02.MACHINE_TO_ROBOT.MCH_UNLD_ANTICIPATION_FACE_R )
      I_Contact( "DB7300_INTERLOCK_GENERAL".LOAD_UNLOAD.UNIT_2.FROM_ROBOT_CELL.PART_UNLOADED_P )
   END_RUNG wire#w1
   // the same network as SCL:
   "DB7330_ETXETAR_ROBOT_CELL_INTERLOCK".INTERLOCKS_UNIT_02.MACHINE_TO_ROBOT.MCH_UNLD_ANTICIPATION_FACE_R := (("DB5000_FIX_TABLE_POSITIONS".UNIT_2.FIXTURE[1].IN_CLEAN_STATION_4 AND "DB2430_FULL_DEPTH".FD_UNIT_02.FIXTURE_1.FULL_DEPTH_STA_4) OR ("DB5000_FIX_TABLE_POSITIONS".UNIT_2.FIXTURE[3].IN_CLEAN_STATION_4 AND "DB2430_FULL_DEPTH".FD_UNIT_02.FIXTURE_3.FULL_DEPTH_STA_4) OR ("DB7330_ETXETAR_ROBOT_CELL_INTERLOCK".INTERLOCKS_UNIT_02.MACHINE_TO_ROBOT.MCH_UNLD_ANTICIPATION_FACE_R AND NOT "DB7300_INTERLOCK_GENERAL".LOAD_UNLOAD.UNIT_2.FROM_ROBOT_CELL.PART_UNLOADED_P)) AND NOT "DB440_MACHINE_ALARM_DECODING".GLOBAL_ALARMS_MACHINE.SEOC_WARNING AND NOT "DB2031_CYCLES_GENERAL".MANUAL_LOAD_CYCLE.CYCLE_SELECTED AND "DB2001_MODES_GENERAL".MG1.GENERAL.AUTOMATIC_SELECTED AND "DB1251_PART_CYCLE_UNIT_2".RUNNING;
END_REGION

REGION Network 86: MACHINE UNLOAD ANTICIPATION FACE N
   RUNG wire#powerrail
      Contact( "DB5000_FIX_TABLE_POSITIONS".UNIT_2.FIXTURE[2].IN_CLEAN_STATION_4 )
      Contact( "DB2430_FULL_DEPTH".FD_UNIT_02.FIXTURE_2.FULL_DEPTH_STA_4 )
      wire#w1
      I_Contact( "DB440_MACHINE_ALARM_DECODING".GLOBAL_ALARMS_MACHINE.SEOC_WARNING )
      I_Contact( "DB2031_CYCLES_GENERAL".MANUAL_LOAD_CYCLE.CYCLE_SELECTED )
      Contact( "DB2001_MODES_GENERAL".MG1.GENERAL.AUTOMATIC_SELECTED )
      Contact( "DB1251_PART_CYCLE_UNIT_2".RUNNING )
      Coil( "DB7330_ETXETAR_ROBOT_CELL_INTERLOCK".INTERLOCKS_UNIT_02.MACHINE_TO_ROBOT.MCH_UNLD_ANTICIPATION_FACE_N )
   END_RUNG
   RUNG wire#powerrail
      Contact( "DB5000_FIX_TABLE_POSITIONS".UNIT_2.FIXTURE[4].IN_CLEAN_STATION_4 )
      Contact( "DB2430_FULL_DEPTH".FD_UNIT_02.FIXTURE_4.FULL_DEPTH_STA_4 )
   END_RUNG wire#w1
   RUNG wire#powerrail
      Contact( "DB7330_ETXETAR_ROBOT_CELL_INTERLOCK".INTERLOCKS_UNIT_02.MACHINE_TO_ROBOT.MCH_UNLD_ANTICIPATION_FACE_N )
      I_Contact( "DB7300_INTERLOCK_GENERAL".LOAD_UNLOAD.UNIT_2.FROM_ROBOT_CELL.PART_UNLOADED_P )
   END_RUNG wire#w1
   // the same network as SCL:
   "DB7330_ETXETAR_ROBOT_CELL_INTERLOCK".INTERLOCKS_UNIT_02.MACHINE_TO_ROBOT.MCH_UNLD_ANTICIPATION_FACE_N := (("DB5000_FIX_TABLE_POSITIONS".UNIT_2.FIXTURE[2].IN_CLEAN_STATION_4 AND "DB2430_FULL_DEPTH".FD_UNIT_02.FIXTURE_2.FULL_DEPTH_STA_4) OR ("DB5000_FIX_TABLE_POSITIONS".UNIT_2.FIXTURE[4].IN_CLEAN_STATION_4 AND "DB2430_FULL_DEPTH".FD_UNIT_02.FIXTURE_4.FULL_DEPTH_STA_4) OR ("DB7330_ETXETAR_ROBOT_CELL_INTERLOCK".INTERLOCKS_UNIT_02.MACHINE_TO_ROBOT.MCH_UNLD_ANTICIPATION_FACE_N AND NOT "DB7300_INTERLOCK_GENERAL".LOAD_UNLOAD.UNIT_2.FROM_ROBOT_CELL.PART_UNLOADED_P)) AND NOT "DB440_MACHINE_ALARM_DECODING".GLOBAL_ALARMS_MACHINE.SEOC_WARNING AND NOT "DB2031_CYCLES_GENERAL".MANUAL_LOAD_CYCLE.CYCLE_SELECTED AND "DB2001_MODES_GENERAL".MG1.GENERAL.AUTOMATIC_SELECTED AND "DB1251_PART_CYCLE_UNIT_2".RUNNING;
END_REGION

REGION Network 87: MACHINE LOAD ANTICIPATION FACE R
   RUNG wire#powerrail
      Contact( "DB2001_MODES_GENERAL".MG1.GENERAL.AUTOMATIC_SELECTED )
      I_Contact( "DB2031_CYCLES_GENERAL".MANUAL_LOAD_CYCLE.CYCLE_SELECTED )
      wire#w1
      Contact( "DB1253_UNIT_2_STATION_1_CYCLE".SEQUENCE.RUNNING )
      wire#w2
      Contact( "DB5000_FIX_TABLE_POSITIONS".UNIT_2.FIXTURE[1].IN_LOAD_UNLOAD_STATION_1 )
      I_Contact( "DB8000_PART_STATUS".UNIT_2.FIXTURE_1.PART_A.STATUS.PRESENT )
      wire#w3
      Coil( "DB7330_ETXETAR_ROBOT_CELL_INTERLOCK".INTERLOCKS_UNIT_02.MACHINE_TO_ROBOT.MCH_LOAD_ANTICIPATION_FACE_R )
   END_RUNG
   RUNG wire#w1
      Contact( "DB1274_UNIT_2_STATION_2_MEAS_CALIBRATION".SEQUENCE.RUNNING )
   END_RUNG wire#w2
   RUNG wire#w1
      Contact( "DB1275_UNIT_2_STATION_3_MEAS_CALIBRATION".SEQUENCE.RUNNING )
   END_RUNG wire#w2
   RUNG wire#w2
      Contact( "DB5000_FIX_TABLE_POSITIONS".UNIT_2.FIXTURE[3].IN_LOAD_UNLOAD_STATION_1 )
      I_Contact( "DB8000_PART_STATUS".UNIT_2.FIXTURE_3.PART_A.STATUS.PRESENT )
   END_RUNG wire#w3
   // the same network as SCL:
   "DB7330_ETXETAR_ROBOT_CELL_INTERLOCK".INTERLOCKS_UNIT_02.MACHINE_TO_ROBOT.MCH_LOAD_ANTICIPATION_FACE_R := "DB2001_MODES_GENERAL".MG1.GENERAL.AUTOMATIC_SELECTED AND NOT "DB2031_CYCLES_GENERAL".MANUAL_LOAD_CYCLE.CYCLE_SELECTED AND ("DB1253_UNIT_2_STATION_1_CYCLE".SEQUENCE.RUNNING OR "DB1274_UNIT_2_STATION_2_MEAS_CALIBRATION".SEQUENCE.RUNNING OR "DB1275_UNIT_2_STATION_3_MEAS_CALIBRATION".SEQUENCE.RUNNING) AND (("DB5000_FIX_TABLE_POSITIONS".UNIT_2.FIXTURE[1].IN_LOAD_UNLOAD_STATION_1 AND NOT "DB8000_PART_STATUS".UNIT_2.FIXTURE_1.PART_A.STATUS.PRESENT) OR ("DB5000_FIX_TABLE_POSITIONS".UNIT_2.FIXTURE[3].IN_LOAD_UNLOAD_STATION_1 AND NOT "DB8000_PART_STATUS".UNIT_2.FIXTURE_3.PART_A.STATUS.PRESENT));
END_REGION

REGION Network 88: MACHINE LOAD ANTICIPATION FACE N
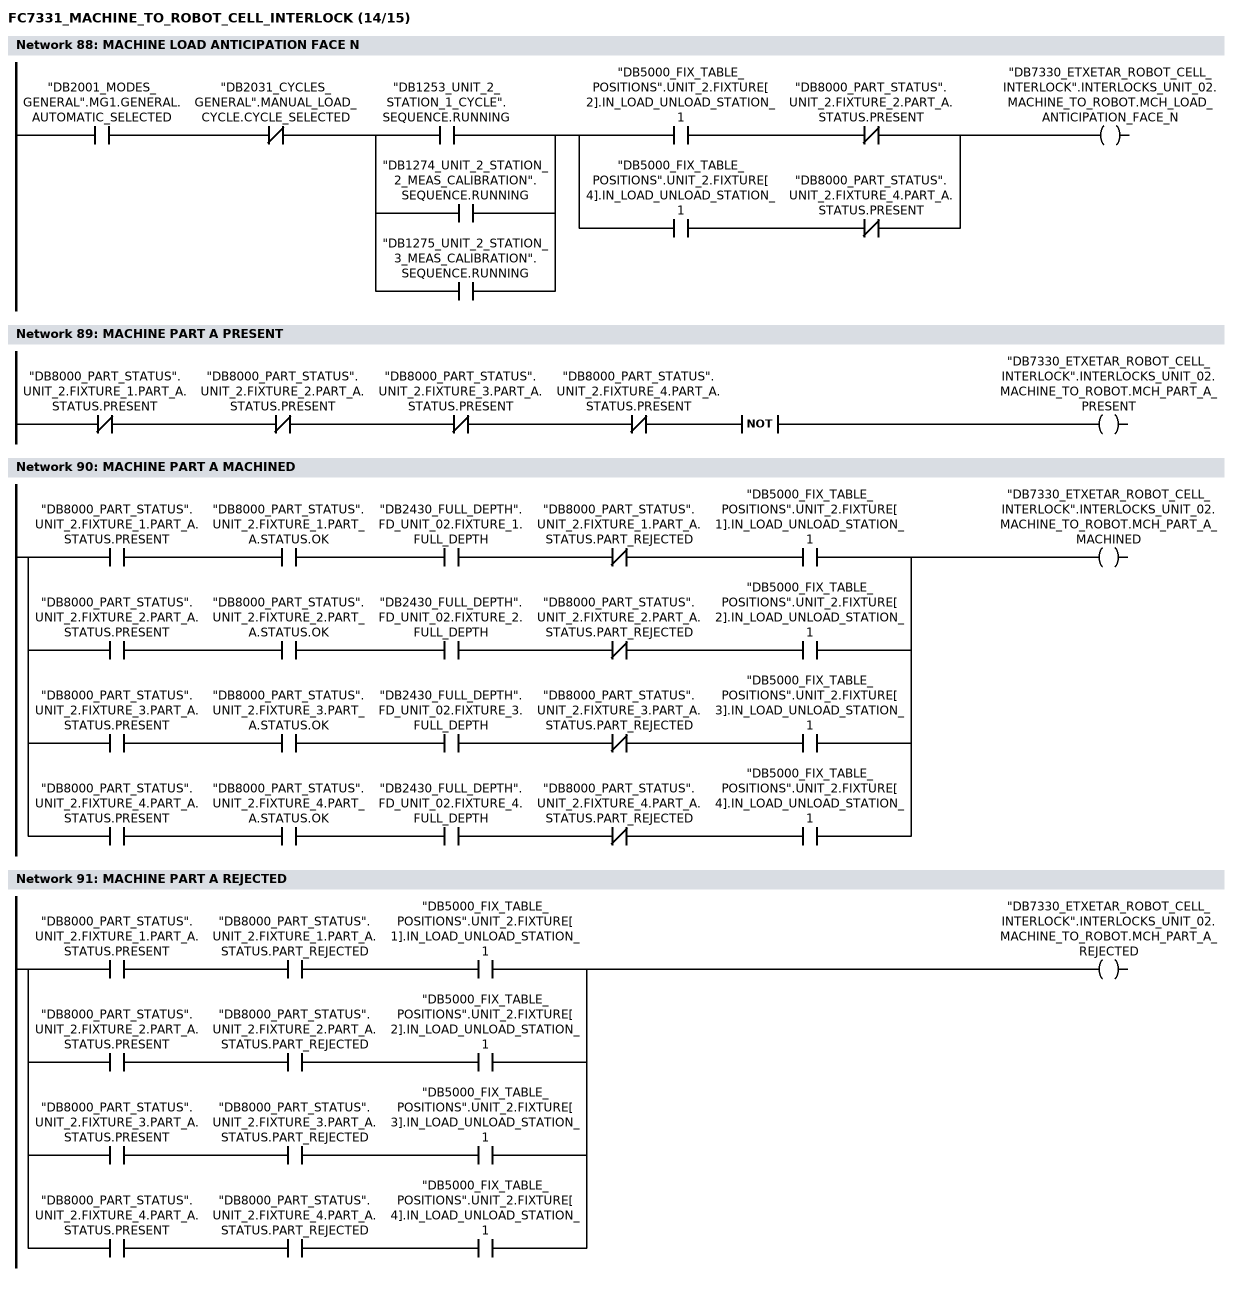
   RUNG wire#powerrail
      Contact( "DB2001_MODES_GENERAL".MG1.GENERAL.AUTOMATIC_SELECTED )
      I_Contact( "DB2031_CYCLES_GENERAL".MANUAL_LOAD_CYCLE.CYCLE_SELECTED )
      wire#w1
      Contact( "DB1253_UNIT_2_STATION_1_CYCLE".SEQUENCE.RUNNING )
      wire#w2
      Contact( "DB5000_FIX_TABLE_POSITIONS".UNIT_2.FIXTURE[2].IN_LOAD_UNLOAD_STATION_1 )
      I_Contact( "DB8000_PART_STATUS".UNIT_2.FIXTURE_2.PART_A.STATUS.PRESENT )
      wire#w3
      Coil( "DB7330_ETXETAR_ROBOT_CELL_INTERLOCK".INTERLOCKS_UNIT_02.MACHINE_TO_ROBOT.MCH_LOAD_ANTICIPATION_FACE_N )
   END_RUNG
   RUNG wire#w1
      Contact( "DB1274_UNIT_2_STATION_2_MEAS_CALIBRATION".SEQUENCE.RUNNING )
   END_RUNG wire#w2
   RUNG wire#w1
      Contact( "DB1275_UNIT_2_STATION_3_MEAS_CALIBRATION".SEQUENCE.RUNNING )
   END_RUNG wire#w2
   RUNG wire#w2
      Contact( "DB5000_FIX_TABLE_POSITIONS".UNIT_2.FIXTURE[4].IN_LOAD_UNLOAD_STATION_1 )
      I_Contact( "DB8000_PART_STATUS".UNIT_2.FIXTURE_4.PART_A.STATUS.PRESENT )
   END_RUNG wire#w3
   // the same network as SCL:
   "DB7330_ETXETAR_ROBOT_CELL_INTERLOCK".INTERLOCKS_UNIT_02.MACHINE_TO_ROBOT.MCH_LOAD_ANTICIPATION_FACE_N := "DB2001_MODES_GENERAL".MG1.GENERAL.AUTOMATIC_SELECTED AND NOT "DB2031_CYCLES_GENERAL".MANUAL_LOAD_CYCLE.CYCLE_SELECTED AND ("DB1253_UNIT_2_STATION_1_CYCLE".SEQUENCE.RUNNING OR "DB1274_UNIT_2_STATION_2_MEAS_CALIBRATION".SEQUENCE.RUNNING OR "DB1275_UNIT_2_STATION_3_MEAS_CALIBRATION".SEQUENCE.RUNNING) AND (("DB5000_FIX_TABLE_POSITIONS".UNIT_2.FIXTURE[2].IN_LOAD_UNLOAD_STATION_1 AND NOT "DB8000_PART_STATUS".UNIT_2.FIXTURE_2.PART_A.STATUS.PRESENT) OR ("DB5000_FIX_TABLE_POSITIONS".UNIT_2.FIXTURE[4].IN_LOAD_UNLOAD_STATION_1 AND NOT "DB8000_PART_STATUS".UNIT_2.FIXTURE_4.PART_A.STATUS.PRESENT));
END_REGION

REGION Network 89: MACHINE PART A PRESENT
   RUNG wire#powerrail
      I_Contact( "DB8000_PART_STATUS".UNIT_2.FIXTURE_1.PART_A.STATUS.PRESENT )
      I_Contact( "DB8000_PART_STATUS".UNIT_2.FIXTURE_2.PART_A.STATUS.PRESENT )
      I_Contact( "DB8000_PART_STATUS".UNIT_2.FIXTURE_3.PART_A.STATUS.PRESENT )
      I_Contact( "DB8000_PART_STATUS".UNIT_2.FIXTURE_4.PART_A.STATUS.PRESENT )
      Not()
      Coil( "DB7330_ETXETAR_ROBOT_CELL_INTERLOCK".INTERLOCKS_UNIT_02.MACHINE_TO_ROBOT.MCH_PART_A_PRESENT )
   END_RUNG
   // the same network as SCL:
   "DB7330_ETXETAR_ROBOT_CELL_INTERLOCK".INTERLOCKS_UNIT_02.MACHINE_TO_ROBOT.MCH_PART_A_PRESENT := NOT (NOT "DB8000_PART_STATUS".UNIT_2.FIXTURE_1.PART_A.STATUS.PRESENT AND NOT "DB8000_PART_STATUS".UNIT_2.FIXTURE_2.PART_A.STATUS.PRESENT AND NOT "DB8000_PART_STATUS".UNIT_2.FIXTURE_3.PART_A.STATUS.PRESENT AND NOT "DB8000_PART_STATUS".UNIT_2.FIXTURE_4.PART_A.STATUS.PRESENT);
END_REGION

REGION Network 90: MACHINE PART A MACHINED
   RUNG wire#powerrail
      Contact( "DB8000_PART_STATUS".UNIT_2.FIXTURE_1.PART_A.STATUS.PRESENT )
      Contact( "DB8000_PART_STATUS".UNIT_2.FIXTURE_1.PART_A.STATUS.OK )
      Contact( "DB2430_FULL_DEPTH".FD_UNIT_02.FIXTURE_1.FULL_DEPTH )
      I_Contact( "DB8000_PART_STATUS".UNIT_2.FIXTURE_1.PART_A.STATUS.PART_REJECTED )
      Contact( "DB5000_FIX_TABLE_POSITIONS".UNIT_2.FIXTURE[1].IN_LOAD_UNLOAD_STATION_1 )
      wire#w1
      Coil( "DB7330_ETXETAR_ROBOT_CELL_INTERLOCK".INTERLOCKS_UNIT_02.MACHINE_TO_ROBOT.MCH_PART_A_MACHINED )
   END_RUNG
   RUNG wire#powerrail
      Contact( "DB8000_PART_STATUS".UNIT_2.FIXTURE_2.PART_A.STATUS.PRESENT )
      Contact( "DB8000_PART_STATUS".UNIT_2.FIXTURE_2.PART_A.STATUS.OK )
      Contact( "DB2430_FULL_DEPTH".FD_UNIT_02.FIXTURE_2.FULL_DEPTH )
      I_Contact( "DB8000_PART_STATUS".UNIT_2.FIXTURE_2.PART_A.STATUS.PART_REJECTED )
      Contact( "DB5000_FIX_TABLE_POSITIONS".UNIT_2.FIXTURE[2].IN_LOAD_UNLOAD_STATION_1 )
   END_RUNG wire#w1
   RUNG wire#powerrail
      Contact( "DB8000_PART_STATUS".UNIT_2.FIXTURE_3.PART_A.STATUS.PRESENT )
      Contact( "DB8000_PART_STATUS".UNIT_2.FIXTURE_3.PART_A.STATUS.OK )
      Contact( "DB2430_FULL_DEPTH".FD_UNIT_02.FIXTURE_3.FULL_DEPTH )
      I_Contact( "DB8000_PART_STATUS".UNIT_2.FIXTURE_3.PART_A.STATUS.PART_REJECTED )
      Contact( "DB5000_FIX_TABLE_POSITIONS".UNIT_2.FIXTURE[3].IN_LOAD_UNLOAD_STATION_1 )
   END_RUNG wire#w1
   RUNG wire#powerrail
      Contact( "DB8000_PART_STATUS".UNIT_2.FIXTURE_4.PART_A.STATUS.PRESENT )
      Contact( "DB8000_PART_STATUS".UNIT_2.FIXTURE_4.PART_A.STATUS.OK )
      Contact( "DB2430_FULL_DEPTH".FD_UNIT_02.FIXTURE_4.FULL_DEPTH )
      I_Contact( "DB8000_PART_STATUS".UNIT_2.FIXTURE_4.PART_A.STATUS.PART_REJECTED )
      Contact( "DB5000_FIX_TABLE_POSITIONS".UNIT_2.FIXTURE[4].IN_LOAD_UNLOAD_STATION_1 )
   END_RUNG wire#w1
   // the same network as SCL:
   "DB7330_ETXETAR_ROBOT_CELL_INTERLOCK".INTERLOCKS_UNIT_02.MACHINE_TO_ROBOT.MCH_PART_A_MACHINED := ("DB8000_PART_STATUS".UNIT_2.FIXTURE_1.PART_A.STATUS.PRESENT AND "DB8000_PART_STATUS".UNIT_2.FIXTURE_1.PART_A.STATUS.OK AND "DB2430_FULL_DEPTH".FD_UNIT_02.FIXTURE_1.FULL_DEPTH AND NOT "DB8000_PART_STATUS".UNIT_2.FIXTURE_1.PART_A.STATUS.PART_REJECTED AND "DB5000_FIX_TABLE_POSITIONS".UNIT_2.FIXTURE[1].IN_LOAD_UNLOAD_STATION_1) OR ("DB8000_PART_STATUS".UNIT_2.FIXTURE_2.PART_A.STATUS.PRESENT AND "DB8000_PART_STATUS".UNIT_2.FIXTURE_2.PART_A.STATUS.OK AND "DB2430_FULL_DEPTH".FD_UNIT_02.FIXTURE_2.FULL_DEPTH AND NOT "DB8000_PART_STATUS".UNIT_2.FIXTURE_2.PART_A.STATUS.PART_REJECTED AND "DB5000_FIX_TABLE_POSITIONS".UNIT_2.FIXTURE[2].IN_LOAD_UNLOAD_STATION_1) OR ("DB8000_PART_STATUS".UNIT_2.FIXTURE_3.PART_A.STATUS.PRESENT AND "DB8000_PART_STATUS".UNIT_2.FIXTURE_3.PART_A.STATUS.OK AND "DB2430_FULL_DEPTH".FD_UNIT_02.FIXTURE_3.FULL_DEPTH AND NOT "DB8000_PART_STATUS".UNIT_2.FIXTURE_3.PART_A.STATUS.PART_REJECTED AND "DB5000_FIX_TABLE_POSITIONS".UNIT_2.FIXTURE[3].IN_LOAD_UNLOAD_STATION_1) OR ("DB8000_PART_STATUS".UNIT_2.FIXTURE_4.PART_A.STATUS.PRESENT AND "DB8000_PART_STATUS".UNIT_2.FIXTURE_4.PART_A.STATUS.OK AND "DB2430_FULL_DEPTH".FD_UNIT_02.FIXTURE_4.FULL_DEPTH AND NOT "DB8000_PART_STATUS".UNIT_2.FIXTURE_4.PART_A.STATUS.PART_REJECTED AND "DB5000_FIX_TABLE_POSITIONS".UNIT_2.FIXTURE[4].IN_LOAD_UNLOAD_STATION_1);
END_REGION

REGION Network 91: MACHINE PART A REJECTED
   RUNG wire#powerrail
      Contact( "DB8000_PART_STATUS".UNIT_2.FIXTURE_1.PART_A.STATUS.PRESENT )
      Contact( "DB8000_PART_STATUS".UNIT_2.FIXTURE_1.PART_A.STATUS.PART_REJECTED )
      Contact( "DB5000_FIX_TABLE_POSITIONS".UNIT_2.FIXTURE[1].IN_LOAD_UNLOAD_STATION_1 )
      wire#w1
      Coil( "DB7330_ETXETAR_ROBOT_CELL_INTERLOCK".INTERLOCKS_UNIT_02.MACHINE_TO_ROBOT.MCH_PART_A_REJECTED )
   END_RUNG
   RUNG wire#powerrail
      Contact( "DB8000_PART_STATUS".UNIT_2.FIXTURE_2.PART_A.STATUS.PRESENT )
      Contact( "DB8000_PART_STATUS".UNIT_2.FIXTURE_2.PART_A.STATUS.PART_REJECTED )
      Contact( "DB5000_FIX_TABLE_POSITIONS".UNIT_2.FIXTURE[2].IN_LOAD_UNLOAD_STATION_1 )
   END_RUNG wire#w1
   RUNG wire#powerrail
      Contact( "DB8000_PART_STATUS".UNIT_2.FIXTURE_3.PART_A.STATUS.PRESENT )
      Contact( "DB8000_PART_STATUS".UNIT_2.FIXTURE_3.PART_A.STATUS.PART_REJECTED )
      Contact( "DB5000_FIX_TABLE_POSITIONS".UNIT_2.FIXTURE[3].IN_LOAD_UNLOAD_STATION_1 )
   END_RUNG wire#w1
   RUNG wire#powerrail
      Contact( "DB8000_PART_STATUS".UNIT_2.FIXTURE_4.PART_A.STATUS.PRESENT )
      Contact( "DB8000_PART_STATUS".UNIT_2.FIXTURE_4.PART_A.STATUS.PART_REJECTED )
      Contact( "DB5000_FIX_TABLE_POSITIONS".UNIT_2.FIXTURE[4].IN_LOAD_UNLOAD_STATION_1 )
   END_RUNG wire#w1
   // the same network as SCL:
   "DB7330_ETXETAR_ROBOT_CELL_INTERLOCK".INTERLOCKS_UNIT_02.MACHINE_TO_ROBOT.MCH_PART_A_REJECTED := ("DB8000_PART_STATUS".UNIT_2.FIXTURE_1.PART_A.STATUS.PRESENT AND "DB8000_PART_STATUS".UNIT_2.FIXTURE_1.PART_A.STATUS.PART_REJECTED AND "DB5000_FIX_TABLE_POSITIONS".UNIT_2.FIXTURE[1].IN_LOAD_UNLOAD_STATION_1) OR ("DB8000_PART_STATUS".UNIT_2.FIXTURE_2.PART_A.STATUS.PRESENT AND "DB8000_PART_STATUS".UNIT_2.FIXTURE_2.PART_A.STATUS.PART_REJECTED AND "DB5000_FIX_TABLE_POSITIONS".UNIT_2.FIXTURE[2].IN_LOAD_UNLOAD_STATION_1) OR ("DB8000_PART_STATUS".UNIT_2.FIXTURE_3.PART_A.STATUS.PRESENT AND "DB8000_PART_STATUS".UNIT_2.FIXTURE_3.PART_A.STATUS.PART_REJECTED AND "DB5000_FIX_TABLE_POSITIONS".UNIT_2.FIXTURE[3].IN_LOAD_UNLOAD_STATION_1) OR ("DB8000_PART_STATUS".UNIT_2.FIXTURE_4.PART_A.STATUS.PRESENT AND "DB8000_PART_STATUS".UNIT_2.FIXTURE_4.PART_A.STATUS.PART_REJECTED AND "DB5000_FIX_TABLE_POSITIONS".UNIT_2.FIXTURE[4].IN_LOAD_UNLOAD_STATION_1);
END_REGION

REGION Network 92: MACHINE PART A QUALITY
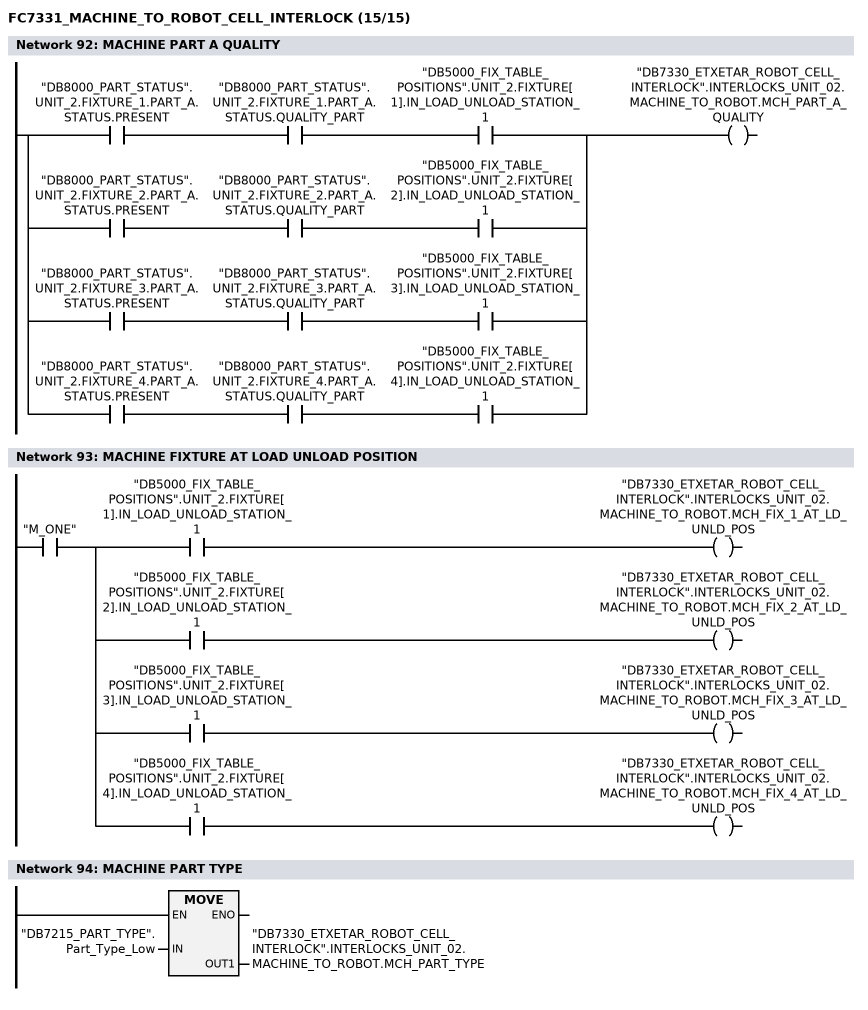
   RUNG wire#powerrail
      Contact( "DB8000_PART_STATUS".UNIT_2.FIXTURE_1.PART_A.STATUS.PRESENT )
      Contact( "DB8000_PART_STATUS".UNIT_2.FIXTURE_1.PART_A.STATUS.QUALITY_PART )
      Contact( "DB5000_FIX_TABLE_POSITIONS".UNIT_2.FIXTURE[1].IN_LOAD_UNLOAD_STATION_1 )
      wire#w1
      Coil( "DB7330_ETXETAR_ROBOT_CELL_INTERLOCK".INTERLOCKS_UNIT_02.MACHINE_TO_ROBOT.MCH_PART_A_QUALITY )
   END_RUNG
   RUNG wire#powerrail
      Contact( "DB8000_PART_STATUS".UNIT_2.FIXTURE_2.PART_A.STATUS.PRESENT )
      Contact( "DB8000_PART_STATUS".UNIT_2.FIXTURE_2.PART_A.STATUS.QUALITY_PART )
      Contact( "DB5000_FIX_TABLE_POSITIONS".UNIT_2.FIXTURE[2].IN_LOAD_UNLOAD_STATION_1 )
   END_RUNG wire#w1
   RUNG wire#powerrail
      Contact( "DB8000_PART_STATUS".UNIT_2.FIXTURE_3.PART_A.STATUS.PRESENT )
      Contact( "DB8000_PART_STATUS".UNIT_2.FIXTURE_3.PART_A.STATUS.QUALITY_PART )
      Contact( "DB5000_FIX_TABLE_POSITIONS".UNIT_2.FIXTURE[3].IN_LOAD_UNLOAD_STATION_1 )
   END_RUNG wire#w1
   RUNG wire#powerrail
      Contact( "DB8000_PART_STATUS".UNIT_2.FIXTURE_4.PART_A.STATUS.PRESENT )
      Contact( "DB8000_PART_STATUS".UNIT_2.FIXTURE_4.PART_A.STATUS.QUALITY_PART )
      Contact( "DB5000_FIX_TABLE_POSITIONS".UNIT_2.FIXTURE[4].IN_LOAD_UNLOAD_STATION_1 )
   END_RUNG wire#w1
   // the same network as SCL:
   "DB7330_ETXETAR_ROBOT_CELL_INTERLOCK".INTERLOCKS_UNIT_02.MACHINE_TO_ROBOT.MCH_PART_A_QUALITY := ("DB8000_PART_STATUS".UNIT_2.FIXTURE_1.PART_A.STATUS.PRESENT AND "DB8000_PART_STATUS".UNIT_2.FIXTURE_1.PART_A.STATUS.QUALITY_PART AND "DB5000_FIX_TABLE_POSITIONS".UNIT_2.FIXTURE[1].IN_LOAD_UNLOAD_STATION_1) OR ("DB8000_PART_STATUS".UNIT_2.FIXTURE_2.PART_A.STATUS.PRESENT AND "DB8000_PART_STATUS".UNIT_2.FIXTURE_2.PART_A.STATUS.QUALITY_PART AND "DB5000_FIX_TABLE_POSITIONS".UNIT_2.FIXTURE[2].IN_LOAD_UNLOAD_STATION_1) OR ("DB8000_PART_STATUS".UNIT_2.FIXTURE_3.PART_A.STATUS.PRESENT AND "DB8000_PART_STATUS".UNIT_2.FIXTURE_3.PART_A.STATUS.QUALITY_PART AND "DB5000_FIX_TABLE_POSITIONS".UNIT_2.FIXTURE[3].IN_LOAD_UNLOAD_STATION_1) OR ("DB8000_PART_STATUS".UNIT_2.FIXTURE_4.PART_A.STATUS.PRESENT AND "DB8000_PART_STATUS".UNIT_2.FIXTURE_4.PART_A.STATUS.QUALITY_PART AND "DB5000_FIX_TABLE_POSITIONS".UNIT_2.FIXTURE[4].IN_LOAD_UNLOAD_STATION_1);
END_REGION

REGION Network 93: MACHINE FIXTURE AT LOAD UNLOAD POSITION
   RUNG wire#powerrail
      Contact( "M_ONE" )
      wire#w1
      Contact( "DB5000_FIX_TABLE_POSITIONS".UNIT_2.FIXTURE[1].IN_LOAD_UNLOAD_STATION_1 )
      Coil( "DB7330_ETXETAR_ROBOT_CELL_INTERLOCK".INTERLOCKS_UNIT_02.MACHINE_TO_ROBOT.MCH_FIX_1_AT_LD_UNLD_POS )
   END_RUNG
   RUNG wire#w1
      Contact( "DB5000_FIX_TABLE_POSITIONS".UNIT_2.FIXTURE[2].IN_LOAD_UNLOAD_STATION_1 )
      Coil( "DB7330_ETXETAR_ROBOT_CELL_INTERLOCK".INTERLOCKS_UNIT_02.MACHINE_TO_ROBOT.MCH_FIX_2_AT_LD_UNLD_POS )
   END_RUNG
   RUNG wire#w1
      Contact( "DB5000_FIX_TABLE_POSITIONS".UNIT_2.FIXTURE[3].IN_LOAD_UNLOAD_STATION_1 )
      Coil( "DB7330_ETXETAR_ROBOT_CELL_INTERLOCK".INTERLOCKS_UNIT_02.MACHINE_TO_ROBOT.MCH_FIX_3_AT_LD_UNLD_POS )
   END_RUNG
   RUNG wire#w1
      Contact( "DB5000_FIX_TABLE_POSITIONS".UNIT_2.FIXTURE[4].IN_LOAD_UNLOAD_STATION_1 )
      Coil( "DB7330_ETXETAR_ROBOT_CELL_INTERLOCK".INTERLOCKS_UNIT_02.MACHINE_TO_ROBOT.MCH_FIX_4_AT_LD_UNLD_POS )
   END_RUNG
   // the same network as SCL:
   "DB7330_ETXETAR_ROBOT_CELL_INTERLOCK".INTERLOCKS_UNIT_02.MACHINE_TO_ROBOT.MCH_FIX_1_AT_LD_UNLD_POS := "M_ONE" AND "DB5000_FIX_TABLE_POSITIONS".UNIT_2.FIXTURE[1].IN_LOAD_UNLOAD_STATION_1;
   "DB7330_ETXETAR_ROBOT_CELL_INTERLOCK".INTERLOCKS_UNIT_02.MACHINE_TO_ROBOT.MCH_FIX_2_AT_LD_UNLD_POS := "M_ONE" AND "DB5000_FIX_TABLE_POSITIONS".UNIT_2.FIXTURE[2].IN_LOAD_UNLOAD_STATION_1;
   "DB7330_ETXETAR_ROBOT_CELL_INTERLOCK".INTERLOCKS_UNIT_02.MACHINE_TO_ROBOT.MCH_FIX_3_AT_LD_UNLD_POS := "M_ONE" AND "DB5000_FIX_TABLE_POSITIONS".UNIT_2.FIXTURE[3].IN_LOAD_UNLOAD_STATION_1;
   "DB7330_ETXETAR_ROBOT_CELL_INTERLOCK".INTERLOCKS_UNIT_02.MACHINE_TO_ROBOT.MCH_FIX_4_AT_LD_UNLD_POS := "M_ONE" AND "DB5000_FIX_TABLE_POSITIONS".UNIT_2.FIXTURE[4].IN_LOAD_UNLOAD_STATION_1;
END_REGION

REGION Network 94: MACHINE PART TYPE
   RUNG wire#powerrail
      { S7_GenerateENO := "TRUE" } Move(in := "DB7215_PART_TYPE".Part_Type_Low, out1 => "DB7330_ETXETAR_ROBOT_CELL_INTERLOCK".INTERLOCKS_UNIT_02.MACHINE_TO_ROBOT.MCH_PART_TYPE)
   END_RUNG
   // the same network as SCL:
   "DB7330_ETXETAR_ROBOT_CELL_INTERLOCK".INTERLOCKS_UNIT_02.MACHINE_TO_ROBOT.MCH_PART_TYPE := "DB7215_PART_TYPE".Part_Type_Low;
END_REGION
END_FUNCTION
